Omron CX-Programmer project 新工程 (CX-Programmer 9.50)

# PLC 金泉负压氦检: CJ2M CPU34
I/O table (CPU CJ2M-CPU34): rack 0 slot 11 CJ2M-EIP21

## Global symbols (name address type ; comment)
0.00 BOOL  ; 扫码1#位有料感应（常闭）
0.01 BOOL  ; 扫码2#位有料感应（常闭）
0.02 BOOL  ; 拉带放料位有料感应（常闭）
0.03 BOOL  ; 上料1#位接近有料感应
0.04 BOOL  ; 上料2#位接近有料感应
0.05 BOOL  ; 扫码左位阻挡气缸缩回位
0.06 BOOL  ; 扫码左位阻挡气缸伸出位
0.07 BOOL  ; 扫码右位阻挡气缸缩回位
0.08 BOOL  ; 扫码右位阻挡气缸伸出位
0.09 BOOL  ; 1#位隔离气缸缩回位
0.10 BOOL  ; 左位隔离气缸伸出位
0.11 BOOL  ; 2#位隔离气缸缩回位
0.12 BOOL  ; 右位隔离气缸伸出位
0.13 BOOL  ; 1#隔离位有料感应
0.14 BOOL  ; 2#隔离位有料感应
0.15 BOOL  ; 备用
100.06 BOOL  ; 异常报警停止
100.11 BOOL  ; 报警中
10.00 BOOL  ; 2#隔离气缸缩回
10.01 BOOL  ; 2#隔离气缸伸出
10.02 BOOL  ; 1#隔离气缸缩回
10.03 BOOL  ; 1#隔离气缸伸出
10.04 BOOL  ; 扫码2#阻挡缩回
10.05 BOOL  ; 扫码2#阻挡伸出
10.06 BOOL  ; 扫码1#阻挡缩回
10.07 BOOL  ; 扫码1#阻挡伸出
10.08 BOOL  ; #1调速电机
10.09 BOOL  ; #2调速电机
10.10 BOOL  ; #3调速电机
10.11 BOOL  ; #4调速电机
10.13 BOOL  ; 进料水平伺服使能
10.14 BOOL  ; 进料升降伺服使能
10.15 BOOL  ; 进料升降伺服刹车
11.00 BOOL  ; 进料旋转伺服使能
11.01 BOOL  ; 扫码缓存推料气缸伸出
11.02 BOOL  ; 扫码缓存推料气缸缩回
11.03 BOOL  ; 进料移栽伸缩气缸伸出
11.04 BOOL  ; 进料移栽伸缩气缸缩回
11.05 BOOL  ; 进料#1夹爪气缸夹紧
11.06 BOOL  ; 进料#1夹爪气缸松开
11.07 BOOL  ; 进料#2夹爪气缸夹紧
11.08 BOOL  ; 进料#2夹爪气缸松开
11.09 BOOL  ; 进料水平伺服报警复位
11.10 BOOL  ; 进料升降伺服报警复位
11.11 BOOL  ; 进料旋转伺服报警复位
11.12 BOOL  ; 备用
11.13 BOOL  ; 腔体上料伺服使能
11.14 BOOL  ; 腔体上料提升气缸下降
11.15 BOOL  ; 腔体上料提升气缸上升
12.00 BOOL  ; 腔体上料#1夹爪气缸夹紧
12.01 BOOL  ; 腔体上料#1夹爪气缸松开
12.02 BOOL  ; 腔体上料#2夹爪气缸夹紧
12.03 BOOL  ; 腔体上料#2夹爪气缸松开
12.04 BOOL  ; 腔体上料#3夹爪气缸夹紧
12.05 BOOL  ; 腔体上料#3夹爪气缸松开
12.06 BOOL  ; 腔体上料#4夹爪气缸夹紧
12.07 BOOL  ; 腔体上料#4夹爪气缸松开
12.08 BOOL  ; 腔体下料伺服使能
12.09 BOOL  ; 腔体下料提升气缸下降
12.10 BOOL  ; 腔体下料提升气缸上升
12.11 BOOL  ; 腔体下料#1夹爪气缸夹紧
12.12 BOOL  ; 腔体下料#1夹爪气缸松开
12.13 BOOL  ; 腔体下料#2夹爪气缸夹紧
12.14 BOOL  ; 腔体下料#2夹爪气缸松开
12.15 BOOL  ; 腔体下料#3夹爪气缸夹紧
1311.00 BOOL  ; #1腔体自检步序开始条件
1311.14 BOOL  ; #1腔体自检步序
1311.15 BOOL  ; #1腔体自检步进
1312 CHANNEL  ; 1#腔体自检
1312.00 BOOL  ; #1腔体自检，数据初始化
1312.01 BOOL  ; #1腔体氦检阀打开、合模
1312.02 BOOL  ; #1腔体抽真空
1312.03 BOOL  ; #1腔体进入自检保压前状态
1312.04 BOOL  ; #1腔体进入自检保压状态
1312.05 BOOL  ; #1腔体破真空步
1312.06 BOOL  ; #1腔体自检完成
1313.00 BOOL  ; #1、#2腔体自动条件
1313.01 BOOL  ; #1、#2腔体自动步序递增条件
1313.02 BOOL  ; #1、#2腔体步进递增
1313.05 BOOL  ; 腔体#1 & #2自动启动
1314 CHANNEL  ; #1腔体自动步序
1314.00 BOOL  ; #1、#2腔体自动步序开始
1314.01 BOOL  ; 关闭#1、#2腔体合模气缸，数据初始化
1314.02 BOOL  ; 开始#1、#2腔体抽真空
1314.03 BOOL  ; #1、#2腔体氦检步
1314.04 BOOL  ; #1、#2腔体氦检结果
1314.05 BOOL  ; #1、#2腔体抽残气步
1314.06 BOOL  ; #1、#2腔体氦检结束，腔体破真空步
1314.07 BOOL  ; #1、#2腔体测试结束，开合模，停止吹气，
1314.08 BOOL  ; #1 & #2腔体一个循环结束
1315.00 BOOL  ; #1、#2腔体复检条件
1315.01 BOOL  ; #1、#2腔体在线复检步序递增条件
1315.02 BOOL  ; #1、#2腔体在线复检步进递增
1316 CHANNEL  ; #1、#2复检前抽真空、破真空步进序号
1316.00 BOOL  ; #1、#2腔体在线复检开始，所有数据初始化
1316.01 BOOL  ; 腔体#1、#2复检前抽真空
1316.02 BOOL  ; #1、#2复检前破真空步
1316.03 BOOL  ; #1、#2复检前关破真空阀、抽真空计数步
1316.04 BOOL  ; #1、#2复检抽真空步
1316.05 BOOL  ; #1、#2复检氦检步
1316.06 BOOL  ; #1、#2复检关氦检阀、破真空(复检)步
1316.07 BOOL  ; #1、#2复检关破真空(复检)步
1316.08 BOOL  ; #1、#2清氦抽真空步
1316.09 BOOL  ; #1、#2清氦抽真空计数步
1316.10 BOOL  ; #1、#2清氦氦检步
1316.11 BOOL  ; #1、#2复检清氦破真空步
1316.12 BOOL  ; #1、#2清氦关破真空步
1316.13 BOOL  ; #1、#2清氦选择步
1316.14 BOOL  ; #1、#2复检结束步
1316.15 BOOL  ; #1、#2复检结束步
1321.00 BOOL  ; #2腔体自检步序开始条件
1321.14 BOOL  ; #2腔体自检步序
1321.15 BOOL  ; #2腔体自检步进
1322 CHANNEL  ; #2腔体自检步序
1322.00 BOOL  ; #2腔体自检，数据初始化
1322.01 BOOL  ; #2腔体氦检阀打开、合模
1322.02 BOOL  ; #2腔体抽真空
1322.03 BOOL  ; #2腔体进入自检保压前状态
1322.04 BOOL  ; #2腔体进入自检保压状态
1322.05 BOOL  ; #2腔体破真空步
1322.06 BOOL  ; #2腔体自检完成
1331.00 BOOL  ; #3腔体自检步序开始条件
1331.14 BOOL  ; #3腔体自检步序
1331.15 BOOL  ; #3腔体自检步进
1332.00 BOOL  ; #3腔体自检，数据初始化
1332.01 BOOL  ; #3腔体氦检阀打开、合模
1332.02 BOOL  ; #3腔体抽真空
1332.03 BOOL  ; #3腔体进入自检保压前状态
1332.04 BOOL  ; #3腔体进入自检保压状态
1332.05 BOOL  ; #3腔体破真空步
1332.06 BOOL  ; #3腔体自检完成
1333.00 BOOL  ; #3、#4腔体自动条件
1333.01 BOOL  ; #3、#4腔体自动步序递增条件
1333.02 BOOL  ; #3、#4腔体步进递增
1333.05 BOOL  ; 腔体#3 & #4自动启动
1334 CHANNEL  ; #3、#4腔体自动步序
1334.00 BOOL  ; #3、#4腔体自动步序开始
1334.01 BOOL  ; 关闭#3、#4腔体合模气缸，数据初始化
1334.02 BOOL  ; 开始#3、#4腔体抽真空
1334.03 BOOL  ; #3、#4腔体氦检步
1334.04 BOOL  ; #3、#4腔体氦检结果
1334.05 BOOL  ; #3、#4腔体抽残气步
1334.06 BOOL  ; #3、#4腔体氦检结束，腔体破真空步
1334.07 BOOL  ; #3、#4腔体测试结束，开合模，停止吹气，
1334.08 BOOL  ; #3 & #4腔体一个循环结束
1335.00 BOOL  ; #3、#4腔体复检条件
1335.01 BOOL  ; #3、#4腔体在线复检步序递增条件
1335.02 BOOL  ; #3、#4腔体在线复检步进递增
1336 CHANNEL  ; #3、#4复检前抽真空、破真空步进序号
1336.00 BOOL  ; #3、#4腔体在线复检开始，所有数据初始化
1336.01 BOOL  ; 腔体#3、#4复检前抽真空
1336.02 BOOL  ; #3、#4复检前破真空步
1336.03 BOOL  ; #3、#4复检前关破真空阀、抽真空计数步
1336.04 BOOL  ; #3、#4复检抽真空步
1336.05 BOOL  ; #3、#4复检氦检步
1336.06 BOOL  ; #3、#4复检关氦检阀、破真空(复检)步
1336.07 BOOL  ; #3、#4复检关破真空(复检)步
1336.08 BOOL  ; #3、#4清氦抽真空步
1336.09 BOOL  ; #3、#4清氦抽真空计数步
1336.10 BOOL  ; #3、#4清氦氦检步
1336.11 BOOL  ; #3、#4复检清氦破真空步
1336.12 BOOL  ; #3、#4清氦关破真空步
1336.13 BOOL  ; #3、#4清氦选择步
1336.14 BOOL  ; #3、#4复检结束步
1336.15 BOOL  ; #3、#4复检结束步
1341.00 BOOL  ; #4腔体自检步序开始条件
1341.14 BOOL  ; #4腔体自检步序
1341.15 BOOL  ; #4腔体自检步进
1342.00 BOOL  ; #4腔体自检，数据初始化
1342.01 BOOL  ; #4腔体氦检阀打开、合模
1342.02 BOOL  ; #4腔体抽真空
1342.03 BOOL  ; #4腔体进入自检保压前状态
1342.04 BOOL  ; #4腔体进入自检保压状态
1342.05 BOOL  ; #4腔体破真空步
1342.06 BOOL  ; #4腔体自检完成
1343.00 BOOL  ; 上料水平伺服自动开始条件
1343.01 BOOL  ; 上料水平伺服自动步序递增条件
1343.02 BOOL  ; 上料水平伺服步进递增
1343.05 BOOL  ; 上料机构手自动启动
1344 CHANNEL  ; 上料水平伺服步序
1344.00 BOOL  ; 上料水平伺服开始
1344.01 BOOL  ; 上料水平伺服到取料位
1344.02 BOOL  ; 抓取料
1344.03 BOOL  ; 上料提升气缸回升
1344.04 BOOL  ; 判断腔体放料位置（优先放#1腔体）
1344.05 BOOL  ; 在腔体位置放料
1344.06 BOOL  ; 放料完成，数据传递，气缸回升
1344.07 BOOL  ; 上料水平伺服回上料位
1345.00 BOOL  ; 下料水平伺服自动开始
1345.01 BOOL  ; 下料水平伺服自动步序递增条件
1345.02 BOOL  ; 下料水平伺服步进
1345.05 BOOL  ; 下料机构手自动启动
1345.08 BOOL  ; 放料完成
1346 CHANNEL  ; 下料水平伺服步序
1346.00 BOOL  ; 下料水平伺服步进开始
1346.01 BOOL  ; 下料机构手在放料位判断取料位置(优先取#1腔体)
1346.02 BOOL  ; 下料机构手去腔体(优先取#1腔体)
1346.03 BOOL  ; 下料机构手在腔体位置下降取料
1346.04 BOOL  ; 下料机构手腔体夹料
1346.05 BOOL  ; 机构手上升 腔体→下料夹爪数据传递
1346.06 BOOL  ; 下料机构手回放料位
1346.07 BOOL  ; 下料机构手下降
1346.08 BOOL  ; 下料水平伺服放料松夹
1346.09 BOOL  ; 下料水平伺服放料完成，数据传递，气缸回升
1346.10 BOOL  ; 下料机手一个循环结束
1350.00 BOOL  ; 4-1旋转_Ready Status
1350.01 BOOL  ; 4-1旋转_Home
1350.02 BOOL  ; 4-1旋转_Sub Home
1350.03 BOOL  ; 4-1旋转_Error
1350.04 BOOL  ; 4-1旋转_Warning
1350.05 BOOL  ; 4-1旋转_Home Cmd
1350.06 BOOL  ; 4-1旋转_Auto Stop CMD
1350.07 BOOL  ; 4-1旋转_Stop Cmplt
1350.08 BOOL  ; 4-1旋转_Interlock
1350.09 BOOL  ; 4-1旋转_1Cycle CMD
1350.10 BOOL  ; 4-1旋转_Step+1C+Run
1350.11 BOOL  ; 4-1旋转_1-Cycle End
1350.12 BOOL  ; 4-1旋转_Task Start
1350.13 BOOL  ; 4-1旋转_Task INC Condition
1350.14 BOOL  ; 4-1旋转_Task INC
1350.15 BOOL  ; 4-1旋转_Task Cmplt
1351.00 BOOL  ; 4-1旋转_Cell Move Home SW[T]
1351.01 BOOL  ; 4-1旋转_Step SW[T]
1351.02 BOOL  ; 4-1旋转_1Cycle SW[T]
1351.03 BOOL  ; 4-1旋转_Task Stop SW [T]
1351.04 BOOL  ; 4-1旋转_Task Cmplt SW[T]
1351.05 BOOL  ; 4-1旋转_Task Cmplt Rst SW[T]
1351.06 BOOL  ; 4-1旋转_Product Data Clear SW[T]
1351.07 BOOL  ; 4-1旋转_
1351.08 BOOL  ; 4-1旋转_
1351.09 BOOL  ; 4-1旋转_
1351.10 BOOL  ; 4-1旋转_Step CMD
1351.11 BOOL  ; 4-1旋转_Initial CMD
1351.12 BOOL  ; 4-1旋转_
1351.13 BOOL  ; 4-1旋转_
1351.14 BOOL  ; 4-1旋转_
1351.15 BOOL  ; 4-1旋转_
1352.00 BOOL  ; 4-1旋转_→请求放料
1352.01 BOOL  ; 4-1旋转_←允许旋转
1352.02 BOOL  ; 4-1旋转_→请求取料1&2
1352.03 BOOL  ; 4-1旋转_→请求取料3&4
1352.04 BOOL  ; 4-1旋转_Allow Idx Act-4
1352.05 BOOL  ; 4-1旋转_Allow Idx Act-5
1352.06 BOOL  ; 4-1旋转_Allow Idx Act-6
1352.07 BOOL  ; 4-1旋转_Allow Idx Act-7
1352.08 BOOL  ; 4-1旋转_Allow Idx Act-8
1352.09 BOOL  ; 4-1旋转_Allow Idx Act-9
1352.10 BOOL  ; 4-1旋转_Allow Idx Act-10
1352.11 BOOL  ; 4-1旋转_Allow Idx Act-11
1352.12 BOOL  ; 4-1旋转_Allow Idx Act-12
1352.13 BOOL  ; 4-1旋转_←4-2允许旋转
1352.14 BOOL  ; 4-1旋转_←上下料允许旋转
1352.15 BOOL  ; 4-1旋转_Allow Idx Act-15
1353.00 BOOL  ; 4-1旋转_Step No.
1353.01 BOOL  ; 4-1旋转_
1353.02 BOOL  ; 4-1旋转_
1353.03 BOOL  ; 4-1旋转_
1353.04 BOOL  ; 4-1旋转_
1353.05 BOOL  ; 4-1旋转_
1353.06 BOOL  ; 4-1旋转_
1353.07 BOOL  ; 4-1旋转_
1353.08 BOOL  ; 4-1旋转_
1353.09 BOOL  ; 4-1旋转_
1353.10 BOOL  ; 4-1旋转_
1353.11 BOOL  ; 4-1旋转_
1353.12 BOOL  ; 4-1旋转_
1353.13 BOOL  ; 4-1旋转_
1353.14 BOOL  ; 4-1旋转_
1353.15 BOOL  ; 4-1旋转_
1354 CHANNEL  ; 4-1_出料旋转不序号
1354.00 BOOL  ; 4-1旋转_Run Start
1354.01 BOOL  ; 4-1旋转_Stp001 →请求放料
1354.02 BOOL  ; 4-1旋转_Stp002 ←允许旋转
1354.03 BOOL  ; 4-1旋转_Stp003
1354.04 BOOL  ; 4-1旋转_Stp004 旋转至1&2#放料位/移至放料位
1354.05 BOOL  ; 4-1旋转_Stp005 →请求4-2取料
1354.06 BOOL  ; 4-1旋转_Stp006 ←4-1允许旋转
1354.07 BOOL  ; 4-1旋转_Stp007
1354.08 BOOL  ; 4-1旋转_Stp008 4-1旋转_Stp004 旋转至3&4#放料位
1354.09 BOOL  ; 4-1旋转_Stp009→请求4-2取料
1354.10 BOOL  ; 4-1旋转_Stp010←4-1允许旋转
1354.11 BOOL  ; 4-1旋转_Stp011 旋转至待机位/移至装载位
1354.12 BOOL  ; 4-1旋转_Stp012
1354.13 BOOL  ; 4-1旋转_Stp013
1354.14 BOOL  ; 4-1旋转_Stp014
1354.15 BOOL  ; 4-1旋转_Stp015
1355.00 BOOL  ; 4-1旋转_Stp016
1355.01 BOOL  ; 4-1旋转_Stp017
1355.02 BOOL  ; 4-1旋转_Stp018
1355.03 BOOL  ; 4-1旋转_Stp019
1355.04 BOOL  ; 4-1旋转_Stp020
1355.05 BOOL  ; 4-1旋转_Stp021
1355.06 BOOL  ; 4-1旋转_Stp022
1355.07 BOOL  ; 4-1旋转_Stp023
1355.08 BOOL  ; 4-1旋转_Stp024
1355.09 BOOL  ; 4-1旋转_Stp025
1355.10 BOOL  ; 4-1旋转_Stp026
1355.11 BOOL  ; 4-1旋转_Stp027
1355.12 BOOL  ; 4-1旋转_Stp028
1355.13 BOOL  ; 4-1旋转_Stp029
1355.14 BOOL  ; 4-1旋转_Stp030
1355.15 BOOL  ; 4-1旋转_Stp031
1356.00 BOOL  ; 4-1旋转_Home
1356.01 BOOL  ; 4-1旋转_Sub Home
1356.02 BOOL  ; 4-1旋转_
1356.03 BOOL  ; 4-1旋转_
1356.04 BOOL  ; 4-1旋转_
1356.05 BOOL  ; 4-1旋转_
1356.06 BOOL  ; 4-1旋转_
1356.07 BOOL  ; 4-1旋转_
1356.08 BOOL  ; 4-1旋转_
1356.09 BOOL  ; 4-1旋转_
1356.10 BOOL  ; 4-1旋转_
1356.11 BOOL  ; 4-1旋转_
1356.12 BOOL  ; 4-1旋转_
1356.13 BOOL  ; 4-1旋转_
1356.14 BOOL  ; 4-1旋转_
1356.15 BOOL  ; 4-1旋转_
1357.00 BOOL  ; 4-1旋转_Error
1357.01 BOOL  ; 4-1旋转_Warning
1357.02 BOOL  ; 4-1旋转_Step+1C+Run
1357.03 BOOL  ; 4-1旋转_
1357.04 BOOL  ; 4-1旋转_
1357.05 BOOL  ; 4-1旋转_
1357.06 BOOL  ; 4-1旋转_
1357.07 BOOL  ; 4-1旋转_
1357.08 BOOL  ; 4-1旋转_
1357.09 BOOL  ; 4-1旋转_
1357.10 BOOL  ; 4-1旋转_
1357.11 BOOL  ; 4-1旋转_
1357.12 BOOL  ; 4-1旋转_
1357.13 BOOL  ; 4-1旋转_
1357.14 BOOL  ; 4-1旋转_
1357.15 BOOL  ; 4-1旋转_
1358.00 BOOL  ; 4-1旋转_
1358.01 BOOL  ; 4-1旋转_
1358.02 BOOL  ; 4-1旋转_
1358.03 BOOL  ; 4-1旋转_
1358.04 BOOL  ; 4-1旋转_
1358.05 BOOL  ; 4-1旋转_
1358.06 BOOL  ; 4-1旋转_
1358.07 BOOL  ; 4-1旋转_
1358.08 BOOL  ; 4-1旋转_
1358.09 BOOL  ; 4-1旋转_
1358.10 BOOL  ; 4-1旋转_
1358.11 BOOL  ; 4-1旋转_
1358.12 BOOL  ; 4-1旋转_
1358.13 BOOL  ; 4-1旋转_
1358.14 BOOL  ; 4-1旋转_
1358.15 BOOL  ; 4-1旋转_
1359.00 BOOL  ; 4-1旋转_Initial-1
1359.01 BOOL  ; 4-1旋转_Initial-2
1359.02 BOOL  ; 4-1旋转_Initial-3
1359.03 BOOL  ; 4-1旋转_Initial-4
1359.04 BOOL  ; 4-1旋转_Initial-5
1359.05 BOOL  ; 4-1旋转_Initial-6
1359.06 BOOL  ; 4-1旋转_Initial-7
1359.07 BOOL  ; 4-1旋转_Initial-8
1359.08 BOOL  ; 4-1旋转_Initial-9
1359.09 BOOL  ; 4-1旋转_Initial-10
1359.10 BOOL  ; 4-1旋转_Initial-11
1359.11 BOOL  ; 4-1旋转_Initial-12
1359.12 BOOL  ; 4-1旋转_Initial-13
1359.13 BOOL  ; 4-1旋转_Initial-14
1359.14 BOOL  ; 4-1旋转_Initial-15
1359.15 BOOL  ; 4-1旋转_Initial-16
1360.00 BOOL  ; 4-2出料模组_Ready Status
1360.01 BOOL  ; 4-2出料模组_Home
1360.02 BOOL  ; 4-2出料模组_Sub Home
1360.03 BOOL  ; 4-2出料模组_Error
1360.04 BOOL  ; 4-2出料模组_Warning
1360.05 BOOL  ; 4-2出料模组_Home Cmd
1360.06 BOOL  ; 4-2出料模组_Auto Stop CMD
1360.07 BOOL  ; 4-2出料模组_Stop Cmplt
1360.08 BOOL  ; 4-2出料模组_Interlock
1360.09 BOOL  ; 4-2出料模组_1Cycle CMD
1360.10 BOOL  ; 4-2出料模组_Step+1C+Run
1360.11 BOOL  ; 4-2出料模组_1-Cycle End
1360.12 BOOL  ; 4-2出料模组_Task Start
1360.13 BOOL  ; 4-2出料模组_Task INC Condition
1360.14 BOOL  ; 4-2出料模组_Task INC
1360.15 BOOL  ; 4-2出料模组_Task Cmplt
1361.00 BOOL  ; 4-2出料模组_Cell Move Home SW[T]
1361.01 BOOL  ; 4-2出料模组_Step SW[T]
1361.02 BOOL  ; 4-2出料模组_1Cycle SW[T]
1361.03 BOOL  ; 4-2出料模组_Task Stop SW [T]
1361.04 BOOL  ; 4-2出料模组_Task Cmplt SW[T]
1361.05 BOOL  ; 4-2出料模组_Task Cmplt Rst SW[T]
1361.06 BOOL  ; 4-2出料模组_Product Data Clear SW[T]
1361.07 BOOL  ; 4-2出料模组_
1361.08 BOOL  ; 4-2出料模组_
1361.09 BOOL  ; 4-2出料模组_
1361.10 BOOL  ; 4-2出料模组_Step CMD
1361.11 BOOL  ; 4-2出料模组_Initial CMD
1361.12 BOOL  ; 4-2出料模组_
1361.13 BOOL  ; 4-2出料模组_
1361.14 BOOL  ; 4-2出料模组_
1361.15 BOOL  ; 4-2出料模组_
1362.00 BOOL  ; 4-2出料模组_→Idx Act-0
1362.01 BOOL  ; 4-2出料模组_Allow Idx Act-1
1362.02 BOOL  ; 4-2出料模组_Allow Idx Act-2
1362.03 BOOL  ; 4-2出料模组_NG缓存自动运行
1362.04 BOOL  ; 1#NG 允许动作
1362.05 BOOL  ; 2#NG 允许动作
1362.06 BOOL  ; NG缓存动作中[伸出]
1362.07 BOOL  ; NG缓存推料气缸[缩回]
1362.08 BOOL  ; 推料完成
1362.09 BOOL  ; 4-2出料模组_Allow Idx Act-9
1362.10 BOOL  ; 4-2出料模组_Allow Idx Act-10
1362.11 BOOL  ; 4-2出料模组_Allow Idx Act-11
1362.12 BOOL  ; 4-2出料模组_Allow Idx Act-12
1362.13 BOOL  ; 4-2出料2#NG优先选择
1362.14 BOOL  ; 4-2出料NG料槽已满，请取走电芯，谢谢！
1362.15 BOOL  ; 4-2出料模组_Allow Idx Act-15
1363.00 BOOL  ; 4-2出料模组_Step No.
1363.01 BOOL  ; 4-2出料模组_
1363.02 BOOL  ; 4-2出料模组_
1363.03 BOOL  ; 4-2出料模组_
1363.04 BOOL  ; 4-2出料模组_
1363.05 BOOL  ; 4-2出料模组_
1363.06 BOOL  ; 4-2出料模组_
1363.07 BOOL  ; 4-2出料模组_
1363.08 BOOL  ; 4-2出料模组_
1363.09 BOOL  ; 4-2出料模组_
1363.10 BOOL  ; 4-2出料模组_
1363.11 BOOL  ; 4-2出料模组_
1363.12 BOOL  ; 4-2出料模组_
1363.13 BOOL  ; 4-2出料模组_
1363.14 BOOL  ; 4-2出料模组_
1363.15 BOOL  ; 4-2出料模组_
1364.00 BOOL  ; 4-2出料模组_Run Start
1364.01 BOOL  ; 4-2出料模组_Stp001 →取料请求
1364.02 BOOL  ; 4-2出料模组_Stp002
1364.03 BOOL  ; 4-2出料模组_Stp003 Z轴至下降位（取料）
1364.04 BOOL  ; 4-2出料模组_Stp004 夹取和数据传递
1364.05 BOOL  ; 4-2出料模组_Stp005
1364.06 BOOL  ; 4-2出料模组_Stp006 Z轴至上升位
1364.07 BOOL  ; 4-2出料模组_Stp007 X至NG位/OK位
1364.08 BOOL  ; 4-2出料模组_Stp007 X至NG位/OK位
1364.09 BOOL  ; 4-2出料模组_Stp008 Z轴下降（放料）
1364.10 BOOL  ; 4-2出料模组_Stp009 松开
1364.11 BOOL  ; 4-2出料模组_Stp010 Z轴上升
1364.12 BOOL  ; 4-2出料模组_Stp011 X轴至取料位
1364.13 BOOL  ; 4-2出料模组_Stp012
1364.14 BOOL  ; 4-2出料模组_Stp013
1364.14 BOOL  ; 4-2出料模组_Stp014
1364.15 BOOL  ; 4-2出料模组_Stp015
1365.00 BOOL  ; 4-2出料模组_Stp016
1365.01 BOOL  ; 4-2出料模组_Stp017
1365.02 BOOL  ; 4-2出料模组_Stp018
1365.03 BOOL  ; 4-2出料模组_Stp019
1365.04 BOOL  ; 4-2出料模组_Stp020
1365.05 BOOL  ; 4-2出料模组_Stp021
1365.06 BOOL  ; 4-2出料模组_Stp022
1365.07 BOOL  ; 4-2出料模组_Stp023
1365.08 BOOL  ; 4-2出料模组_Stp024
1365.09 BOOL  ; 4-2出料模组_Stp025
1365.10 BOOL  ; 4-2出料模组_Stp026
1365.11 BOOL  ; 4-2出料模组_Stp027
1365.12 BOOL  ; 4-2出料模组_Stp028
1365.13 BOOL  ; 4-2出料模组_Stp029
1365.14 BOOL  ; 4-2出料模组_Stp030
1365.15 BOOL  ; 4-2出料模组_Stp031
1366.00 BOOL  ; 4-2出料模组_Home
1366.01 BOOL  ; 4-2出料模组_Sub Home
1366.02 BOOL  ; 4-2出料模组_
1366.03 BOOL  ; 4-2出料模组_
1366.04 BOOL  ; 4-2出料模组_
1366.05 BOOL  ; 4-2出料模组_
1366.06 BOOL  ; 4-2出料模组_
1366.07 BOOL  ; 4-2出料模组_
1366.08 BOOL  ; 4-2出料模组_
1366.09 BOOL  ; 4-2出料模组_
1366.10 BOOL  ; 4-2出料模组_
1366.11 BOOL  ; 4-2出料模组_
1366.12 BOOL  ; 4-2出料模组_
1366.13 BOOL  ; 4-2出料模组_
1366.14 BOOL  ; 4-2出料模组_
1366.15 BOOL  ; 4-2出料模组_
1367.00 BOOL  ; 4-2出料模组_Error
1367.01 BOOL  ; 4-2出料模组_Warning
1367.02 BOOL  ; 4-2出料模组_Step+1C+Run
1367.03 BOOL  ; 4-2出料模组_
1367.04 BOOL  ; 4-2出料模组_
1367.05 BOOL  ; 4-2出料模组_
1367.06 BOOL  ; 4-2出料模组_
1367.07 BOOL  ; 4-2出料模组_
1367.08 BOOL  ; 4-2出料模组_
1367.09 BOOL  ; 4-2出料模组_
1367.10 BOOL  ; 4-2出料模组_
1367.11 BOOL  ; 4-2出料模组_
1367.12 BOOL  ; 4-2出料模组_
1367.13 BOOL  ; 4-2出料模组_
1367.14 BOOL  ; 4-2出料模组_
1367.15 BOOL  ; 4-2出料模组_
1368.00 BOOL  ; 4-2出料模组_
1368.01 BOOL  ; 4-2出料模组_
1368.02 BOOL  ; 4-2出料模组_
1368.03 BOOL  ; 4-2出料模组_
1368.04 BOOL  ; 4-2出料模组_
1368.05 BOOL  ; 4-2出料模组_
1368.06 BOOL  ; 4-2出料模组_
1368.07 BOOL  ; 4-2出料模组_
1368.08 BOOL  ; 4-2出料模组_
1368.09 BOOL  ; 4-2出料模组_
1368.10 BOOL  ; 检测NG推料气缸缩回复位
1368.11 BOOL  ; 4-2出料模组_
1368.12 BOOL  ; 4-2出料模组_
1368.13 BOOL  ; 4-2出料模组_
1368.14 BOOL  ; 4-2出料模组_
1368.15 BOOL  ; 4-2出料模组_
1369.00 BOOL  ; 4-2出料模组_Initial-1
1369.01 BOOL  ; 4-2出料模组_Initial-2
1369.02 BOOL  ; 4-2出料模组_Initial-3
1369.03 BOOL  ; 4-2出料模组_Initial-4
1369.04 BOOL  ; 4-2出料模组_Initial-5
1369.05 BOOL  ; 4-2出料模组_Initial-6
1369.06 BOOL  ; 4-2出料模组_Initial-7
1369.07 BOOL  ; 4-2出料模组_Initial-8
1369.08 BOOL  ; 4-2出料模组_Initial-9
1369.09 BOOL  ; 4-2出料模组_Initial-10
1369.10 BOOL  ; 4-2出料模组_Initial-11
1369.11 BOOL  ; 4-2出料模组_Initial-12
1369.12 BOOL  ; 4-2出料模组_Initial-13
1369.13 BOOL  ; 4-2出料模组_Initial-14
1369.14 BOOL  ; 4-2出料模组_Initial-15
1369.15 BOOL  ; 4-2出料模组_Initial-16
1390.00 BOOL  ; 进料输送机构初始位
1390.01 BOOL  ; 进料输送执行条件
1390.02 BOOL  ; 进料输送机构自动步进条件
1390.05 BOOL  ; 重复1#扫码
1390.06 BOOL  ; 重复2#扫码
1390.15 BOOL  ; 进料输送机构步序移位
1391 CHANNEL  ; 进料输送机构自动步序
1391.00 BOOL  ; 进料输送步序开始
1391.01 BOOL  ; 进料输送马达运转
1391.02 BOOL  ; 左右隔离气缸伸出
1391.03 BOOL  ; 进料输送马达停止
1391.04 BOOL  ; 扫码开始
1391.05 BOOL  ; 进料输送马达运转
1391.06 BOOL  ; 左右阻挡气缸缩回
1391.07 BOOL  ; 进料输送马达运转
1391.08 BOOL  ; 左右阻挡气缸伸出、电机停止
1391.09 BOOL  ; 左右隔离气缸缩回
1391.10 BOOL  ; 步序循环结束
1391.11 BOOL  ; 左右隔离气缸缩回
1391.12 BOOL  ; 步序循环结束
1391.13 BOOL  ; 步序循环结束
1398.00 BOOL  ; 放料缓存步序条件
1398.02 BOOL  ; 直接NG缓存放料条件
1398.14 BOOL  ; NG放料步进
1398.15 BOOL  ; 放料缓存步进
1399.00 BOOL  ; 配对缓存步序条件
1399.12 BOOL  ; 直接NG缓存放料条件
1399.13 BOOL  ; 放料缓存运行
13.00 BOOL  ; 腔体下料#3夹爪气缸松开
13.01 BOOL  ; 腔体下料#4夹爪气缸夹紧
13.02 BOOL  ; 腔体下料#4夹爪气缸松开
13.03 BOOL  ; 上料伺服报警复位
13.04 BOOL  ; 腔体下料伺服报警复位
13.05 BOOL  ; 备用
13.06 BOOL  ; 备用
13.07 BOOL  ; #1合模气缸缩回
13.08 BOOL  ; #1合模气缸伸出
13.09 BOOL  ; #2合模气缸缩回
13.10 BOOL  ; #2合模气缸伸出
13.11 BOOL  ; #3合模气缸缩回
13.12 BOOL  ; #3合模气缸伸出
13.13 BOOL  ; #4合模气缸缩回
13.14 BOOL  ; #4合模气缸伸出
13.15 BOOL  ; 备用
1400.00 BOOL  ; 进料机构正常放料执行
1400.01 BOOL  ; 进料机构缓存放料
1400.02 BOOL  ; 进料机构缓存取料
1400.03 BOOL  ; 进料机构自动步进条件
1400.04 BOOL  ; 进料旋转初始条件
1400.05 BOOL  ; 进料机构自动步进移位
1400.06 BOOL  ; 进料机构正常放料执行
1400.07 BOOL  ; 进料机构旋转步进条件
1400.08 BOOL  ; 进料机构旋转步进
1400.09 BOOL  ; 配对缓存初始条件
1400.10 BOOL  ; 执行配对
1400.11 BOOL  ; 执行正常上料
1400.12 BOOL  ; 进料旋转运行
1400.13 BOOL  ; 配对缓存运行
1400.14 BOOL  ; 配对缓存启动运行
1400.15 BOOL  ; 配对缓存步进
1401 CHANNEL  ; 进料伺服自动步序
1401.00 BOOL  ; 进料机构自动开始
1401.01 BOOL  ; 进料升降至取料位
1401.02 BOOL  ; 进料左右夹爪夹紧
1401.03 BOOL  ; 进料升降伺服取料后回待料位
1401.04 BOOL  ; 进料水平伺服平移到放料位
1401.05 BOOL  ; 进料升降伺服至放料位
1401.06 BOOL  ; 进料左右夹爪松开
1401.07 BOOL  ; 进料机构升降回待料位
1401.08 BOOL  ; 进料水平伺服回取料位
1401.09 BOOL  ; 循环结束
1402 CHANNEL  ; 进料旋转步
1402.00 BOOL  ; 进料旋转机构步序开始
1402.01 BOOL  ; 进料旋转气缸伸出
1402.02 BOOL  ; 进料旋转启动(到#1待料位)
1402.03 BOOL  ; 进料旋转伺服到#2待料位
1402.04 BOOL  ; 进料旋转伺服回上料位
1402.05 BOOL  ; 进料旋转气缸缩回
1402.06 BOOL  ; 对接等待
1402.07 BOOL  ; 进料旋转气缸伸出
1402.08 BOOL  ; 循环完成
1402.09 BOOL  ; 循环完成
1403 CHANNEL  ; 配对缓存自动步序
1403.00 BOOL  ; 步序开始
1403.01 BOOL  ; 判断NG位左/右缓存
1403.02 BOOL  ; 升降至NG缓存位
1403.03 BOOL  ; 进料夹爪张开放料
1403.04 BOOL  ; 进料升降伺服回待料位
1403.05 BOOL  ; NG缓存推料气缸伸出
1403.06 BOOL  ; 判断配对取料位
1403.07 BOOL  ; NG缓存推料气缸缩回
1403.08 BOOL  ; 进料升降伺服至配对位抓料
1403.09 BOOL  ; 进料升降夹爪夹紧
1403.10 BOOL  ; 进料升降回待料位
1403.11 BOOL  ; 配对完成
1403.12 BOOL  ; 配对步序循环完成
1404.00 BOOL  ; 放料缓存步序开始
1404.01 BOOL  ; 升降至配对位放OK料
1404.02 BOOL  ; 夹爪张开放OK料
1404.03 BOOL  ; 进料升降回待料位
1404.04 BOOL  ; 升降至NG缓存位放料
1404.05 BOOL  ; 夹爪张开放NG料
1404.06 BOOL  ; 进料升降回待料位
1404.07 BOOL  ; NG缓存推料气缸伸出
1404.08 BOOL  ; 预留
1404.09 BOOL  ; 进料夹爪无料回取料位
1404.10 BOOL  ; NG缓存推料气缸缩回
1404.11 BOOL  ; 预留
1404.12 BOOL  ; 放料缓存循环结束
1405.00 BOOL  ; 直接NG缓存放料开始
1405.01 BOOL  ; 进料机构至NG缓存位
1405.02 BOOL  ; 升降伺服至缓存放料位
1405.03 BOOL  ; 夹爪张开放NG料
1405.04 BOOL  ; 进料升降回待料位
1405.05 BOOL  ; 进料夹爪无料回取料位
1405.06 BOOL  ; 循环完成
1405.07 BOOL  ; NG缓存推料气缸缩回
1405.08 BOOL  ; 循环完成
1420.10 BOOL  ; #1腔体自检步序开始条件
1420.13 BOOL  ; #1腔体自检步序
1420.14 BOOL  ; #1腔体自检步进
1423 CHANNEL  ; #1腔体自检（复检）步序
1424 CHANNEL  ; #1腔体自检
1424.00 BOOL  ; #1腔体自检，数据初始化
1424.01 BOOL  ; #1腔体抽真空
1424.02 BOOL  ; #1腔体进入自检保压前状态
1424.03 BOOL  ; #1腔体进入自检保压状态
1424.04 BOOL  ; #1腔体破真空步
1424.05 BOOL  ; #1腔体自检完成
1425 CHANNEL  ; #2腔体自检步序
1425.00 BOOL  ; #2腔体自检，数据初始化
1425.01 BOOL  ; #2腔体抽真空
1425.02 BOOL  ; #2腔体进入自检保压前状态
1425.03 BOOL  ; #2腔体进入自检保压状态
1425.04 BOOL  ; #2腔体破真空步
1425.05 BOOL  ; #2腔体自检完成
1426 CHANNEL  ; #2腔体自检（复检）步序
1426.00 BOOL  ; #2腔体自检步序开始（关闭合模，数据初始化）
1427.10 BOOL  ; #2腔体自检步序开始条件
1427.13 BOOL  ; #2腔体自检步序条件
1427.14 BOOL  ; #2腔体自检步进
14.00 BOOL  ; 备用
14.01 BOOL  ; #1抽真空阀
14.02 BOOL  ; #2抽真空阀
14.03 BOOL  ; #3抽真空阀
14.04 BOOL  ; #4抽真空阀
14.05 BOOL  ; #1总氦检阀
14.06 BOOL  ; #2总氦检阀
14.07 BOOL  ; #1氦检阀
14.08 BOOL  ; #2氦检阀
14.09 BOOL  ; #3氦检阀
14.10 BOOL  ; #4氦检阀
14.11 BOOL  ; #1破真空阀
14.12 BOOL  ; #2破真空阀
14.13 BOOL  ; #3破真空阀
14.14 BOOL  ; #4破真空阀
14.15 BOOL  ; #1吹气阀
1534.15 BOOL  ; 单元1的串口1执行中标志
1544.15 BOOL  ; 单元1的串口2执行标志
1550.03 BOOL  ; 单元2串口1异常退出
1559.15 BOOL  ; 单元2的串口1执行标志
1584.15 BOOL  ; 单元3的串口1执行中标志
1594.15 BOOL  ; 单元3的串口2执行标志
15.00 BOOL  ; #2吹气阀
15.01 BOOL  ; #3吹气阀
15.02 BOOL  ; #4吹气阀
15.03 BOOL  ; 备用
15.04 BOOL  ; 备用
15.05 BOOL  ; 备用
15.06 BOOL  ; 备用
15.07 BOOL  ; 备用
15.08 BOOL  ; 备用
15.09 BOOL  ; 备用
15.10 BOOL  ; 备用
15.11 BOOL  ; 备用
15.12 BOOL  ; 备用
15.13 BOOL  ; 放料请求
15.14 BOOL  ; 备用
15.15 BOOL  ; 备用
1600.00 BOOL  ; NG位左缓存放左爪NG料
1600.01 BOOL  ; 去缓存放1#爪扫码NG料
1600.02 BOOL  ; 去右配对位取料
1600.03 BOOL  ; 去NG缓存放2#爪NG料
1600.04 BOOL  ; 去左配对位取料
1600.05 BOOL  ; NG位缓存放1#爪NG料
1600.06 BOOL  ; 放爪扫码NG位
1600.07 BOOL  ; 去NG缓存位放1#2#爪NG料
1600.08 BOOL  ; NG缓存位放2#爪NG料
1600.09 BOOL  ; 去OK配对位抓料
1600.10 BOOL  ; 去NG位放NG料
1600.11 BOOL  ; 去水平放料位放料
1600.12 BOOL  ; 去左配对位抓料
1600.13 BOOL  ; 去配对位抓料
16.00 BOOL  ; 出料水平伺服使能
16.01 BOOL  ; 出料升降伺服使能
16.02 BOOL  ; 出料升降伺服刹车
16.03 BOOL  ; 出料旋转伺服使能
16.04 BOOL  ; 出料移栽伸缩气缸伸出
16.05 BOOL  ; 出料移栽伸缩气缸缩回
16.06 BOOL  ; 检测NG缓存推料气缸伸出
16.07 BOOL  ; 检测NG缓存推料气缸缩回
16.08 BOOL  ; 出料#1夹爪气缸夹紧
16.09 BOOL  ; 出料#1夹爪气缸张开
16.10 BOOL  ; 出料#2夹爪气缸夹紧
16.11 BOOL  ; 出料#2夹爪气缸张开
16.12 BOOL  ; 出料水平伺服报警复位
16.13 BOOL  ; 出料升降伺服报警复位
16.14 BOOL  ; 出料旋转伺服报警复位
1700.00 BOOL  ; 进料平移伺服到达
1700.01 BOOL  ; 进料放料缓存配对位开始
1700.02 BOOL  ; 放OK料后到达NG缓存位
1700.03 BOOL  ; 放NG料到达NG缓存位
1700.05 BOOL  ; 进料平移在取料位
17.00 BOOL  ; 氦检仪启动
17.01 BOOL  ; #1真空泵
17.02 BOOL  ; #2真空泵
17.03 BOOL  ; 启动指示灯
17.04 BOOL  ; 停止指示灯
17.05 BOOL  ; 复位指示灯
17.06 BOOL  ; 三色红灯
17.07 BOOL  ; 三色黄灯
17.08 BOOL  ; 三色绿灯
17.09 BOOL  ; 蜂鸣器
17.10 BOOL  ; $?St$Bk?_#[4] / 氦检仪 / 电源$?St$Bk?_#[4]
1.00 BOOL  ; 备用
1.02 BOOL  ; 备用
1.03 BOOL  ; 备用
1.04 BOOL  ; 扫码OK配对位有料感应（常闭）
1.05 BOOL  ; 扫码NG缓存#1有料感应
1.06 BOOL  ; 扫码NG缓存#2有料感应
1.07 BOOL  ; NG位缓存对射有料感应
1.08 BOOL  ; 进料移栽料盘放料位有料感应（常闭）
1.09 BOOL  ; 备用
1.10 BOOL  ; 备用
1.11 BOOL  ; 备用
1.12 BOOL  ; 备用
1.13 BOOL  ; 进料水平伺服准备就绪
1.14 BOOL  ; 进料水平伺服报警
1.15 BOOL  ; 进料升降伺服准备就绪
2000.03 BOOL  ; 进料升降伺服绝对移动
2000.09 BOOL  ; 进料升降伺服点动
2000.10 BOOL  ; 进料升降伺服方向
2000.12 BOOL  ; 进料升降伺服复位
2000.15 BOOL  ; 进料升降伺服停止
2002.03 BOOL  ; 进料移栽伺服绝对移动
2002.06 BOOL  ; 进料旋转伺服归零
2002.09 BOOL  ; 进料旋转伺服点动
2002.10 BOOL  ; 进料旋转伺服方向
2002.12 BOOL  ; 进料旋转伺服报警复位
2002.15 BOOL  ; 进料旋转伺服停止
2004.03 BOOL  ; 出料升降伺服绝对移动
2004.06 BOOL  ; 出料升降伺服归零
2004.09 BOOL  ; 出料升降伺服点动
2004.10 BOOL  ; 出料升降伺服点动方向
2004.12 BOOL  ; 出料升降伺服报警复位
2004.15 BOOL  ; 出料升降伺服停止
2006.03 BOOL  ; 出料移栽伺服绝对移动
2006.06 BOOL  ; 出料移栽伺服归零
2006.09 BOOL  ; 出料移栽伺服点动
2006.10 BOOL  ; 出料移栽伺服点动方向
2006.12 BOOL  ; 出料移栽伺服报警复位
2006.15 BOOL  ; 出料移栽伺服停止
2008.06 BOOL  ; 进料升降伺服无原点标志
2008.13 BOOL  ; 进料升降伺服忙标志
2009.08 BOOL  ; 进料升降伺服正极限
2009.09 BOOL  ; 进料升降伺服负极限
2010 CHANNEL  ; 进料升降伺服错误代码
2011.06 BOOL  ; 进料移栽伺服无原点标志
2011.13 BOOL  ; 进料旋转伺服忙标志
2012.08 BOOL  ; 进料旋转伺服正极限
2012.09 BOOL  ; 进料旋转伺服负极限
2013 CHANNEL  ; 进料旋转伺服错误代码
2014.06 BOOL  ; 出料升降伺服无原点
2014.13 BOOL  ; 出料升降伺服脉冲输出中
2015.08 BOOL  ; 出料升降伺服正极限
2015.09 BOOL  ; 出料升降伺服负极限
2016 CHANNEL  ; 出料升降伺服错误代码
2017.06 BOOL  ; 出料移栽伺服无原点
2017.13 BOOL  ; 出料移栽伺服脉冲输出中
2018.08 BOOL  ; 出料移栽伺服正极限
2018.09 BOOL  ; 出料移栽伺服负极限
2019 CHANNEL  ; 出料移栽伺服错误代码
2031 CHANNEL  ; #1真空计读出数值
2032 CHANNEL  ; #2真空计读出数值
20.06 BOOL  ; 氦检仪内部校准
20.12 BOOL  ; 氦检仪内部校准
2960.00 BOOL  ; $?St$Bk?_#[5] / 上料水平伺服原点 / 上料水平伺服原点 / 腔体上料伺服原点$?St$Bk?_#[5]
2960.02 BOOL  ; $?St$Bk?_#[6] / 上料水平伺服原点 / 上料水平伺服原点 / 腔体下料伺服原点$?St$Bk?_#[6]
2960.06 BOOL  ; 进料水平伺服负极限
2960.07 BOOL  ; 进料水平伺服正极限
2960.08 BOOL  ; 出料水平伺服负极限
2960.09 BOOL  ; 出料水平伺服正极限
2962.06 BOOL  ; 上料水平伺服负极限
2962.07 BOOL  ; 上料水平伺服正极限
2962.08 BOOL  ; 下料水平伺服负极限
2962.09 BOOL  ; 下料水平伺服正极限
2.00 BOOL  ; 进料升降伺服报警
2.01 BOOL  ; 进料升降伺服柔性报警
2.02 BOOL  ; 进料旋转伺服准备就绪
2.03 BOOL  ; 进料旋转伺服报警
2.04 BOOL  ; 扫码NG料缓存推料气缸缩回位
2.05 BOOL  ; 扫码NG料缓存推料气缸伸出位
2.06 BOOL  ; 备用
2.07 BOOL  ; 备用
2.08 BOOL  ; 备用
2.09 BOOL  ; 备用
2.10 BOOL  ; 进料移栽伸缩气缸缩回位
2.11 BOOL  ; 进料移栽伸缩气缸伸出位
2.12 BOOL  ; 进料#1夹爪张开位
2.13 BOOL  ; 进料#1夹爪夹紧位
2.14 BOOL  ; 进料#2夹爪张开位
2.15 BOOL  ; 进料#2夹爪夹紧位
303.05 BOOL  ; 进料升降伺服异常
304.02 BOOL  ; 上料水平伺服正极限异常
304.14 BOOL  ; 下料提升气缸柔性异常
30.01 BOOL  ; 进料机构复位
30.02 BOOL  ; 上下料机构手复位
30.03 BOOL  ; 腔体机构手复位
30.04 BOOL  ; 出料机构手复位
3800.06 BOOL  ; 进料平移在取料位
3.00 BOOL  ; 备用
3.01 BOOL  ; 备用
3.02 BOOL  ; 备用
3.03 BOOL  ; 备用
3.04 BOOL  ; 备用
3.05 BOOL  ; 备用
3.06 BOOL  ; 腔体上料准备就绪
3.07 BOOL  ; 腔体上料报警
3.08 BOOL  ; 腔体上料柔性报警
3.09 BOOL  ; 腔体上料提升气缸缩回位
3.10 BOOL  ; 腔体上料提升气缸伸出位
3.11 BOOL  ; 腔体上料#1夹爪张开位
3.12 BOOL  ; 腔体上料#1夹爪夹紧位
3.13 BOOL  ; 腔体上料#2夹爪张开位
3.14 BOOL  ; 腔体上料#2夹爪夹紧位
3.15 BOOL  ; 腔体上料#3夹爪张开位
40.00 BOOL  ; 进料机构初始位
40.01 BOOL  ; 进料机构初始位
40.02 BOOL  ; 进料机构升降初始位
40.03 BOOL  ; 进料旋转机构初始位
41.10 BOOL  ; 进料机构感应器异常
41.11 BOOL  ; 进料机构出错
45.00 BOOL  ; 进料机构 出错
4.00 BOOL  ; 腔体上料#3夹爪夹紧位
4.01 BOOL  ; 腔体上料#4夹爪张开位
4.02 BOOL  ; 腔体上料#4夹爪夹紧位
4.03 BOOL  ; 备用
4.04 BOOL  ; 备用
4.05 BOOL  ; 备用
4.06 BOOL  ; 备用
4.07 BOOL  ; 腔体下料伺服准备就绪
4.08 BOOL  ; 腔体下料伺服报警
4.09 BOOL  ; 腔体下料伺服柔性报警
4.10 BOOL  ; 腔体下料提升气缸缩回位
4.11 BOOL  ; 腔体下料提升气缸伸出位
4.12 BOOL  ; 腔体下料#1夹爪张开位
4.13 BOOL  ; 腔体下料#1夹爪夹紧位
4.14 BOOL  ; 腔体下料#2夹爪张开位
4.15 BOOL  ; 腔体下料#2夹爪夹紧位
50.00 BOOL  ; 上下料机构手在初始位
50.01 BOOL  ; 上料机构手在初始位
50.02 BOOL  ; 下料机构手在初始位
50.05 BOOL  ; 整机初始化(HMI)(SW)
50.06 BOOL  ; 整机记忆清除
51.10 BOOL  ; 上料机构手感应器异常
51.11 BOOL  ; 上料机构手 出错
52.10 BOOL  ; 下料机构手感应器异常
52.11 BOOL  ; 下料机构手 出错
53.00 BOOL  ; 上料机手复位
54.00 BOOL  ; 下料机手复位
55.00 BOOL  ; 上下料机构手 出错
5.00 BOOL  ; 腔体下料#3夹爪张开位
5.01 BOOL  ; 腔体下料#3夹爪夹紧位
5.02 BOOL  ; 腔体下料#4夹爪张开位
5.03 BOOL  ; 腔体下料#4夹爪夹紧位
5.04 BOOL  ; 备用
5.05 BOOL  ; 备用
5.06 BOOL  ; 备用
5.07 BOOL  ; 备用
5.08 BOOL  ; #1合模气缸缩回位
5.09 BOOL  ; #1合模气缸伸出位
5.10 BOOL  ; #2合模气缸缩回位
5.11 BOOL  ; #2合模气缸伸出位
5.12 BOOL  ; #3合模气缸缩回位
5.13 BOOL  ; #3合模气缸伸出位
5.14 BOOL  ; #4合模气缸缩回位
5.15 BOOL  ; #4合模气缸伸出位
60.00 BOOL  ; 腔体在初始位
60.01 BOOL  ; 腔体#1 & #2在初始位
60.02 BOOL  ; 腔体#3 & #4在初始位
61.10 BOOL  ; #1 & #2 腔体感应器异常
61.11 BOOL  ; #1 & #2 腔体出错
62.10 BOOL  ; #3 & #4 腔体感应器异常
62.11 BOOL  ; #3 & #4 腔体出错
65.00 BOOL  ; 腔体机构 出错
6.00 BOOL  ; #1腔体有料感应（常闭）
6.01 BOOL  ; #2腔体有料感应（常闭）
6.02 BOOL  ; #1总氦检气缸缩回位
6.03 BOOL  ; #1总氦检气缸伸出位
6.04 BOOL  ; #2总氦检气缸缩回位
6.05 BOOL  ; #2总氦检气缸伸出位
6.06 BOOL  ; #1氦检气缸原位
6.07 BOOL  ; #1氦检气缸伸出位
6.08 BOOL  ; #2氦检气缸原位
6.09 BOOL  ; #2氦检气缸伸出位
6.10 BOOL  ; #3氦检气缸原位
6.11 BOOL  ; #3氦检气缸伸出位
6.12 BOOL  ; #4氦检气缸原位
6.13 BOOL  ; #4氦检气缸伸出位
6.14 BOOL  ; 出料水平伺服准备就绪
6.15 BOOL  ; 出料水平伺服报警
70.00 BOOL  ; 出料机构初始位
70.05 BOOL  ; 蜂鸣器关
75.00 BOOL  ; 出料机构 出错
7.00 BOOL  ; 出料升降伺服准备就绪
7.01 BOOL  ; 出料升降伺服报警
7.02 BOOL  ; 出料升降伺服柔性报警
7.03 BOOL  ; 出料旋转伺服准备
7.04 BOOL  ; 出料旋转伺服报警
7.05 BOOL  ; 出料移栽伸缩气缸缩回位
7.06 BOOL  ; 出料移栽伸缩气缸伸出位
7.07 BOOL  ; 检测NG缓存推料气缸缩回位
7.08 BOOL  ; 检测NG缓存推料气缸伸出位
7.09 BOOL  ; 出料#1夹爪张开位
7.10 BOOL  ; 出料#1夹爪夹紧位
7.11 BOOL  ; 出料#2夹爪张开位
7.12 BOOL  ; 出料#2夹爪夹紧位
7.13 BOOL  ; 备用
7.14 BOOL  ; 备用
7.15 BOOL  ; 备用
8.00 BOOL  ; 备用
8.01 BOOL  ; 出料移栽放料位有料感应（无料=1）
8.02 BOOL  ; 检测NG缓存放料位有料感应（常闭）
8.03 BOOL  ; 检测NG缓存#1有料感应
8.04 BOOL  ; 检测NG缓存#2有料感应
8.05 BOOL  ; 检测NG缓存#3有料感应
8.06 BOOL  ; 检测NG缓存#4有料感应
8.07 BOOL  ; 备用
8.08 BOOL  ; 备用
8.09 BOOL  ; 备用
8.10 BOOL  ; 备用
8.11 BOOL  ; 备用
8.12 BOOL  ; 上工站信号
8.13 BOOL  ; 下工站信号
8.14 BOOL  ; 气源压力信号
8.15 BOOL  ; 氦检仪报警信号
9.00 BOOL  ; 备用
9.01 BOOL  ; 备用
9.02 BOOL  ; 备用
9.03 BOOL  ; 备用
9.04 BOOL  ; 启动按钮信号
9.05 BOOL  ; 停止按钮信号
9.06 BOOL  ; 复位按钮信号
9.07 BOOL  ; 急停按钮信号
9.08 BOOL  ; 前门门禁信号
9.09 BOOL  ; 后门门禁信号
9.10 BOOL  ; 左门门禁信号
9.11 BOOL  ; 右门门禁信号
9.12 BOOL  ; 手/自动切换
9.13 BOOL  ; 备用
9.14 BOOL  ; 备用
9.15 BOOL  ; 备用
A202.01 BOOL  ; 通信端口1允许标志
A202.02 BOOL  ; 通讯端口2允许
A202.03 BOOL  ; 通讯端口3允许
A276 CHANNEL  ; 进料水平伺服当前脉冲
A278 CHANNEL  ; 出料水平伺服当前脉冲
A280.04 BOOL  ; 进料水平伺服脉冲输出中
A280.05 BOOL  ; 进料水平伺服无原点标志
A281.04 BOOL  ; 出料水平伺服脉冲输出中
A281.05 BOOL  ; 出料水平伺服无原点标志
A322 CHANNEL  ; 腔体上料伺服位置脉冲
A324 CHANNEL  ; 下料水平伺服位置脉冲
A326.04 BOOL  ; 上料水平伺服脉冲输出中
A326.05 BOOL  ; 上料水平伺服无原点
A327.04 BOOL  ; 下料水平伺服脉冲输出中
A327.05 BOOL  ; 下料水平伺服无原点标志
A540.08 BOOL  ; 进料水平伺服CW
A540.09 BOOL  ; 进料水平伺服CCW
A541.08 BOOL  ; 出料水平伺服正极限
A541.09 BOOL  ; 出料水平伺服负极限
A542.08 BOOL  ; 上料水平伺服正极限
A542.09 BOOL  ; 上料水平伺服负极限
A543.08 BOOL  ; 下料水平伺服正极限
A543.09 BOOL  ; 下料水平伺服负极限
C0001 BOOL  ; 1#位重复扫码次数
C0002 BOOL  ; 2#位重复扫码次数
C0011 BOOL  ; #1、#2复检前抽气次数设定值
C0012 BOOL  ; #1、#2清氦次数
C0021 BOOL  ; #3、#4复检前抽气次数设定值
C0022 BOOL  ; #3、#4清氦次数
D0.00 BOOL  ; 紧急停止
D0.01 BOOL  ; 自动运行启动
D0.01 BOOL  ; 自动中
D0.02 BOOL  ; 自动停止
D0.02 BOOL  ; 启动/停止
D0.04 BOOL  ; 报警清除&错误复位
D0.05 BOOL  ; 整机复位启动
D0.10 BOOL  ; 机台有故障
D0.12 BOOL  ; 自动运行启动条件
D10 CHANNEL  ; 进料水平伺服自动速度   HMI
D100 CHANNEL  ; 进料水平伺服上料位参数设定 (M)
D1000 CHANNEL  ; 扫码左阻挡缩回屏蔽延时设定  HMI
D10000 CHANNEL  ; 下料1#夹爪腔体真空实际值
D10002 CHANNEL  ; 下料1#夹爪腔体抽气时间
D10004 CHANNEL  ; 下料2#夹爪腔体真空值
D10006 CHANNEL  ; 下料2#夹爪腔体抽气时间
D10008 CHANNEL  ; 下料夹爪3#腔体真空值
D1001 CHANNEL  ; 扫码左阻挡伸出屏蔽延时  HMI
D10010 CHANNEL  ; 下料夹爪3#腔体抽气时间
D10012 CHANNEL  ; 下料夹爪4#腔体真空值
D10014 CHANNEL  ; 下料夹爪4#腔体抽气时间
D10016 CHANNEL  ; 出料移栽1#腔体真空值
D10018 CHANNEL  ; 出料移栽1#腔体抽气时间
D1002 CHANNEL  ; 扫码右阻挡缩回屏蔽延时  HMI
D10020 CHANNEL  ; 出料移栽2#腔体真空值
D10022 CHANNEL  ; 出料移栽2#腔体抽真空时间
D10024 CHANNEL  ; 出料移栽3#腔体真空值
D10026 CHANNEL  ; 出料移栽3#腔体抽真空时间
D10028 CHANNEL  ; 出料移栽4#腔体真空值
D1003 CHANNEL  ; 扫码右阻挡伸出屏蔽延时  HMI
D10030 CHANNEL  ; 出料移栽4#腔体抽气时间
D1004 CHANNEL  ; 左隔离气缸缩回屏蔽延时  HMI
D1005 CHANNEL  ; 左隔离气缸伸出屏蔽延时  HMI
D1006 CHANNEL  ; 右隔离气缸缩回屏蔽延时  HMI
D1007 CHANNEL  ; 右隔离伸出屏蔽延时  HMI
D1008 CHANNEL  ; 扫码缓存推料气缸缩回屏蔽延时  HMI
D1009 CHANNEL  ; 扫码缓存推料气缸伸出屏蔽延时  HMI
D100 CHANNEL  ; 进料水平伺服上料位置脉冲
D1010 CHANNEL  ; 进料移栽伸缩气缸缩回屏蔽延时  HMI
D1011 CHANNEL  ; 进料移栽伸缩气缸伸出屏蔽延时  HMI
D1012 CHANNEL  ; 进料#1夹爪张开位屏蔽延时  HMI
D1013 CHANNEL  ; 进料#1夹爪夹紧屏蔽延时  HMI
D1014 CHANNEL  ; 进料#2夹爪张开屏蔽延时  HMI
D1015 CHANNEL  ; 进料#2夹爪夹紧屏蔽延时  HMI
D1016 CHANNEL  ; 上料提升气缸上升屏蔽延时  HMI
D1017 CHANNEL  ; 上料提升气缸下降屏蔽延时  HMI
D1018 CHANNEL  ; 上料#1夹爪张开屏蔽延时  HMI
D1019 CHANNEL  ; 上料#1夹爪夹紧屏蔽延时  HMI
D102 CHANNEL  ; 进料水平伺服左爪OK配对位参数设定 (M)
D1020 CHANNEL  ; 上料#2夹爪张开屏蔽延时  HMI
D1021 CHANNEL  ; 上料#2夹爪夹紧屏蔽延时时间  HMI
D1022 CHANNEL  ; 上料#3夹爪张开屏蔽延时  HMI
D1023 CHANNEL  ; 上料#3夹爪夹紧屏蔽延时  HMI
D1024 CHANNEL  ; 上料#4夹爪张开屏蔽延时  HMI
D1025 CHANNEL  ; 上料#4夹爪夹紧屏蔽延时  HMI
D1026 CHANNEL  ; 下料提升气缸上升屏蔽延时  HMI
D1027 CHANNEL  ; 下料提升气缸下降屏蔽延时  HMI
D1028 CHANNEL  ; 下料#1夹爪张开屏蔽延时  HMI
D1029 CHANNEL  ; 下料#1夹爪夹紧屏蔽延时  HMI
D1030 CHANNEL  ; 下料#2夹爪张开屏蔽延时  HMI
D1031 CHANNEL  ; 下料#2夹爪夹紧屏蔽延时  HMI
D1032 CHANNEL  ; 下料#3夹爪张开屏蔽延时  HMI
D1032.00 BOOL  ; 100-1St 上料平移X轴1#伺服归零脉冲(M)
D1033 CHANNEL  ; 下料#3夹爪夹紧屏蔽延时  HMI
D1034 CHANNEL  ; 下料#4夹爪张开屏蔽延时  HMI
D1035 CHANNEL  ; 下料#4夹爪夹紧屏蔽延时  HMI
D1036 CHANNEL  ; #1合模气缸缩回屏蔽延时  HMI
D1037 CHANNEL  ; #1合模气缸伸出屏蔽延时  HMI
D1038 CHANNEL  ; #2合模气缸缩回屏蔽延时  HMI
D1039 CHANNEL  ; #2合模气缸伸出屏蔽延时  HMI
D104 CHANNEL  ; 进料水平伺服右爪OK配对位参数设定 (M)
D1040 CHANNEL  ; #3合模气缸缩回屏蔽延时  HMI
D1041 CHANNEL  ; #3合模气缸伸出屏蔽延时  HMI
D1042 CHANNEL  ; #4合模气缸缩回屏蔽延时  HMI
D1043 CHANNEL  ; #4合模气缸伸出屏蔽延时  HMI
D1044 CHANNEL  ; #1总氦检阀关闭屏蔽延时  HMI
D1045 CHANNEL  ; #1总氦检阀打开屏蔽延时  HMI
D1046 CHANNEL  ; #2总氦检阀关闭屏蔽延时  HMI
D1047 CHANNEL  ; #2总氦检阀打开屏蔽延时  HMI
D1048 CHANNEL  ; #1氦检阀关闭屏蔽延时  HMI
D1049 CHANNEL  ; #1氦检阀打开屏蔽延时  HMI
D1050 CHANNEL  ; #2氦检阀关闭屏蔽延时  HMI
D1051 CHANNEL  ; #2氦检阀打开屏蔽延时  HMI
D1052 CHANNEL  ; #3氦检阀关闭屏蔽延时  HMI
D1053 CHANNEL  ; #3氦检阀打开屏蔽延时  HMI
D1054 CHANNEL  ; #4氦检阀关闭屏蔽延时  HMI
D1055 CHANNEL  ; #4氦检阀打开屏蔽延时  HMI
D1056 CHANNEL  ; 出料移栽伸缩气缸缩回屏蔽延时  HMI
D1057 CHANNEL  ; 出料移栽伸缩气缸伸出屏蔽延时  HMI
D1058 CHANNEL  ; 检测NG推料气缸缩回屏蔽延时  HMI
D1059 CHANNEL  ; 检测NG推料气缸伸出屏蔽延时  HMI
D106 CHANNEL  ; 进料水平伺服左爪缓存位参数设定 (M)
D1060 CHANNEL  ; 出料#1夹爪张开屏蔽延时  HMI
D1061 CHANNEL  ; 出料#1夹爪夹紧屏蔽延时  HMI
D1062 CHANNEL  ; 出料#2夹爪张开屏蔽延时  HMI
D1063 CHANNEL  ; 出料#2夹爪夹紧屏蔽延时  HMI
D106 CHANNEL  ; 进料水平伺服右爪OK配对位参数设定 (M)
D108 CHANNEL  ; 进料水平伺服右爪缓存位参数设定 (M)
D110 CHANNEL  ; 进料水平伺服NG位参数设定 (M)
D1100 CHANNEL  ; 扫码左阻挡缩回延时时间
D1101 CHANNEL  ; 扫码左阻挡伸出延时时间
D1102 CHANNEL  ; 扫码右阻挡缩回延时时间
D1103 CHANNEL  ; 扫码右阻挡伸出延时时间
D1104 CHANNEL  ; 左隔离气缸缩回延时时间
D1105 CHANNEL  ; 左隔离气缸伸出延时时间
D1106 CHANNEL  ; 右隔离气缸缩回延时时间
D1107 CHANNEL  ; 右隔离气缸伸出延时时间
D1108 CHANNEL  ; 扫码缓存推料气缸缩回延时时间
D1109 CHANNEL  ; 扫码缓存气缸伸出延时时间
D110 CHANNEL  ; 进料水平伺服左爪缓存位参数设定 (M)
D1110 CHANNEL  ; 进料移栽伸缩气缸缩回延时时间
D1111 CHANNEL  ; 进料移栽伸缩气缸伸出延时时间
D1112 CHANNEL  ; 进料#1夹爪张开位延时时间
D1113 CHANNEL  ; 进料#1夹爪夹紧延时时间
D1114 CHANNEL  ; 进料#2夹爪张开延时时间
D1115 CHANNEL  ; 进料#2夹爪夹紧延时时间
D1116 CHANNEL  ; 上料提升气缸上升延时时间
D1117 CHANNEL  ; 上料提升气缸下降延时时间
D1118 CHANNEL  ; 上料#1夹爪张开延时时间
D1119 CHANNEL  ; 上料#1夹爪夹紧延时时间
D1120 CHANNEL  ; 上料#2夹爪张开延时时间
D1121 CHANNEL  ; 上料#2夹爪夹紧延时时间
D1122 CHANNEL  ; 上料#3夹爪张开延时时间
D1123 CHANNEL  ; 上料#3夹爪夹紧延时时间
D1124 CHANNEL  ; 上料#4夹爪张开延时时间
D1125 CHANNEL  ; 上料#4夹爪夹紧延时时间
D1126 CHANNEL  ; 下料提升气缸上升延时时间
D1127 CHANNEL  ; 下料提升气缸下降延时时间
D1128 CHANNEL  ; 下料#1夹爪张开延时时间
D1129 CHANNEL  ; 下料#1夹爪夹紧延时时间
D1130 CHANNEL  ; 下料#2夹爪张开延时时间
D1131 CHANNEL  ; 下料#2夹爪夹紧延时时间
D1132 CHANNEL  ; 下料#3夹爪张开延时时间
D1133 CHANNEL  ; 下料#3夹爪夹紧延时时间
D1134 CHANNEL  ; 下料#4夹爪张开延时时间
D1135 CHANNEL  ; 下料#4夹爪夹紧延时时间
D1136 CHANNEL  ; #1合模气缸缩回延时时间
D1137 CHANNEL  ; #1合模气缸伸出延时时间
D1138 CHANNEL  ; #2合模气缸缩回延时时间
D1139 CHANNEL  ; #2合模气缸伸出延时时间
D114 CHANNEL  ; 进料水平伺服右爪缓存位参数设定 (M)
D1140 CHANNEL  ; #3合模气缸缩回延时时间
D1141 CHANNEL  ; #3合模气缸伸出延时时间
D1142 CHANNEL  ; #4合模气缸缩回延时时间
D1143 CHANNEL  ; #4合模气缸伸出延时时间
D1144 CHANNEL  ; #1总氦检阀关闭延时时间
D1145 CHANNEL  ; #1总氦检阀打开延时时间
D1146 CHANNEL  ; #2总氦检阀关闭延时时间
D1147 CHANNEL  ; #2总氦检阀打开延时时间
D1148 CHANNEL  ; #1氦检阀关闭延时时间
D1149 CHANNEL  ; #1氦检阀打开延时时间
D1150 CHANNEL  ; #2氦检阀关闭延时时间
D1151 CHANNEL  ; #2氦检阀打开延时时间
D1152 CHANNEL  ; #3氦检阀关闭延时时间
D1153 CHANNEL  ; #3氦检阀打开延时时间
D1154 CHANNEL  ; #4氦检阀关闭延时时间
D1155 CHANNEL  ; #4氦检阀打开延时时间
D1156 CHANNEL  ; 出料移栽伸缩气缸缩回延时时间
D1157 CHANNEL  ; 出料移栽伸缩气缸伸出延时时间
D1158 CHANNEL  ; 检测NG推料气缸缩回延时时间
D1159 CHANNEL  ; 检测NG推料气缸伸出延时时间
D1160 CHANNEL  ; 出料#1夹爪张开延时时间
D1161 CHANNEL  ; 出料#1夹爪夹紧延时时间
D1162 CHANNEL  ; 出料#2夹爪张开延时时间
D1163 CHANNEL  ; 出料#2夹爪夹紧延时时间
D118 CHANNEL  ; 进料水平伺服放料位参数设定 (M)
D118 CHANNEL  ; 进料水平伺服缓存位参数设定 (M)
D1199 CHANNEL  ; 传感器延时
D12 CHANNEL  ; 进料水平伺服手动速度   HMI
D122 CHANNEL  ; 进料水平伺服放料位参数设定 (M)
D124 CHANNEL  ; 进料升降伺服缓存位参数设定
D126 CHANNEL  ; 进料升降伺服放料位参数设定
D128 CHANNEL  ; 进料升降伺服待料位参数设定
D130 CHANNEL  ; 进料旋转伺服#1待料位参数设定
D132 CHANNEL  ; 进料旋转伺服#2待料位参数设定
D134 CHANNEL  ; 进料旋转伺服上料位参数设定
D136 CHANNEL  ; 上料水平伺服待料位参数设定 (M)
D138 CHANNEL  ; 上料水平伺服#1腔体位参数设定 (M)
D14 CHANNEL  ; 进料升降伺服自动速度   HMI
D140 CHANNEL  ; 上料水平伺服#2腔体位参数设定 (M)
D142 CHANNEL  ; 下料水平伺服#1腔体位参数设定 (M)
D144 CHANNEL  ; 下料水平伺服#2腔体位参数设定 (M)
D146 CHANNEL  ; 下料水平伺服放料位参数设定 (M)
D148 CHANNEL  ; 出料水平伺服取料位参数设定 (M)
D150 CHANNEL  ; 出料水平伺服#1NG缓存位参数设定 (M)
D1501.03 BOOL  ; Inital_Cmd_Pls
D152 CHANNEL  ; 出料水平伺服#2NG缓存位参数设定 (M)
D154 CHANNEL  ; 出料放料待机位参数设定 (M)
D158 CHANNEL  ; 出料水平伺服放料位参数设定 (M)
D16 CHANNEL  ; 进料升降伺服手动速度   HMI
D160 CHANNEL  ; 出料升降伺服待料位参数设定
D162 CHANNEL  ; 出料升降伺服取料位参数设定
D164 CHANNEL  ; 出料升降伺服放料位参数设定
D166 CHANNEL  ; 出料旋转伺服#1出料位参数设定
D168 CHANNEL  ; 出料旋转伺服#2出料位参数设定
D170 CHANNEL  ; 出料旋转伺服待料位参数设定
D174 CHANNEL  ; 升降伺服上料位
D176 CHANNEL  ; 出料升降伺服NG缓存位参数设定
D18 CHANNEL  ; 进料旋转伺服自动速度   HMI
D1.00 BOOL  ; 整机复位开始
D1.01 BOOL  ; 整机复位开始延时
D1.10 BOOL  ; 整机在初始位
D20 CHANNEL  ; 进料旋转伺服手动速度   HMI
D200 CHANNEL  ; 进料水平伺服上料位置浮点数
D20124 CHANNEL  ; 进料升降伺服定位位置
D20126 CHANNEL  ; 进料升降伺服运行速度
D20128 CHANNEL  ; 进料升降伺服加速时间
D20130 CHANNEL  ; 进料升降伺服减速时间
D20136 CHANNEL  ; 进料移栽伺服位置
D20138 CHANNEL  ; 进料移栽伺服运行速度
D20140 CHANNEL  ; 进料移栽伺服加速时间
D20142 CHANNEL  ; 进料移栽伺服减速时间
D20148 CHANNEL  ; 出料升降定位位置
D20150 CHANNEL  ; 出料升降伺服运行速度
D20152 CHANNEL  ; 出料升降伺服加速时间
D20154 CHANNEL  ; 出料升降伺服减速时间
D20160 CHANNEL  ; 出料移栽定位位置
D20162 CHANNEL  ; 出料移栽伺服运行速度
D20164 CHANNEL  ; 出料移栽伺服加速时间
D20166 CHANNEL  ; 出料移栽伺服减速时间
D20172 CHANNEL  ; 进料升降伺服当前位置
D20176 CHANNEL  ; 进料移栽伺服当前位置
D20180 CHANNEL  ; 出料升降伺服当前位置
D20184 CHANNEL  ; 出料移栽伺服当前位置
D20236 CHANNEL  ; 进料移栽伺服位置
D20300 CHANNEL  ; #1至#2模拟量使用设置
D20301 CHANNEL  ; #1至#2模拟量输入范围为0-10V
D20318 CHANNEL  ; #1至#2的模拟量输入分辨率为8000   普通模式
D204 CHANNEL  ; 进料水平伺服左爪OK配对位置浮点数
D208 CHANNEL  ; 进料水平伺服右爪OK配对位置浮点数
D212 CHANNEL  ; 进料水平伺服左爪缓存位置浮点数
D216 CHANNEL  ; 进料水平伺服右爪缓存位置浮点数
D22 CHANNEL  ; 上料水平伺服自动速度   HMI
D220 CHANNEL  ; 进料水平伺服缓存位置浮点数
D224 CHANNEL  ; 进料水平伺服放料位置浮点数
D228 CHANNEL  ; 进料升降伺服上料位置浮点数
D230 CHANNEL  ; 进料升降伺服放料位置浮点数
D232 CHANNEL  ; 进料升降伺服待料位置浮点数
D234 CHANNEL  ; 进料移栽伺服#1待料位置浮点数
D236 CHANNEL  ; 进料移栽伺服#2待料位置浮点数
D238 CHANNEL  ; 进料移栽伺服上料位置浮点数
D24 CHANNEL  ; 上料水平伺服手动速度   HMI
D240 CHANNEL  ; 上料水平伺服待料位置浮点数
D244 CHANNEL  ; 上料水平伺服#1腔体位置浮点数
D248 CHANNEL  ; 上料水平伺服#2腔体位置浮点数
D2500 CHANNEL  ; 检漏口压力设定值
D2502 CHANNEL  ; 检漏口压力底数转换
D2504 CHANNEL  ; 漏率设定值
D2506 CHANNEL  ; 泄漏率底数转换
D2510 CHANNEL  ; #1 &#2腔体检漏口压力浮点数
D2512 CHANNEL  ; #1 &#2腔体漏率浮点数
D2514 CHANNEL  ; #1 &#2腔体测试检漏口压力
D2516 CHANNEL  ; #1 &#2腔体测试漏率
D252 CHANNEL  ; 下料水平伺服#1腔体位置浮点数
D2520 CHANNEL  ; #3 &#4腔体检漏口压力浮点数
D2522 CHANNEL  ; #3 &#4腔体漏率浮点数
D2524 CHANNEL  ; #3 &#4腔体测试检漏口压力
D2526 CHANNEL  ; #3 &#4腔体测试漏率
D256 CHANNEL  ; 下料水平伺服#2腔体位置浮点数
D26 CHANNEL  ; 下料水平伺服自动速度   HMI
D260 CHANNEL  ; 下料水平伺服待料位置浮点数
D264 CHANNEL  ; 出料水平伺服取料位置浮点数
D268 CHANNEL  ; 出料水平伺服#1缓存位置浮点数
D272 CHANNEL  ; 出料水平伺服#2缓存位置浮点数
D276 CHANNEL  ; 出料水平伺服放料位置浮点数
D28 CHANNEL  ; 下料水平伺服手动速度   HMI
D280 CHANNEL  ; 出料升降伺服待料位置浮点数
D282 CHANNEL  ; 出料升降伺服上料位置浮点数
D284 CHANNEL  ; 出料升降伺服放料位置浮点数
D286 CHANNEL  ; 出料移栽伺服#1出料位置浮点数
D288 CHANNEL  ; 出料移栽伺服#2出料位置浮点数
D290 CHANNEL  ; 出料移栽伺服待料位置浮点数
D30 CHANNEL  ; 出料水平伺服自动速度   HMI
D3000 CHANNEL  ; 真空阀值到达
D3002 CHANNEL  ; 抽真空时间（SP）
D3004 CHANNEL  ; 抽残气压力（SP）
D3006 CHANNEL  ; 氦检时间（SP）
D3008 CHANNEL  ; 破真空阀值（SP）
D3010 CHANNEL  ; 氦检仪稳定时间（SP）
D3011 CHANNEL  ; 氦检仪状态 0-未启用 1-未启动  2-稳定中 3-已稳定 4-内部校准中 5-校准完成 6-校准出错
D3012 CHANNEL  ; 检漏口压力指数（SP）
D3014 CHANNEL  ; 检漏口压力底数（SP）
D3016 CHANNEL  ; 泄漏率指数（SP）
D3018 CHANNEL  ; 泄漏率底数（SP）
D301.10 BOOL  ; 出料升降至取料位条件
D301.11 BOOL  ; 出料升降至NG放料位条件
D3020 CHANNEL  ; 自检真空到达阀值（SP）
D3022 CHANNEL  ; 自检抽真空时间（SP）
D3024 CHANNEL  ; 自检泄漏量（SP）
D3026 CHANNEL  ; 自检保压前延时（SP）
D3028 CHANNEL  ; 自检保压时间（SP）
D3032 CHANNEL  ; 氦检关真空延时（SP）
D3034 CHANNEL  ; #1腔体自检保压前真空值
D3036 CHANNEL  ; #1腔体自检保压后真空值
D3038 CHANNEL  ; #1腔体自检泄漏量
D3040 CHANNEL  ; #1腔体自检抽真空时间（PV）
D3042 CHANNEL  ; #1腔体自检保压前时间（PV）
D3044 CHANNEL  ; #1腔体自检保压时间（PV)
D3046 CHANNEL  ; #1腔体自检结果  0-未进行  1-自检中  2-自检OK  3-自检泄漏  4-自检抽真空NG
D3048 CHANNEL  ; #2腔体自检保压前真空值
D3050 CHANNEL  ; #2腔体自检保压后真空值
D3052 CHANNEL  ; #2腔体自检泄漏量
D3054 CHANNEL  ; #2腔体自检抽真空时间（PV）
D3056 CHANNEL  ; #2腔体自检保压前时间（PV）
D3058 CHANNEL  ; #2腔体自检保压时间（PV)
D3060 CHANNEL  ; #2腔体自检结果
D3062 CHANNEL  ; #3腔体自检保压前真空值
D3064 CHANNEL  ; #3腔体自检保压后真空值
D3066 CHANNEL  ; #3腔体自检泄漏量
D3068 CHANNEL  ; #3腔体自检抽真空时间（PV）
D3070 CHANNEL  ; #3腔体自检保压前时间（PV）
D3072 CHANNEL  ; #3腔体自检保压时间（PV)
D3074 CHANNEL  ; #3腔体自检结果  0-未进行  1-自检中  2-自检OK  3-自检泄漏  4-自检抽真空NG
D3076 CHANNEL  ; #4腔体自检保压前真空值
D3078 CHANNEL  ; #4腔体自检保压后真空值
D3080 CHANNEL  ; #4腔体自检泄漏量
D3082 CHANNEL  ; #4腔体自检抽真空时间（PV）
D3084 CHANNEL  ; #4腔体自检保压前时间（PV）
D3086 CHANNEL  ; #4腔体自检保压时间（PV)
D3088 CHANNEL  ; #4腔体自检结果  0-未进行  1-自检中  2-自检OK  3-自检泄漏  4-自检抽真空NG
D3090 CHANNEL  ; #5腔体自检保压前真空值
D3092 CHANNEL  ; #5腔体自检保压后真空值
D3094 CHANNEL  ; #5腔体自检泄漏量
D3096 CHANNEL  ; #5腔体自检抽真空时间（PV）
D3098 CHANNEL  ; #5腔体自检保压前时间（PV）
D3100 CHANNEL  ; #5腔体自检保压时间（PV)
D3102 CHANNEL  ; #5腔体自检结果  0-未进行  1-自检中  2-自检OK  3-自检泄漏  4-自检抽真空NG
D3104 CHANNEL  ; #6腔体自检保压前真空值
D3106 CHANNEL  ; #6腔体自检保压后真空值
D3108 CHANNEL  ; #6腔体自检泄漏量
D3110 CHANNEL  ; #6腔体自检抽真空时间（PV）
D3112 CHANNEL  ; #6腔体自检保压前时间（PV）
D3114 CHANNEL  ; #6腔体自检保压时间（PV)
D3116 CHANNEL  ; #6腔体自检结果  0-未进行  1-自检中  2-自检OK  3-自检泄漏  4-自检抽真空NG
D3118 CHANNEL  ; #7腔体自检保压前真空值
D3120 CHANNEL  ; #7腔体自检保压后真空值
D3122 CHANNEL  ; #7腔体自检泄漏量
D3124 CHANNEL  ; #7腔体自检抽真空时间（PV）
D3126 CHANNEL  ; #7腔体自检保压前时间（PV）
D3128 CHANNEL  ; #7腔体自检保压时间（PV)
D3130 CHANNEL  ; #7腔体自检结果  0-未进行  1-自检中  2-自检OK  3-自检泄漏  4-自检抽真空NG
D3132 CHANNEL  ; #8腔体自检保压前真空值
D3134 CHANNEL  ; #8腔体自检保压后真空值
D3136 CHANNEL  ; #8腔体自检泄漏量
D3138 CHANNEL  ; #8腔体自检抽真空时间（PV）
D3140 CHANNEL  ; #8腔体自检保压前时间（PV）
D3142 CHANNEL  ; #8腔体自检保压时间（PV)
D3144 CHANNEL  ; #8腔体自检结果  0-未进行  1-自检中  2-自检OK  3-自检泄漏  4-自检抽真空NG
D3150 CHANNEL  ; 腔体#1测试结果 1-OK  2-NG  3-腔体泄漏
D3152 CHANNEL  ; 腔体#2测试结果 1-OK  2-NG  3-腔体泄漏
D3154 CHANNEL  ; 腔体#3测试结果 1-OK  2-NG  3-腔体泄漏
D3156 CHANNEL  ; 腔体#4测试结果 1-OK  2-NG  3-腔体泄漏
D3158 CHANNEL  ; 腔体#5测试结果 1-OK  2-NG  3-腔体泄漏
D3160 CHANNEL  ; 腔体#6测试结果 1-OK  2-NG  3-腔体泄漏
D3162 CHANNEL  ; 腔体#7测试结果 1-OK  2-NG  3-腔体泄漏
D3164 CHANNEL  ; 腔体#8测试结果 1-OK  2-NG  3-腔体泄漏
D3166 CHANNEL  ; 下料机械手#1夹爪测试结果 1-OK  2-NG  3-腔体泄漏
D3168 CHANNEL  ; 下料机械手#2夹爪测试结果 1-OK  2-NG  3-腔体泄漏
D3170 CHANNEL  ; 下料机械手#3夹爪测试结果 1-OK  2-NG  3-腔体泄漏
D3172 CHANNEL  ; 下料机械手#4夹爪测试结果 1-OK  2-NG  3-腔体泄漏
D3174 CHANNEL  ; 出料移栽#1料盒测试结果 1-OK  2-NG  3-腔体泄漏
D3176 CHANNEL  ; 出料移栽#2料盒测试结果 1-OK  2-NG  3-腔体泄漏
D3178 CHANNEL  ; 出料移栽#3料盒测试结果 1-OK  2-NG  3-腔体泄漏
D3180 CHANNEL  ; 出料移栽#4料盒测试结果 1-OK  2-NG  3-腔体泄漏
D3186 CHANNEL  ; 腔体#1完成时检漏口压力
D3188 CHANNEL  ; 腔体#1完成时漏率
D3190 CHANNEL  ; 腔体#2完成时检漏口压力
D3192 CHANNEL  ; 腔体#2完成时漏率
D3193 CHANNEL  ; 腔体#2完成时漏率
D3194 CHANNEL  ; 腔体#3完成时检漏口压力
D3196 CHANNEL  ; 腔体#3完成时漏率
D3198 CHANNEL  ; 腔体#4完成时检漏口压力
D32 CHANNEL  ; 出料水平伺服手动速度   HMI
D3200 CHANNEL  ; 腔体#4完成时漏率
D3202 CHANNEL  ; 腔体#3 &#4完成时检漏口压力
D3204 CHANNEL  ; 腔体#3 &#4完成时漏率
D3206 CHANNEL  ; 腔体#6完成时检漏口压力
D3208 CHANNEL  ; 腔体#6完成时漏率
D3210 CHANNEL  ; 腔体#7完成时检漏口压力
D32100 CHANNEL  ; 左扫码NG次数
D32101 CHANNEL  ; 右扫码失败次数
D3212 CHANNEL  ; 腔体#7完成时漏率
D3214 CHANNEL  ; 腔体#8完成时检漏口压力
D3216 CHANNEL  ; 腔体#8完成时漏率
D3218 CHANNEL  ; 下料机械手#1夹爪完成时检漏口压力
D3220 CHANNEL  ; 下料机械手#1夹爪完成时漏率
D32201 CHANNEL  ; 当前扫码OK缓存数量（对）
D3222 CHANNEL  ; 下料机械手#2夹爪完成时检漏口压力
D3224 CHANNEL  ; 下料机械手#2夹爪完成时漏率
D3226 CHANNEL  ; 下料机械手#3夹爪完成时检漏口压力
D3228 CHANNEL  ; 下料机械手#3夹爪完成时漏率
D3230 CHANNEL  ; 下料机械手#4夹爪完成时检漏口压力
D3232 CHANNEL  ; 下料机械手#4夹爪完成时漏率
D3234 CHANNEL  ; 出料移栽料盘#1完成时检漏口压力
D3236 CHANNEL  ; 出料移栽料盘#1完成时漏力
D3238 CHANNEL  ; 出料移栽料盘#2完成时检漏口压力
D3240 CHANNEL  ; 出料移栽料盘#2完成时漏力
D3242 CHANNEL  ; 出料移栽料盘#3完成时检漏口压力
D3244 CHANNEL  ; 出料移栽料盘#3完成时漏力
D3246 CHANNEL  ; 出料移栽料盘#4完成时检漏口压力
D3248 CHANNEL  ; 出料移栽料盘#4完成时漏力
D3258 CHANNEL  ; #1号腔抽气时间
D3259 CHANNEL  ; #2号腔抽气时间
D3260 CHANNEL  ; #3号腔抽气时间
D3261 CHANNEL  ; #4号腔抽气时间
D3262 CHANNEL  ; #5号腔抽气时间
D3263 CHANNEL  ; #6号腔抽气时间
D3264 CHANNEL  ; #7号腔抽气时间
D3265 CHANNEL  ; #8号腔抽气时间
D328 CHANNEL  ; 进料升降伺服上料位置脉冲
D3288 CHANNEL  ; 下料机械手#1夹爪工位标记
D3290 CHANNEL  ; 下料机械手#2夹爪工位标记
D3292 CHANNEL  ; 下料机械手#3夹爪工位标记
D3294 CHANNEL  ; 下料机械手#4夹爪工位标记
D3296 CHANNEL  ; 出料移栽料盘#1工位标记
D3298 CHANNEL  ; 出料移栽料盘#2工位标记
D330 CHANNEL  ; 进料升降伺服放料位置脉冲
D3300 CHANNEL  ; 出料移栽料盘#3工位标记
D3302 CHANNEL  ; 出料移栽料盘#4工位标记
D332 CHANNEL  ; 进料升降伺服待料位置脉冲
D3320 CHANNEL  ; 接收漏率浮点数
D3322 CHANNEL  ; 氦检仪稳定漏率设定值(Float)
D3324 CHANNEL  ; 氦检设定漏率指数
D3328 CHANNEL  ; 氦检设置漏率底数
D334 CHANNEL  ; 进料移栽伺服#1待料位置脉冲
D3340 CHANNEL  ; #1真空值
D3342 CHANNEL  ; #2真空值
D3344 CHANNEL  ; #3真空值
D3346 CHANNEL  ; #4真空值
D3348 CHANNEL  ; 腔体#5实时真空值
D3350 CHANNEL  ; 腔体#1测试完成真空值
D3352 CHANNEL  ; 腔体#2测试完成真空值
D3354 CHANNEL  ; 腔体#3测试完成真空值
D3356 CHANNEL  ; 腔体#4测试完成真空值
D336 CHANNEL  ; 进料移栽伺服#2待料位置脉冲
D338 CHANNEL  ; 进料移栽伺服上料位置脉冲
D34 CHANNEL  ; 出料升降伺服自动速度   HMI
D340 CHANNEL  ; 上料水平伺服待料位置脉冲
D344 CHANNEL  ; 上料水平伺服#1腔体位置脉冲
D348 CHANNEL  ; 上料水平伺服#2腔体位置脉冲
D352 CHANNEL  ; 下料水平伺服#1腔体位置脉冲
D356 CHANNEL  ; 下料水平伺服#2腔体位置脉冲
D3560 CHANNEL  ; #1号腔抽气时间
D3562 CHANNEL  ; #2号腔抽气时间
D3564 CHANNEL  ; #3号腔抽气时间
D3566 CHANNEL  ; #4号腔抽气时间
D36 CHANNEL  ; 出料升降伺服手动速度   HMI
D360 CHANNEL  ; 下料水平伺服待料位置脉冲
D364 CHANNEL  ; 出料水平伺服取料位置脉冲
D368 CHANNEL  ; 出料水平伺服#1缓存位置脉冲
D3700 CHANNEL  ; 报警延时时间
D372 CHANNEL  ; 出料水平伺服#2缓存位置脉冲
D374 CHANNEL  ; 出料放料待机位位置脉冲
D376 CHANNEL  ; 出料水平伺服放料位置脉冲
D38 CHANNEL  ; 出料旋转伺服自动速度   HMI
D380 CHANNEL  ; 出料升降伺服待料位置脉冲
D382 CHANNEL  ; 出料升降伺服取料位置脉冲
D384 CHANNEL  ; 出料升降伺服放料位置脉冲
D386 CHANNEL  ; 出料旋转伺服#1出料位置脉冲
D388 CHANNEL  ; 出料旋转伺服#2出料位置脉冲
D390 CHANNEL  ; 出料旋转伺服待料位置脉冲
D40 CHANNEL  ; 出料旋转伺服手动速度   HMI
D400 CHANNEL  ; 伺服方向脉冲浮点
D4000 CHANNEL  ; 真空值1转存
D4002 CHANNEL  ; #1真空值运算1
D4004 CHANNEL  ; #1真空值运算2
D4006 CHANNEL  ; #1真空值运算3
D4008 CHANNEL  ; #1真空值运算4
D4010 CHANNEL  ; #1真空值
D402 CHANNEL  ; 轴控预留量
D4020 CHANNEL  ; #2真空值转存
D4022 CHANNEL  ; #2真空值运算1
D4024 CHANNEL  ; #2真空值运算2
D4026 CHANNEL  ; #2真空值运算3
D4028 CHANNEL  ; #2真空值运算4
D4030 CHANNEL  ; #3 & #4真空值
D404 CHANNEL  ; 伺服当前脉冲量（浮点数）
D404.04 BOOL  ; 复位[Flag]
D416 CHANNEL  ; 进料水平伺服当前脉冲
D426 CHANNEL  ; 进料升降伺服当前脉冲
D446 CHANNEL  ; 腔体上料伺服当前脉冲
D456 CHANNEL  ; 腔体上料伺服当前脉冲
D466 CHANNEL  ; 腔体下料伺服当前脉冲
D476 CHANNEL  ; 出料升降伺服当前脉冲
D486 CHANNEL  ; 出料升降伺服当前脉冲
D496 CHANNEL  ; 出料旋转伺服当前脉冲
D500 CHANNEL  ; 进料水平伺服自动状态加速比率
D501 CHANNEL  ; 进料水平伺服自动状态减速比率
D502 CHANNEL  ; 进料水平伺服自动状态目标频率（低位）
D503 CHANNEL  ; 进料水平伺服自动状态目标频率（高位）
D504 CHANNEL  ; 进料水平伺服自动状态脉冲输出量（低位）
D505 CHANNEL  ; 进料水平伺服自动状态脉冲输出量（高位）
D506 CHANNEL  ; 进料水平伺服自动状态启动频率（低位）
D507 CHANNEL  ; 进料水平伺服自动状态启动频率（高位）
D508 CHANNEL  ; 进料水平伺服自动状态脉冲  Plus/s
D510 CHANNEL  ; 进料升降伺服自动状态加速比率
D5100 CHANNEL  ; 1#位扫码长度
D5101 CHANNEL  ; #1位条码
D511 CHANNEL  ; 进料升降伺服自动状态减速比率
D512 CHANNEL  ; 进料升降伺服自动状态目标频率（低位）
D5120 CHANNEL  ; #1扫码位电池条码
D513 CHANNEL  ; 进料升降伺服自动状态目标频率（高位）
D514 CHANNEL  ; 进料升降伺服自动状态脉冲输出量（低位）
D515 CHANNEL  ; 进料升降伺服自动状态脉冲输出量（高位）
D516 CHANNEL  ; 进料升降伺服自动状态启动频率（低位）
D517 CHANNEL  ; 进料升降伺服自动状态启动频率（高位）
D518 CHANNEL  ; 进料升降伺服自动状态脉冲  Plus/s
D520 CHANNEL  ; 进料旋转伺服自动状态加速比率
D5200 CHANNEL  ; 2#位扫码长度
D5201 CHANNEL  ; #2位条码
D521 CHANNEL  ; 进料旋转伺服自动状态减速比率
D522 CHANNEL  ; 进料旋转伺服自动状态目标频率（低位）
D523 CHANNEL  ; 进料旋转伺服自动状态目标频率（高位）
D524 CHANNEL  ; 进料旋转伺服自动状态脉冲输出量（低位）
D5240 CHANNEL  ; #2扫码位电池条码
D525 CHANNEL  ; 进料旋转伺服自动状态脉冲输出量（高位）
D526 CHANNEL  ; 进料旋转伺服自动状态启动频率（低位）
D527 CHANNEL  ; 进料旋转伺服自动状态启动频率（高位）
D528 CHANNEL  ; 进料旋转伺服自动状态脉冲  Plus/s
D52.00 BOOL  ; 清零良品
D52.01 BOOL  ; 清零NG
D52.02 BOOL  ; 清零总数
D530 CHANNEL  ; 上料水平伺服自动状态加速比率
D531 CHANNEL  ; 上料水平伺服自动状态减速比率
D532 CHANNEL  ; 上料水平伺服自动状态目标频率（低位）
D533 CHANNEL  ; 上料水平伺服自动状态目标频率（高位）
D534 CHANNEL  ; 上料水平伺服自动状态脉冲输出量（低位）
D535 CHANNEL  ; 上料水平伺服自动状态脉冲输出量（高位）
D536 CHANNEL  ; 上料水平伺服自动状态启动频率（低位）
D537 CHANNEL  ; 上料水平伺服自动状态启动频率（高位）
D538 CHANNEL  ; 上料水平伺服自动状态脉冲  Plus/s
D540 CHANNEL  ; 下料水平伺服自动状态加速比率
D541 CHANNEL  ; 下料水平伺服自动状态减速比率
D542 CHANNEL  ; 下料水平伺服自动状态目标频率（低位）
D543 CHANNEL  ; 下料水平伺服自动状态目标频率（高位）
D544 CHANNEL  ; 下料水平伺服自动状态脉冲输出量（低位）
D545 CHANNEL  ; 下料水平伺服自动状态脉冲输出量（高位）
D546 CHANNEL  ; 下料水平伺服自动状态启动频率（低位）
D547 CHANNEL  ; 下料水平伺服自动状态启动频率（高位）
D548 CHANNEL  ; 下料水平伺服自动状态脉冲  Plus/s
D550 CHANNEL  ; 出料水平伺服自动状态加速比率
D551 CHANNEL  ; 出料水平伺服自动状态减速比率
D552 CHANNEL  ; 出料水平伺服自动状态目标频率（低位）
D553 CHANNEL  ; 出料水平伺服自动状态目标频率（高位）
D554 CHANNEL  ; 出料水平伺服自动状态脉冲输出量（低位）
D555 CHANNEL  ; 出料水平伺服自动状态脉冲输出量（高位）
D556 CHANNEL  ; 出料水平伺服自动状态启动频率（低位）
D557 CHANNEL  ; 出料水平伺服自动状态启动频率（高位）
D558 CHANNEL  ; 出料水平伺服自动状态脉冲  Plus/s
D560 CHANNEL  ; 出料升降伺服自动状态加速比率
D561 CHANNEL  ; 出料升降伺服自动状态减速比率
D562 CHANNEL  ; 出料升降伺服自动状态目标频率（低位）
D563 CHANNEL  ; 出料升降伺服自动状态目标频率（高位）
D564 CHANNEL  ; 出料升降伺服自动状态脉冲输出量（低位）
D565 CHANNEL  ; 出料升降伺服自动状态脉冲输出量（高位）
D566 CHANNEL  ; 出料升降伺服自动状态启动频率（低位）
D567 CHANNEL  ; 出料升降伺服自动状态启动频率（高位）
D568 CHANNEL  ; 出料升降伺服自动状态脉冲  Plus/s
D570 CHANNEL  ; 出料旋转伺服自动状态加速比率
D571 CHANNEL  ; 出料旋转伺服自动状态减速比率
D572 CHANNEL  ; 出料旋转伺服自动状态目标频率（低位）
D573 CHANNEL  ; 出料旋转伺服自动状态目标频率（高位）
D574 CHANNEL  ; 出料旋转伺服自动状态脉冲输出量（低位）
D575 CHANNEL  ; 出料旋转伺服自动状态脉冲输出量（高位）
D576 CHANNEL  ; 出料旋转伺服自动状态启动频率（低位）
D577 CHANNEL  ; 出料旋转伺服自动状态启动频率（高位）
D578 CHANNEL  ; 出料旋转伺服自动状态脉冲  Plus/s
D5920 CHANNEL  ; 缓存位条码
D600 CHANNEL  ; 进料水平伺服手动状态加速比率
D6000 CHANNEL  ; #1扫码位位电池条码
D601 CHANNEL  ; 进料水平伺服手动状态减速比率
D602 CHANNEL  ; 进料水平伺服手动状态目标频率（低位）
D6020 CHANNEL  ; #1扫码位电池条码
D6020 CHANNEL  ; #1上料位电池条码
D603 CHANNEL  ; 进料水平伺服手动状态目标频率（高位）
D604 CHANNEL  ; 进料水平伺服手动状态脉冲输出量（低位）
D6040 CHANNEL  ; #2上料位电池条码
D605 CHANNEL  ; 进料水平伺服手动状态脉冲输出量（高位）
D606 CHANNEL  ; 进料水平伺服手动状态启动频率（低位）
D607 CHANNEL  ; 进料水平伺服手动状态启动频率（高位）
D608 CHANNEL  ; 进料水平伺服手动状态脉冲  Plus/s
D6080 CHANNEL  ; 进料机械手#1夹爪电池条码
D610 CHANNEL  ; 进料升降伺服手动状态加速比率
D6100 CHANNEL  ; 进料机械手_腔体真空设定值
D6102 CHANNEL  ; 进料机械手_漏率设定值
D6104 CHANNEL  ; 进料机械手_检漏口压力设定值
D6106 CHANNEL  ; 进料机械手_氦检时间设定值
D6108 CHANNEL  ; 进料机械手_腔体真空实际值
D611 CHANNEL  ; 进料升降伺服手动状态减速比率
D6110 CHANNEL  ; 进料机械手_漏率
D6112 CHANNEL  ; 进料机械手_检漏口压力
D6114 CHANNEL  ; 进料机械手_腔体抽气时间
D6116 CHANNEL  ; 进料机械手_结果/NG类型
D6118 CHANNEL  ; 进料机械手_腔体工位
D6119 CHANNEL  ; 进料机械手_电池记忆
D612 CHANNEL  ; 进料升降伺服手动状态目标频率（低位）
D6120 CHANNEL  ; 进料机械手_电池条码1
D613 CHANNEL  ; 进料升降伺服手动状态目标频率（高位）
D614 CHANNEL  ; 进料升降伺服手动状态脉冲输出量（低位）
D6140 CHANNEL  ; 进料机械手_电池条码2
D615 CHANNEL  ; 进料升降伺服手动状态脉冲输出量（高位）
D616 CHANNEL  ; 进料升降伺服手动状态启动频率（低位）
D6160 CHANNEL  ; 进料机械手_电池条码3
D617 CHANNEL  ; 进料升降伺服手动状态启动频率（高位）
D618 CHANNEL  ; 进料升降伺服手动状态脉冲  Plus/s
D6180 CHANNEL  ; 进料机械手_电池条码4
D620 CHANNEL  ; 进料旋转伺服手动状态加速比率
D6200 CHANNEL  ; 进料旋转机构_腔体真空设定值
D6202 CHANNEL  ; 进料旋转机构_漏率设定值
D6204 CHANNEL  ; 进料旋转机构_检漏口压力设定值
D6206 CHANNEL  ; 进料旋转机构_氦检时间设定值
D6208 CHANNEL  ; 进料旋转机构_腔体真空实际值
D621 CHANNEL  ; 进料旋转伺服手动状态减速比率
D6210 CHANNEL  ; 进料旋转机构_漏率
D6212 CHANNEL  ; 进料旋转机构_检漏口压力
D6214 CHANNEL  ; 进料旋转机构_腔体抽气时间
D6216 CHANNEL  ; 进料旋转机构_结果/NG类型
D6218 CHANNEL  ; 进料旋转机构_腔体工位
D6219 CHANNEL  ; 进料旋转机构_电池记忆
D622 CHANNEL  ; 进料旋转伺服手动状态目标频率（低位）
D6220 CHANNEL  ; 进料旋转机构_电池条码1
D623 CHANNEL  ; 进料旋转伺服手动状态目标频率（高位）
D624 CHANNEL  ; 进料旋转伺服手动状态脉冲输出量（低位）
D6240 CHANNEL  ; 进料旋转机构_电池条码2
D625 CHANNEL  ; 进料旋转伺服手动状态脉冲输出量（高位）
D626 CHANNEL  ; 进料旋转伺服手动状态启动频率（低位）
D6260 CHANNEL  ; 进料旋转机构_电池条码4
D627 CHANNEL  ; 进料旋转伺服手动状态启动频率（高位）
D628 CHANNEL  ; 进料旋转伺服手动状态脉冲  Plus/s
D6280 CHANNEL  ; 进料旋转机构_电池条码3
D630 CHANNEL  ; 上料水平伺服手动状态加速比率
D6300 CHANNEL  ; 腔体上料机械手_腔体真空设定值
D6302 CHANNEL  ; 腔体上料机械手_漏率设定值
D6304 CHANNEL  ; 腔体上料机械手_检漏口压力设定值
D6306 CHANNEL  ; 腔体上料机械手_氦检时间设定值
D6308 CHANNEL  ; 腔体上料机械手_腔体真空实际值
D631 CHANNEL  ; 上料水平伺服手动状态减速比率
D6310 CHANNEL  ; 腔体上料机械手_漏率
D6312 CHANNEL  ; 腔体上料机械手_检漏口压力
D6314 CHANNEL  ; 腔体上料机械手_腔体抽气时间
D6316 CHANNEL  ; 腔体上料机械手_结果/NG类型
D6318 CHANNEL  ; 腔体上料机械手_腔体工位
D6319 CHANNEL  ; 腔体上料机械手_电池记忆
D632 CHANNEL  ; 上料水平伺服手动状态目标频率（低位）
D6320 CHANNEL  ; 腔体上料机械手_电池条码1
D633 CHANNEL  ; 上料水平伺服手动状态目标频率（高位）
D634 CHANNEL  ; 上料水平伺服手动状态脉冲输出量（低位）
D6340 CHANNEL  ; 腔体上料机械手_电池条码2
D635 CHANNEL  ; 上料水平伺服手动状态脉冲输出量（高位）
D636 CHANNEL  ; 上料水平伺服手动状态启动频率（低位）
D6360 CHANNEL  ; 腔体上料机械手_电池条码4
D637 CHANNEL  ; 上料水平伺服手动状态启动频率（高位）
D638 CHANNEL  ; 上料水平伺服手动状态脉冲  Plus/s
D6380 CHANNEL  ; 腔体上料机械手_电池条码3
D640 CHANNEL  ; 下料水平伺服手动状态加速比率
D6400 CHANNEL  ; 腔体#1_腔体真空设定值
D6401 CHANNEL  ; 腔体#1_腔体真空设定值
D6403 CHANNEL  ; 腔体#1_漏率设定值
D6405 CHANNEL  ; 腔体#1_检漏口压力设定值
D6407 CHANNEL  ; 腔体#1_氦检时间设定值
D6408 CHANNEL  ; 腔体#1_腔体真空实际值
D6409 CHANNEL  ; 腔体#1_腔体真空实际值
D641 CHANNEL  ; 下料水平伺服手动状态减速比率
D6410 CHANNEL  ; 腔体#1_漏率
D6411 CHANNEL  ; 腔体#1_漏率
D6412 CHANNEL  ; 腔体#1_检漏口压力
D6413 CHANNEL  ; 腔体#1_检漏口压力
D6414 CHANNEL  ; 腔体#1_腔体抽气时间
D6415 CHANNEL  ; 腔体#1_腔体抽气时间
D6416 CHANNEL  ; 腔体#1_结果/NG类型
D6417 CHANNEL  ; 腔体#1_结果/NG类型
D6418 CHANNEL  ; 腔体#1_腔体工位
D6419 CHANNEL  ; 腔体#1_腔体工位
D6419.00 BOOL  ; #1腔体1#位有电芯
D6419.01 BOOL  ; #1腔体2#位有电芯
D642 CHANNEL  ; 下料水平伺服手动状态目标频率（低位）
D6420 CHANNEL  ; 腔体#1_电池记忆
D6421 CHANNEL  ; 腔体#1_电池条码1
D643 CHANNEL  ; 下料水平伺服手动状态目标频率（高位）
D644 CHANNEL  ; 下料水平伺服手动状态脉冲输出量（低位）
D6441 CHANNEL  ; 腔体#1_电池条码2
D645 CHANNEL  ; 下料水平伺服手动状态脉冲输出量（高位）
D646 CHANNEL  ; 下料水平伺服手动状态启动频率（低位）
D647 CHANNEL  ; 下料水平伺服手动状态启动频率（高位）
D648 CHANNEL  ; 下料水平伺服手动状态脉冲  Plus/s
D6480 CHANNEL  ; #2腔体电池条码
D650 CHANNEL  ; 出料水平伺服手动状态加速比率
D6500 CHANNEL  ; 腔体#2_腔体真空设定值
D6502 CHANNEL  ; 腔体#2_漏率设定值
D6504 CHANNEL  ; 腔体#2_检漏口压力设定值
D6506 CHANNEL  ; 腔体#2_氦检时间设定值
D6508 CHANNEL  ; 腔体#2_腔体真空实际值
D651 CHANNEL  ; 出料水平伺服手动状态减速比率
D6510 CHANNEL  ; 腔体#2_漏率
D6512 CHANNEL  ; 腔体#2_检漏口压力
D6514 CHANNEL  ; 腔体#2_腔体抽气时间
D6516 CHANNEL  ; 腔体#2_结果/NG类型
D6518 CHANNEL  ; 腔体#2_腔体工位
D6519 CHANNEL  ; 腔体#2_电池记忆
D6519.00 BOOL  ; #2腔体1#位有电芯
D6519.01 BOOL  ; #2腔体2#位有电芯
D652 CHANNEL  ; 出料水平伺服手动状态目标频率（低位）
D653 CHANNEL  ; 出料水平伺服手动状态目标频率（高位）
D654 CHANNEL  ; 出料水平伺服手动状态脉冲输出量（低位）
D655 CHANNEL  ; 出料水平伺服手动状态脉冲输出量（高位）
D656 CHANNEL  ; 出料水平伺服手动状态启动频率（低位）
D6560 CHANNEL  ; 腔体#2_电池条码1
D657 CHANNEL  ; 出料水平伺服手动状态启动频率（高位）
D658 CHANNEL  ; 出料水平伺服手动状态脉冲  Plus/s
D6580 CHANNEL  ; 腔体#2_电池条码2
D660 CHANNEL  ; 出料升降伺服手动状态加速比率
D6600 CHANNEL  ; 腔体#3_腔体真空设定值
D6602 CHANNEL  ; 腔体#3_漏率设定值
D6604 CHANNEL  ; 腔体#3_检漏口压力设定值
D6606 CHANNEL  ; 腔体#3_氦检时间设定值
D6608 CHANNEL  ; 腔体#3_腔体真空实际值
D661 CHANNEL  ; 出料升降伺服手动状态减速比率
D6610 CHANNEL  ; 腔体#3_漏率
D6612 CHANNEL  ; 腔体#3_检漏口压力
D6614 CHANNEL  ; 腔体#3_腔体抽气时间
D6616 CHANNEL  ; 腔体#3_结果/NG类型
D6618 CHANNEL  ; 腔体#3_腔体工位
D6619 CHANNEL  ; 腔体#3_电池记忆
D6619.00 BOOL  ; #3腔体1#位有电芯
D6619.01 BOOL  ; #3腔体2#位有电芯
D662 CHANNEL  ; 出料升降伺服手动状态目标频率（低位）
D6620 CHANNEL  ; 腔体#3_电池条码1
D663 CHANNEL  ; 出料升降伺服手动状态目标频率（高位）
D664 CHANNEL  ; 出料升降伺服手动状态脉冲输出量（低位）
D6640 CHANNEL  ; 腔体#3_电池条码2
D665 CHANNEL  ; 出料升降伺服手动状态脉冲输出量（高位）
D666 CHANNEL  ; 出料升降伺服手动状态启动频率（低位）
D6660 CHANNEL  ; #4腔体电池条码1
D667 CHANNEL  ; 出料升降伺服手动状态启动频率（高位）
D668 CHANNEL  ; 出料升降伺服手动状态脉冲  Plus/s
D6680 CHANNEL  ; #4腔体电池条码2
D670 CHANNEL  ; 出料旋转伺服手动状态加速比率
D6700 CHANNEL  ; 腔体#4_腔体真空设定值
D6702 CHANNEL  ; 腔体#4_漏率设定值
D6704 CHANNEL  ; 腔体#4_检漏口压力设定值
D6706 CHANNEL  ; 腔体#4_氦检时间设定值
D6708 CHANNEL  ; 腔体#4_腔体真空实际值
D671 CHANNEL  ; 出料旋转伺服手动状态减速比率
D6710 CHANNEL  ; 腔体#4_漏率
D6712 CHANNEL  ; 腔体#4_检漏口压力
D6714 CHANNEL  ; 腔体#4_腔体抽气时间
D6716 CHANNEL  ; 腔体#4_结果/NG类型
D6718 CHANNEL  ; 腔体#4_腔体工位
D6719 CHANNEL  ; 腔体#4_电池记忆
D6719.00 BOOL  ; #4腔体1#位有电芯
D6719.01 BOOL  ; #4腔体2#位有电芯
D672 CHANNEL  ; 出料旋转伺服手动状态目标频率（低位）
D673 CHANNEL  ; 出料旋转伺服手动状态目标频率（高位）
D674 CHANNEL  ; 出料旋转伺服手动状态脉冲输出量（低位）
D675 CHANNEL  ; 出料旋转伺服手动状态脉冲输出量（高位）
D676 CHANNEL  ; 出料旋转伺服手动状态启动频率（低位）
D6760 CHANNEL  ; 腔体#4_电池条码3
D677 CHANNEL  ; 出料旋转伺服手动状态启动频率（高位）
D678 CHANNEL  ; 出料旋转伺服手动状态脉冲  Plus/s
D6780 CHANNEL  ; 腔体#4_电池条码4
D6800 CHANNEL  ; 腔体下料机械手1&2_腔体真空设定值
D6802 CHANNEL  ; 腔体下料机械手1&2_漏率设定值
D6804 CHANNEL  ; 腔体下料机械手1&2_检漏口压力设定值
D6806 CHANNEL  ; 腔体下料机械手1&2_氦检时间设定值
D6808 CHANNEL  ; 腔体下料机械手1&2_腔体真空实际值
D6810 CHANNEL  ; 腔体下料机械手1&2_漏率
D6812 CHANNEL  ; 腔体下料机械手1&2_检漏口压力
D6814 CHANNEL  ; 腔体下料机械手1&2_腔体抽气时间
D6816 CHANNEL  ; 腔体下料机械手1&2_结果/NG类型
D6818 CHANNEL  ; 腔体下料机械手1&2_腔体工位
D6819 CHANNEL  ; 腔体下料机械手1&2_电池记忆
D6820 CHANNEL  ; 腔体下料机械手1&2_电池条码1
D6840 CHANNEL  ; 腔体下料机械手1&2_电池条码2
D690 CHANNEL  ; 上下料水平伺服总距离（移动的距离）
D6900 CHANNEL  ; 腔体下料机械手3&4_腔体真空设定值
D6902 CHANNEL  ; 腔体下料机械手3&4_漏率设定值
D6904 CHANNEL  ; 腔体下料机械手3&4_检漏口压力设定值
D6906 CHANNEL  ; 腔体下料机械手3&4_氦检时间设定值
D6908 CHANNEL  ; 腔体下料机械手3&4_腔体真空实际值
D6910 CHANNEL  ; 腔体下料机械手3&4_漏率
D6912 CHANNEL  ; 腔体下料机械手3&4_检漏口压力
D6914 CHANNEL  ; 腔体下料机械手3&4_腔体抽气时间
D6916 CHANNEL  ; 腔体下料机械手3&4_结果/NG类型
D6918 CHANNEL  ; 腔体下料机械手3&4_腔体工位
D6919 CHANNEL  ; 腔体下料机械手3&4_电池记忆
D6919.00 BOOL  ; 旋转移载位1#有料
D6919.01 BOOL  ; 旋转移载位2#有料
D692 CHANNEL  ; 两原点之间总距离
D694 CHANNEL  ; 上下料水平伺服相距距离
D696 CHANNEL  ; 两轴限制距离
D6960 CHANNEL  ; 腔体下料机械手3&4_电池条码3
D6980 CHANNEL  ; 腔体下料机械手3&4_电池条码4
D700 CHANNEL  ; 进料水平伺服自动状态脉冲 Plus/s
D7000 CHANNEL  ; 出料旋转机构1&2_腔体真空设定值
D7001 CHANNEL  ; 左位条码
D7002 CHANNEL  ; 出料旋转机构1&2_漏率设定值
D7004 CHANNEL  ; 出料旋转机构1&2_检漏口压力设定值
D7006 CHANNEL  ; 出料旋转机构1&2_氦检时间设定值
D7008 CHANNEL  ; 出料旋转机构1&2_腔体真空实际值
D7010 CHANNEL  ; 出料旋转机构1&2_漏率
D7012 CHANNEL  ; 出料旋转机构1&2_检漏口压力
D7014 CHANNEL  ; 出料旋转机构1&2_腔体抽气时间
D7016 CHANNEL  ; 出料旋转机构1&2_结果/NG类型
D7018 CHANNEL  ; 出料旋转机构1&2_腔体工位
D7019 CHANNEL  ; 出料旋转机构1&2_电池记忆
D7019.00 BOOL  ; 旋转移载位3#有料
D7019.01 BOOL  ; 旋转移载位4#有料
D7020 CHANNEL  ; 出料旋转机构1&2_电池条码1
D7040 CHANNEL  ; 出料旋转机构1&2_电池条码2
D708 CHANNEL  ; 上料水平伺服自动状态脉冲  Puls/s
D7100 CHANNEL  ; 出料旋转机构3&4_腔体真空设定值
D7102 CHANNEL  ; 出料旋转机构3&4_漏率设定值
D7104 CHANNEL  ; 出料旋转机构3&4_检漏口压力设定值
D7106 CHANNEL  ; 出料旋转机构3&4_氦检时间设定值
D7108 CHANNEL  ; 出料旋转机构3&4_腔体真空实际值
D7110 CHANNEL  ; 出料旋转机构3&4_漏率
D7112 CHANNEL  ; 出料旋转机构3&4_检漏口压力
D7114 CHANNEL  ; 出料旋转机构3&4_腔体抽气时间
D7116 CHANNEL  ; 出料旋转机构3&4_结果/NG类型
D7118 CHANNEL  ; 出料旋转机构3&4_腔体工位
D7119 CHANNEL  ; 出料旋转机构3&4_电池记忆
D7119.00 BOOL  ; 旋转移载位1#有料
D7119.01 BOOL  ; 旋转移载位2#有料
D712 CHANNEL  ; 上料水平伺服手动状态脉冲  Puls/s
D716 CHANNEL  ; 下料水平伺服自动状态脉冲  Puls/s
D7160 CHANNEL  ; 出料旋转机构3&4_电池条码3
D7180 CHANNEL  ; 出料旋转机构3&4_电池条码4
D720 CHANNEL  ; 下料水平伺服手动状态脉冲  Puls/s
D7200 CHANNEL  ; 右位扫码长度
D7201 CHANNEL  ; 右位条码
D724 CHANNEL  ; 出料水平伺服自动状态脉冲  Puls/s
D728 CHANNEL  ; 出料水平伺服手动状态脉冲  Puls/s
D7500 CHANNEL  ; 电池条码长度设置
D7502 CHANNEL  ; 设置条码长度字
D7504 CHANNEL  ; 比较条码字长度
D7506 CHANNEL  ; #2比较条码字长度
D7550 CHANNEL  ; 重扫次数
D7560 CHANNEL  ; 复检前抽气次数设定值
D7562 CHANNEL  ; 清氦次数设定值
D7600 CHANNEL  ; 重扫次数
D800 CHANNEL  ; 氦检仪检漏状态起始字
D8000 CHANNEL  ; 检漏状态第一字节
D8001 CHANNEL  ; 检漏状态第二字节
D8002 CHANNEL  ; 检漏状态结束字节
D801 CHANNEL  ; 氦检仪接收状态
D8010 CHANNEL  ; 待机状态第一字节
D8011 CHANNEL  ; 待机状态第二字节
D8012 CHANNEL  ; 待机状态结束字节
D8020 CHANNEL  ; 定标状态第一字节
D8021 CHANNEL  ; 定标状态第二字节
D8022 CHANNEL  ; 定标状态结束字节
D8030 CHANNEL  ; 启动状态第一字节
D8031 CHANNEL  ; 启动状态第二字节
D8032 CHANNEL  ; 启动状态结束字节
D8040 CHANNEL  ; 错误状态第一字节
D8041 CHANNEL  ; 错误状态第二字节
D8042 CHANNEL  ; 错误状态结束字节
D8050 CHANNEL  ; 暂停状态第一字节
D8051 CHANNEL  ; 暂停状态第二字节
D8052 CHANNEL  ; 暂停状态结束字节
D810 CHANNEL  ; 接收检漏口压力起始字
D8100 CHANNEL  ; 氦检仪状态(1-检漏,2-待机,3-启动,4-定标,5-错误,6-暂停)
D811 CHANNEL  ; 接收的检漏口压力  ASCII
D820 CHANNEL  ; 读漏率起始字
D821 CHANNEL  ; 接收漏率ASCII.
D8400 CHANNEL  ; 读氦检仪报警
D8500 CHANNEL  ; 读氦检仪内部校准状态
D8600 CHANNEL  ; 氦检校准暂存状态1-完成
D8601 CHANNEL  ; 氦检校准暂存状态1-完成
D8610 CHANNEL  ; 氦检校准暂存状态2-通过
D8611 CHANNEL  ; 氦检校准暂存状态2-通过
D8612 CHANNEL  ; 氦检校准暂存状态3
D8620 CHANNEL  ; 氦检校准暂存状态3-进行
D8621 CHANNEL  ; 氦检校准暂存状态3-进行
D8622 CHANNEL  ; 氦检校准暂存状态3-进行
D888 CHANNEL  ; 触摸屏界面  HMI
D9000 CHANNEL  ; PC交互地址
D900.00 BOOL  ; 急停错误
D900.01 BOOL  ; 气源压力错误
D900.02 BOOL  ; 安全门开错误
D910.00 BOOL  ; 急停错误
D910.01 BOOL  ; Main Auto Start[Pls]
D910.02 BOOL  ; Main Auto Stop[Pls]
D910.03 BOOL  ; Origin Cmd
D910.05 BOOL  ; End Stop Cmd
D910.06 BOOL  ; Auto Stop Cmd
D910.07 BOOL  ; Auto Stop Complete
D910.09 BOOL  ; Buzzer Stop
D910.10 BOOL  ; All Work Empty
D910.11 BOOL  ; All Work Sensor Empty
D910.15 BOOL  ; All Cycle Stop Check
D911.00 BOOL  ; All Home Stop Check
D911.04 BOOL  ; BKT Enable
D911.05 BOOL  ; All Home Check
D911.10 BOOL  ; Emergency Stop
D911.11 BOOL  ; Safety Plug
D911.12 BOOL  ; Cp/Nfb Trip
D911.13 BOOL  ; Total Error
D911.14 BOOL  ; Total Warning
D911.15 BOOL  ; All Total Error
D912.00 BOOL  ; 自动运行中
D912.01 BOOL  ; 自动停止中
D912.02 BOOL  ; 清料停止中
D912.03 BOOL  ; 所有停止完成
D912.04 BOOL  ; 强制停止
D913.01 BOOL  ; 自动Flag
D913.02 BOOL  ; 手动Flag
D913.06 BOOL  ; 机台所有故障
D913.07 BOOL  ; 警告
D9400 CHANNEL  ; 腔体#1状态0-屏蔽 1-待料中 2-测试中 3-测试完成 4-在线复检
D9402 CHANNEL  ; 腔体#2状态0-屏蔽 1-待料中 2-测试中 3-测试完成 4-在线复检
D9404 CHANNEL  ; 腔体#3状态0-屏蔽 1-待料中 2-测试中 3-测试完成 4-在线复检
D9406 CHANNEL  ; 腔体#4状态0-屏蔽 1-待料中 2-测试中 3-测试完成 4-在线复检
D9600 CHANNEL  ; 出料机械手_腔体真空设定值
D9602 CHANNEL  ; 出料机械手_漏率设定值
D9604 CHANNEL  ; 出料机械手_检漏口压力设定值
D9606 CHANNEL  ; 出料机械手_氦检时间设定值
D9608 CHANNEL  ; 出料机械手_腔体真空实际值
D9610 CHANNEL  ; 出料机械手_漏率
D9612 CHANNEL  ; 出料机械手_检漏口压力
D9614 CHANNEL  ; 出料机械手_腔体工位
D9616 CHANNEL  ; 出料机械手_结果/NG类型
D9617 CHANNEL  ; 出料机械手_
D9618 CHANNEL  ; 出料机械手_
D9619 CHANNEL  ; 出料机械手_电池记忆
D9619.00 BOOL  ; 4-2出料模组1#电芯记忆
D9619.01 BOOL  ; 4-2出料模组2#电芯记忆
D9620 CHANNEL  ; 出料机械手_电池条码1
D9640 CHANNEL  ; 出料机械手_电池条码2
D9804 CHANNEL  ; MES接口调用结果（左位）
D9904 CHANNEL  ; MES接口调用结果（右位）
E0_0 CHANNEL  ; 异常延时
E0_32100 CHANNEL  ; 总计
E0_32102 CHANNEL  ; OK数
E0_32104 CHANNEL  ; NG数
E0_8 CHANNEL  ; Run Delay
E2_2590.00 BOOL  ; 焊接总OK
E2_2594.00 BOOL  ; 贴胶总OK
E2_3100.00 BOOL  ; 300B-11StCell Mover-1Product Detect
H0.00 BOOL  ; 1-空跑  0-正常
H0.01 BOOL  ; #1腔体  1-屏蔽   0-启用
H0.02 BOOL  ; #2腔体  1-屏蔽  0-启用
H0.03 BOOL  ; 扫码屏蔽(1-屏蔽  0-启用)
H0.04 BOOL  ; 重复扫码1-屏蔽  0-启用
H0.05 BOOL  ; 氦检仪 1-屏蔽  0-启用
H0.06 BOOL  ; MES调用 1-屏蔽 0-启用
H0.07 BOOL  ; 门磁屏蔽 1-屏蔽  0-启用
H0.09 BOOL  ; 电脑 1 -屏蔽 0-启用
H0.10 BOOL  ; 真空泵屏蔽  HMI
H0.11 BOOL  ; 拉带屏蔽  HMI
H0.12 BOOL  ; 复测开
H0.13 BOOL  ; 清氦功能打开
H10.00 BOOL  ; 扫码左阻挡缩回屏蔽  HMI
H10.01 BOOL  ; 扫码左阻挡伸出屏蔽  HMI
H10.02 BOOL  ; 扫码右阻挡缩回屏蔽  HMI
H10.03 BOOL  ; 扫码右阻挡伸出屏蔽  HMI
H10.04 BOOL  ; 左隔离气缸缩回屏蔽  HMI
H10.05 BOOL  ; 左隔离气缸伸出屏蔽  HMI
H10.06 BOOL  ; 右隔离气缸缩回屏蔽  HMI
H10.07 BOOL  ; 右隔离气缸伸出屏蔽  HMI
H10.08 BOOL  ; 扫码缓存推料气缸缩回屏蔽   HMI
H10.09 BOOL  ; 扫码缓存推料气缸伸出屏蔽   HMI
H10.10 BOOL  ; 进料移栽伸缩气缸缩回屏蔽  HMI
H10.11 BOOL  ; 进料移栽伸缩气缸伸出屏蔽   HMI
H10.12 BOOL  ; 进料#1夹爪张开位屏蔽  HMI
H10.13 BOOL  ; 进料#1夹爪夹紧屏蔽  HMI
H10.14 BOOL  ; 进料#2夹爪张开屏蔽  HMI
H10.15 BOOL  ; 进料#2夹爪夹紧屏蔽  HMI
H11.00 BOOL  ; 上料提升气缸上升屏蔽  HMI
H11.01 BOOL  ; 上料提升气缸下降屏蔽  HMI
H11.02 BOOL  ; 上料#1夹爪张开屏蔽  HMI
H11.03 BOOL  ; 上料#1夹爪夹紧屏蔽  HMI
H11.04 BOOL  ; 上料#2夹爪张开屏蔽  HMI
H11.05 BOOL  ; 上料#2夹爪夹紧屏蔽  HMI
H11.06 BOOL  ; 上料#3夹爪张开屏蔽  HMI
H11.07 BOOL  ; 上料#3夹爪夹紧屏蔽  HMI
H11.08 BOOL  ; 上料#4夹爪张开屏蔽  HMI
H11.09 BOOL  ; 上料#4夹爪夹紧屏蔽  HMI
H11.10 BOOL  ; 下料提升气缸上升屏蔽  HMI
H11.11 BOOL  ; 下料提升气缸下降屏蔽  HMI
H11.12 BOOL  ; 下料#1夹爪张开屏蔽  HMI
H11.13 BOOL  ; 下料#1夹爪夹紧屏蔽  HMI
H11.14 BOOL  ; 下料#2夹爪张开屏蔽  HMI
H11.15 BOOL  ; 下料#2夹爪夹紧屏蔽  HMI
H12.00 BOOL  ; 下料#3夹爪张开屏蔽  HMI
H12.01 BOOL  ; 下料#3夹爪夹紧屏蔽  HMI
H12.02 BOOL  ; 下料#4夹爪张开屏蔽  HMI
H12.03 BOOL  ; 下料#4夹爪夹紧屏蔽  HMI
H12.04 BOOL  ; #1合模气缸缩回屏蔽  HMI
H12.05 BOOL  ; #1合模气缸伸出屏蔽  HMI
H12.06 BOOL  ; #2合模气缸缩回屏蔽  HMI
H12.07 BOOL  ; #2合模气缸伸出屏蔽  HMI
H12.08 BOOL  ; #3合模气缸缩回屏蔽  HMI
H12.09 BOOL  ; #3合模气缸伸出屏蔽  HMI
H12.10 BOOL  ; #4合模气缸缩回屏蔽  HMI
H12.11 BOOL  ; #4合模气缸伸出屏蔽  HMI
H12.12 BOOL  ; #1总氦检阀关闭屏蔽
H12.13 BOOL  ; #1总氦检阀打开屏蔽  HMI
H12.14 BOOL  ; #2总氦检阀关闭屏蔽
H12.15 BOOL  ; #2总氦检阀打开屏蔽  HMI
H13.00 BOOL  ; #1氦检阀关闭屏蔽  HMI
H13.01 BOOL  ; #1氦检阀打开屏蔽  HMI
H13.02 BOOL  ; #2氦检阀关闭屏蔽  HMI
H13.03 BOOL  ; #2氦检阀打开屏蔽  HMI
H13.04 BOOL  ; #3氦检阀关闭屏蔽  HMI
H13.05 BOOL  ; #3氦检阀打开屏蔽延时  HMI
H13.06 BOOL  ; #4氦检阀关闭屏蔽延时  HMI
H13.07 BOOL  ; #4氦检阀打开屏蔽  HMI
H13.08 BOOL  ; 出料移栽伸缩气缸缩回屏蔽  HMI
H13.09 BOOL  ; 出料移栽伸缩气缸伸出屏蔽  HMI
H13.10 BOOL  ; 检测NG推料气缸缩回屏蔽  HMI
H13.11 BOOL  ; 检测NG推料气缸伸出屏蔽  HMI
H13.12 BOOL  ; 出料#1夹爪张开屏蔽  HMI
H13.13 BOOL  ; 出料#1夹爪夹紧屏蔽  HMI
H13.14 BOOL  ; 出料#2夹爪张开屏蔽  HMI
H13.15 BOOL  ; 出料#2夹爪夹紧屏蔽  HMI
H188.08 BOOL  ; 调试临时
H1.00 BOOL  ; 整机复位完成记忆
H25.00 BOOL  ; 进料水平伺服归零完成
H25.01 BOOL  ; 进料升降伺服归零完成
H25.02 BOOL  ; 进料旋转伺服归零完成
H25.03 BOOL  ; 上料水平伺服归零完成
H25.04 BOOL  ; 下料水平伺服归零完成
H25.05 BOOL  ; 出料水平伺服归零完成
H25.06 BOOL  ; 出料升降伺服归零完成
H25.07 BOOL  ; 出料旋转伺服归零完成
H25.13 BOOL  ; 断腔体上料伺服归零
H25.14 BOOL  ; 断下料水平伺服归零
H31.00 BOOL  ; #1复检中
H31.01 BOOL  ; #1模组清氦OK
H31.03 BOOL  ; #1清氦完成
H31.04 BOOL  ; #1复检完成
H31.05 BOOL  ; #1& #2腔体测试中
H32.00 BOOL  ; #2复检中
H32.01 BOOL  ; #2模组清氦OK
H32.04 BOOL  ; #2复检完成
H33.00 BOOL  ; #3复检中
H33.01 BOOL  ; #3模组清氦OK
H33.03 BOOL  ; #3清氦完成
H33.04 BOOL  ; #3复检完成
H33.05 BOOL  ; #3& #4腔体测试中
H34.00 BOOL  ; #4复检中
H34.01 BOOL  ; #4模组清氦OK
H34.04 BOOL  ; #4复检完成
H35.00 BOOL  ; #1、#2腔体测试完成标志
H35.01 BOOL  ; #3、#4腔体测试完成标志
H3.12 BOOL  ; 上对接开
H3.15 BOOL  ; 下对接开
H40.00 BOOL  ; 进料夹爪无料记忆辅助
H40.01 BOOL  ; 上料夹爪无料记忆辅助
H40.02 BOOL  ; 下料夹爪无料记忆辅助
H40.03 BOOL  ; 出料夹爪无料记忆辅助
H40.04 BOOL  ; 腔体无料记忆辅助
H40.05 BOOL  ; 拉带无料状态辅助
H40.06 BOOL  ; 进料移栽位无料状态
H40.07 BOOL  ; 出料移栽无料状态
H40.08 BOOL  ; 扫码OK配对位无料状态
H501.02 BOOL  ; 500_2St有料记忆
H50.00 BOOL  ; 1#扫码OK记忆
H50.01 BOOL  ; 2#扫码OK记忆
H50.02 BOOL  ; 1#扫码NG记忆
H50.03 BOOL  ; 2#扫码NG记忆
H50.04 BOOL  ; 进料1#夹爪OK有料记忆
H50.05 BOOL  ; 进料2#夹爪OK有料记忆
H50.06 BOOL  ; 进料1#夹爪NG料
H50.07 BOOL  ; 进料2#夹爪NG料
H50.08 BOOL  ; 扫码OK配对位有料
H50.09 BOOL  ; 扫码NG缓存左下料位有料
H50.10 BOOL  ; 扫码NG缓存右下料位有料
H50.11 BOOL  ; 扫码NG缓存左位有料
H50.12 BOOL  ; 扫码NG缓存右位有料
H51.02 BOOL  ; 左夹爪配对OK记忆
H51.03 BOOL  ; 右夹爪配对OK记忆
H51.05 BOOL  ; 进料#1移栽位有料
H51.06 BOOL  ; 进料#2移栽位有料
H51.07 BOOL  ; 进料#3移栽位有料
H51.08 BOOL  ; 进料#4移栽位有料
H51.09 BOOL  ; 出料#1移栽位有料
H51.10 BOOL  ; 出料#2移栽位有料
H51.11 BOOL  ; 出料#3移栽位有料
H51.12 BOOL  ; 出料#4移栽位有料
H51.13 BOOL  ; 出料#1爪有OK料
H51.14 BOOL  ; 出料#2爪有OK料
H51.15 BOOL  ; 出料#1爪有NG料
H52.00 BOOL  ; 出料#2爪有NG料
H52.01 BOOL  ; 出料#1NG缓存位有料
H52.02 BOOL  ; 出料#2NG缓存位有料
H52.03 BOOL  ; 出料#3NG缓存位有料
H52.04 BOOL  ; 出料#4NG缓存位有料
H52.06 BOOL  ; 出料#1NG缓存下料位有料
H52.07 BOOL  ; 出料#2NG缓存下料位有料
H52.08 BOOL  ; 出料#3NG缓存下料位有料
H52.09 BOOL  ; 出料#4NG缓存下料位有料
H52.12 BOOL  ; 进料#1夹爪有料记忆
H52.13 BOOL  ; 进料#2夹爪有料记忆
H52.14 BOOL  ; 出料夹爪#1有料
H52.15 BOOL  ; 出料夹爪#2有料
H53.00 BOOL  ; 进料夹爪#1手动记忆有料
H53.01 BOOL  ; 进料夹爪#2手动记忆有料
H53.02 BOOL  ; 上料夹爪#1手动记忆有料
H53.03 BOOL  ; 上料夹爪#2手动记忆有料
H53.04 BOOL  ; 上料夹爪#3手动记忆有料
H53.05 BOOL  ; 上料夹爪#4手动记忆有料
H53.06 BOOL  ; 下料夹爪#1手动记忆有料
H53.07 BOOL  ; 下料夹爪#2手动记忆有料
H53.08 BOOL  ; 下料夹爪#3手动记忆有料
H53.09 BOOL  ; 下料夹爪#4手动记忆有料
H53.10 BOOL  ; 出料夹爪#1手动记忆有料
H53.11 BOOL  ; 出料夹爪#2手动记忆有料
H55.00 BOOL  ; 上料#1夹爪有料标志
H55.01 BOOL  ; 上料#2夹爪有料标志
H55.02 BOOL  ; 上料#3夹爪有料标志
H55.03 BOOL  ; 上料#4夹爪有料标志
H55.04 BOOL  ; 下料#1夹爪有料标志
H55.05 BOOL  ; 下料#2夹爪有料标志
H55.06 BOOL  ; 下料#3夹爪有料标志
H55.07 BOOL  ; 下料#4夹爪有料标志
H55.08 BOOL  ; 上料水平伺服去#1腔体标志
H55.09 BOOL  ; 下料水平伺服去#1腔体标志
H55.10 BOOL  ; 上料水平伺服去#2腔体标志
H55.11 BOOL  ; 下料水平伺服去#2腔体标志
H56.00 BOOL  ; 1#上料OK记忆
H56.01 BOOL  ; 2#上料OK记忆
H56.02 BOOL  ; 1#上料NG记忆
H56.03 BOOL  ; 2#上料NG记忆
H57.00 BOOL  ; 缓存有料记忆
H5.15 BOOL  ; 清氦后进行氦检确认
H60.00 BOOL  ; #1腔体测试完成标志
H60.01 BOOL  ; #2腔体测试完成标志
H60.02 BOOL  ; #1、#2腔体放料完成标志
H60.03 BOOL  ; #2腔体放料完成标志
H60.04 BOOL  ; #1 & #2腔体有料标记
H60.05 BOOL  ; #3 & #4腔体有料标记
H60.06 BOOL  ; 腔体#1-1有料标记
H60.07 BOOL  ; 腔体#1-2有料标记
H60.08 BOOL  ; 腔体#2-1有料标记
H60.09 BOOL  ; 腔体#2-2有料标记
H60.10 BOOL  ; 腔体#3-1有料标记
H60.11 BOOL  ; 腔体#3-2有料标记
H60.12 BOOL  ; 腔体#4-1有料标记
H60.13 BOOL  ; 腔体#4-2有料标记
H60.14 BOOL  ; #1腔体有待测料
H70.00 BOOL  ; 上料加速
H81.00 BOOL  ; 老氦检仪选择
H81.01 BOOL  ; 氦检仪电源关闭中
H8.00 BOOL  ; 进料水平伺服归零标志
H8.01 BOOL  ; 进料升降伺服归零标志
H8.02 BOOL  ; 进料旋转伺服归零标志
H8.03 BOOL  ; 上料水平伺服归零标志
H8.04 BOOL  ; 下料水平伺服归零标志
H8.05 BOOL  ; 出料水平伺服归零标志
H8.06 BOOL  ; 出料升降伺服归零标志
H8.07 BOOL  ; 出料移栽伺服归零标志
T0000 BOOL  ; PLC上电
T0001 BOOL  ; PC断线持续时间
T0002 BOOL  ; PC正常持续时间
T0003 BOOL  ; 启动延时  2秒
T0004 BOOL  ; 自动停止完成延时
T0005 BOOL  ; 整机在初始位延时
T0006 BOOL  ; 切换手动延时
T0007 BOOL  ; 切换自动延时
T0008 BOOL  ; 停止开关ON延时
T0009 BOOL  ; 机台有故障延时
T0010 BOOL  ; 启动进料旋转步进延时
T0011 BOOL  ; 1St#1 Cell MoveTask Start Delay
T0013 BOOL  ; 推料伸出延时
T0014 BOOL  ; 复位开关ON延时
T0015 BOOL  ; 整机初始化延时
T0016 BOOL  ; 启动进料放料缓存步进延时
T0017 BOOL  ; 直接NG缓存放料延时
T0018 BOOL  ; 配对缓存步进延时
T0019 BOOL  ; 切换手动延时复位自动SET
T0020 BOOL  ; 进料旋转机构步进延时
T0021 BOOL  ; 进料输送启动延时
T0023 BOOL  ; 整机在初始位延时
T0025 BOOL  ; 1#位扫码完成延时
T0026 BOOL  ; 2#位扫码完成延时
T0030 BOOL  ; 出料升降伺服柔性异常延时
T0031 BOOL  ; 进料升降伺服柔性异常延时
T0033 BOOL  ; PC数据调试延时
T0034 BOOL  ; PC数据调试延时
T0035 BOOL  ; 延时归零
T0040 BOOL  ; 进料夹爪取料后无法往下放料判断延时
T0090 BOOL  ; 进料机构在初始位延时
T0102 BOOL  ; 进料水平轴空闲=1
T0103 BOOL  ; 进料旋转伺服停止延时
T0104 BOOL  ; 进料升降伺服停止延时
T0105 BOOL  ; 进料机构感应器异常延时
T0106 BOOL  ; 进料机构伺服异常延时
T0107 BOOL  ; 进料机构升降回待料位 延时
T0108 BOOL  ; 气源压力过低延时
T0109 BOOL  ; 延时关氦检仪没稳定报警
T0111 BOOL  ; #1抽真空阀关闭延时
T0112 BOOL  ; #2抽真空阀关闭延时
T0113 BOOL  ; #1、#2破真空阀关闭延时
T0114 BOOL  ; #1、#2抽真空值到达延时
T0115 BOOL  ; #1/#2破真空阀值延时
T0116 BOOL  ; #1/#2氦检阀关闭延时
T0117 BOOL  ; #1 & #2腔体抽真空异常结束延时跳转
T0118 BOOL  ; 都没有氦检延时
T0121 BOOL  ; #3抽真空阀关闭延时
T0122 BOOL  ; #4抽真空阀关闭延时
T0123 BOOL  ; #3、#4破真空阀关闭延时
T0124 BOOL  ; #3、#4抽真空值到达延时
T0125 BOOL  ; #3、#4破真空阀值延时
T0126 BOOL  ; #3、#4氦检阀关闭延时
T0127 BOOL  ; #3 & #4腔体抽真空异常结束延时跳转
T0130 BOOL  ; 上料水平伺服脉冲输出停止延时
T0131 BOOL  ; 下料伺服自动定位延时
T0132 BOOL  ; 下料伺服自动定位关延时
T0135 BOOL  ; 上料机构手感应器异常延时
T0136 BOOL  ; 上料机构手在初始位延时
T0137 BOOL  ; 腔体上料伺服延时报警
T0138 BOOL  ; 腔体上料柔性报警延时
T0140 BOOL  ; 下料水平伺服脉冲输出停止延时
T0141 BOOL  ; 上料伺服自动定位延时
T0142 BOOL  ; 上料伺服自动定位关延时
T0145 BOOL  ; 下料机构手感应器异常延时
T0146 BOOL  ; 下料机构手在初始位延时
T0148 BOOL  ; 腔体下料伺服延时报警
T0149 BOOL  ; 腔体下料柔性报警延时
T0153 BOOL  ; 出料旋转伺服停止延时
T0155 BOOL  ; 腔体#1 & #2感应器异常延时
T0156 BOOL  ; 腔体#3 & #4感应器异常延时
T0160 BOOL  ; #1腔体自检数据初始化延时
T0161 BOOL  ; #1腔体抽真空设定时间
T0162 BOOL  ; #1腔体自检保压前延时
T0163 BOOL  ; 腔体自检保压设定时间
T0164 BOOL  ; #1腔体自检破真空到达延时
T0165 BOOL  ; #1腔体抽真空失败延时跳转
T0166 BOOL  ; #1复检关氦检后延时
T0167 BOOL  ; #1复检关破真空后延时
T0170 BOOL  ; #2腔体自检数据初始化延时
T0171 BOOL  ; #2腔体抽真空设定时间
T0172 BOOL  ; #2腔体自检保压前延时
T0173 BOOL  ; #2腔体自检保压设定时间
T0174 BOOL  ; #2腔体自检破真空到达延时
T0175 BOOL  ; #2腔体抽真空失败延时跳转
T0176 BOOL  ; 腔体#1 & #2在初始位延时
T0177 BOOL  ; 腔体#3 & #4在初始位延时
T0180 BOOL  ; #3腔体自检数据初始化延时
T0181 BOOL  ; #3腔体抽真空设定时间
T0182 BOOL  ; #3腔体自检保压前延时
T0183 BOOL  ; #3腔体自检保压设定时间
T0184 BOOL  ; #3腔体自检破真空到达延时
T0185 BOOL  ; #3腔体抽真空失败延时跳转
T0190 BOOL  ; #4腔体自检数据初始化延时
T0191 BOOL  ; #4腔体抽真空设定时间
T0192 BOOL  ; #4腔体自检保压前延时
T0193 BOOL  ; #4腔体自检保压设定时间
T0194 BOOL  ; #4腔体自检破真空到达延时
T0195 BOOL  ; #4腔体抽真空失败延时跳转
T0200 BOOL  ; 自动回进料水平伺服上料位辅助延时
T0201 BOOL  ; 自动回进料水平伺服左爪OK配对位辅助延时
T0202 BOOL  ; 自动回进料水平伺服右爪OK配对位辅助延时
T0203 BOOL  ; 自动回进料水平伺服左爪缓存位辅助延时
T0204 BOOL  ; 自动回进料水平伺服右爪缓存位辅助延时
T0205 BOOL  ; 自动回进料水平伺服缓存位辅助延时
T0206 BOOL  ; 备用
T0207 BOOL  ; 备用
T0208 BOOL  ; 备用
T0209 BOOL  ; 自动回进料水平伺服放料位辅助延时
T0210 BOOL  ; 备用
T0211 BOOL  ; 进料升降伺服回上料位辅助延时
T0212 BOOL  ; 进料升降伺服回放料位辅助延时
T0213 BOOL  ; 进料升降伺服回待料位辅助延时
T0214 BOOL  ; 备用
T0215 BOOL  ; 进料旋转伺服回#1待料位辅助延时
T0216 BOOL  ; 进料旋转伺服回#2待料位辅助延时
T0217 BOOL  ; 进料旋转伺服回上料位位辅助延时
T0218 BOOL  ; 自动回上料料水平伺服待料位辅助延时
T0219 BOOL  ; 自动回上料料水平伺服#1腔体位辅助延时
T0220 BOOL  ; 自动回上料料水平伺服#2腔体位辅助延时
T0221 BOOL  ; 自动回下料水平伺服#1腔体位辅助延时
T0222 BOOL  ; 自动回下料水平伺服#2腔体位辅助延时
T0223 BOOL  ; 自动回下料水平伺服放料位辅助延时
T0224 BOOL  ; 自动回出料水平伺服取料位辅助延时
T0225 BOOL  ; 自动回出料水平伺服#1缓存位辅助延时
T0226 BOOL  ; 自动回出料水平伺服#2缓存位辅助延时
T0227 BOOL  ; 出料水平伺服自动回放料待机位延时
T0229 BOOL  ; 自动回出料水平伺服放料位辅助延时
T0230 BOOL  ; 出料升降伺服回待料位辅助延时
T0231 BOOL  ; 出料升降伺服回取料位辅助延时
T0232 BOOL  ; 出料升降伺服回放料位辅助延时
T0233 BOOL  ; 出料旋转伺服回#1出料位辅助延时
T0234 BOOL  ; 出料旋转伺服回#2出料位辅助延时
T0235 BOOL  ; 出料旋转伺服回待料位辅助延时
T0250 BOOL  ; 进料水平伺服归零辅助延时
T0251 BOOL  ; 进料水平伺服前进辅助延时
T0252 BOOL  ; 进料水平伺服后退辅助延时
T0253 BOOL  ; 手动回进料水平伺服上料位辅助延时
T0254 BOOL  ; 手动回进料水平伺服左爪OK配对位辅助延时
T0255 BOOL  ; 手动回进料水平伺服右爪OK配对位辅助延时
T0256 BOOL  ; 手动回进料水平伺服左爪缓存位辅助延时
T0257 BOOL  ; 手动回进料水平伺服右爪缓存位辅助延时
T0258 BOOL  ; 手动回进料水平伺服缓存位辅助延时
T0259 BOOL  ; 手动回进料水平伺服放料位辅助延时
T0261 BOOL  ; 进料升降伺服归零辅助延时
T0262 BOOL  ; 进料升降伺服前进辅助延时
T0263 BOOL  ; 进料升降伺服后退辅助延时
T0264 BOOL  ; 进料升降伺服回上料位辅助延时
T0265 BOOL  ; 进料升降伺服回放料位辅助延时
T0266 BOOL  ; 进料升降伺服回待料位辅助延时
T0269 BOOL  ; 进料旋转伺服归零辅助延时
T0270 BOOL  ; 进料旋转伺服前进辅助延时
T0271 BOOL  ; 进料旋转伺服后退辅助延时
T0272 BOOL  ; 进料旋转伺服回#1待料位辅助延时
T0273 BOOL  ; 进料旋转伺服回#2待料位辅助延时
T0274 BOOL  ; 进料旋转伺服回上料位位辅助延时
T0275 BOOL  ; 备用
T0276 BOOL  ; 备用
T0277 BOOL  ; 上料水平伺服归零辅助延时
T0278 BOOL  ; 上料水平伺服前进辅助延时
T0279 BOOL  ; 上料水平伺服后退辅助延时
T0280 BOOL  ; 手动回上料料水平伺服待料位辅助延时
T0281 BOOL  ; 手动回上料料水平伺服#1腔体位辅助延时
T0282 BOOL  ; 手动回上料料水平伺服#2腔体位辅助延时
T0283 BOOL  ; 下料水平伺服归零辅助延时
T0284 BOOL  ; 下料水平伺服前进辅助延时
T0285 BOOL  ; 下料水平伺服后退辅助延时
T0286 BOOL  ; 手动回下料水平伺服#1腔体位辅助延时
T0287 BOOL  ; 手动回下料水平伺服#2腔体位辅助延时
T0288 BOOL  ; 手动回下料水平伺服放料位辅助延时
T0289 BOOL  ; 出料水平伺服归零辅助延时
T0290 BOOL  ; 出料水平伺服前进辅助延时
T0291 BOOL  ; 出料水平伺服后退辅助延时
T0292 BOOL  ; 手动回出料水平伺服取料位辅助延时
T0293 BOOL  ; 手动回出料水平伺服#1缓存位辅助延时
T0294 BOOL  ; 手动回出料水平伺服#2缓存位辅助延时
T0295 BOOL  ; 手动回出料水平伺服放料待机位延时
T0297 BOOL  ; 手动回出料水平伺服放料位辅助延时
T0300 BOOL  ; #1腔体有料感应延时
T0301 BOOL  ; #2腔体有料感应延时
T0302 BOOL  ; 氦检仪电源关闭延时
T0303 BOOL  ; 氦检仪电源打开延时延时
T0320 BOOL  ; 扫码1#阻挡缩回位延时
T0321 BOOL  ; 扫码1#阻挡伸出位延时
T0322 BOOL  ; 扫码2#阻挡缩回位延时
T0323 BOOL  ; 扫码2#阻挡伸出位延时
T0324 BOOL  ; 1#隔离气缸缩回位延时
T0325 BOOL  ; 左隔离气缸伸出位延时
T0326 BOOL  ; 2#隔离气缸缩回位延时
T0327 BOOL  ; 右隔离气缸伸出位延时
T0328 BOOL  ; 扫码缓存推料气缸缩回位延时
T0329 BOOL  ; 扫码缓存推料气缸伸出位延时
T0330 BOOL  ; 进料旋转伸缩气缸缩回位延时
T0331 BOOL  ; 进料移栽伸缩气缸伸出位延时
T0332 BOOL  ; 进料1#夹爪张开位延时
T0333 BOOL  ; 进料1#夹爪夹紧位延时
T0334 BOOL  ; 进料2#夹爪张开位延时
T0335 BOOL  ; 进料2#夹爪夹紧位延时
T0336 BOOL  ; 上料提升气缸缩回位延时
T0337 BOOL  ; 上料提升气缸伸出延时
T0338 BOOL  ; 上料#1夹爪张开位延时
T0339 BOOL  ; 上料#1夹爪夹紧位延时
T0340 BOOL  ; 上料#2夹爪张开位延时
T0341 BOOL  ; 上料#2夹爪夹紧位延时
T0342 BOOL  ; 上料#3夹爪张开位延时
T0343 BOOL  ; 上料#3夹爪夹紧位延时
T0344 BOOL  ; 上料#4夹爪张开位延时
T0345 BOOL  ; 上料#4夹爪夹紧位延时
T0346 BOOL  ; 下料提升气缸缩回位延时
T0347 BOOL  ; 下料提升气缸伸出延时
T0348 BOOL  ; 下料#1夹爪张开位延时
T0349 BOOL  ; 下料#1夹爪夹紧位延时
T0350 BOOL  ; 下料#2夹爪张开位延时
T0351 BOOL  ; 下料#2夹爪夹紧位延时
T0352 BOOL  ; 下料#3夹爪张开位延时
T0353 BOOL  ; 下料#3夹爪夹紧延时
T0354 BOOL  ; 下料#4夹爪张开位延时
T0355 BOOL  ; 下料#4夹爪夹紧位延时
T0356 BOOL  ; #1合模气缸缩回位延时
T0357 BOOL  ; #1合模气缸伸出位延时
T0358 BOOL  ; #2合模气缸缩回位延时
T0359 BOOL  ; #2合模气缸伸出位延时
T0360 BOOL  ; #3合模气缸缩回位延时
T0361 BOOL  ; #3合模伸出位延时
T0362 BOOL  ; #4合模气缸缩回位延时
T0363 BOOL  ; #4合模气缸伸出位延时
T0364 BOOL  ; #1总氦检阀关闭位延时
T0365 BOOL  ; #1总氦检阀打开延时
T0366 BOOL  ; #2总氦检阀关闭位延时
T0367 BOOL  ; #2总氦检阀打开延时
T0368 BOOL  ; #1氦检阀关闭位延时
T0369 BOOL  ; #1氦检阀打开位延时
T0370 BOOL  ; #2氦检阀关闭延时
T0371 BOOL  ; #2氦检阀打开延时
T0372 BOOL  ; #3氦检阀关闭延时
T0373 BOOL  ; #3氦检阀打开延时
T0374 BOOL  ; #4氦检阀关闭延时
T0375 BOOL  ; #4氦检阀打开延时
T0376 BOOL  ; 出料旋转伸缩气缸缩回延时
T0377 BOOL  ; 出料旋转伸缩气缸伸出延时
T0378 BOOL  ; 检测NG推料气缸缩回位延时
T0379 BOOL  ; 检测NG推料气缸伸出位延时
T0380 BOOL  ; 出料#1夹爪张开延位时
T0381 BOOL  ; 出料#1夹爪夹紧位延时
T0382 BOOL  ; 出料#2夹爪张开位延时
T0383 BOOL  ; 出料#2夹爪夹紧位延时
T0390 BOOL  ; #4氦检气缸原位延时
T0392 BOOL  ; #1真空泵启动延时
T0393 BOOL  ; #1真空泵关闭延时
T0394 BOOL  ; #2真空泵启动延时
T0395 BOOL  ; #2真空泵关闭延时
T0410 BOOL  ; 真空屏蔽
T0411 BOOL  ; 开抽真空延时
T0412 BOOL  ; 1#腔体抽真空设置时间到达
T0413 BOOL  ; 氦检延时关抽气阀
T0414 BOOL  ; 氦检时间
T0415 BOOL  ; #1腔体氦检正常结束数据传递延时
T0416 BOOL  ; 抽残气延时
T0417 BOOL  ; 破真空阀值到达延时
T0418 BOOL  ; 开腔体#1到达延时
T0419 BOOL  ; #1延时打开氦检阀
T0420 BOOL  ; #1、#2清氦抽真空计数步延时
T0421 BOOL  ; #1抽真空时间
T0422 BOOL  ; 腔体#1、#2复检关抽真空延时
T0423 BOOL  ; #1、#2氦检时间
T0425 BOOL  ; #1、#2腔体氦检正常结束数据传递延时
T0426 BOOL  ; #1/#2破真空阀值到达延时
T0427 BOOL  ; #1、#2腔体吹气延时
T0428 BOOL  ; #1/#2破真空延时
T0429 BOOL  ; #1复检关破真空后延时
T0430 BOOL  ; 真空屏蔽
T0431 BOOL  ; 开抽真空延时
T0432 BOOL  ; 3#腔体抽真空设置时间到达
T0433 BOOL  ; 氦检延时关抽气阀
T0434 BOOL  ; 氦检时间
T0435 BOOL  ; #3腔体氦检正常结束数据传递延时
T0436 BOOL  ; 抽残气延时
T0437 BOOL  ; 破真空阀值到达延时
T0438 BOOL  ; 开腔体#1到达延时
T0439 BOOL  ; #3延时打开氦检阀
T0440 BOOL  ; #3、#4清氦抽真空计数步延时
T0441 BOOL  ; #3抽真空时间
T0442 BOOL  ; 腔体#3、#4复检关抽真空延时
T0443 BOOL  ; #3、#4氦检时间
T0445 BOOL  ; #3、#4腔体氦检正常结束数据传递延时
T0446 BOOL  ; #3、#4破真空阀值到达延时
T0447 BOOL  ; #3、#4腔体吹气延时
T0448 BOOL  ; #1/#2破真空延时
T0449 BOOL  ; #3复检关破真空后延时
T0450 BOOL  ; 1#腔体抽残气超时
T0451 BOOL  ; 2#腔体抽残气超时
T0455 BOOL  ; 检测异常结束
T0456 BOOL  ; 检测异常传输
T0463 BOOL  ; #1总氦检气缸伸出位延时
T0465 BOOL  ; #2总氦检气缸伸出位延时
T0466 BOOL  ; #1氦检气缸原位延时
T0468 BOOL  ; #2氦检气缸原位延时
T0470 BOOL  ; #3氦检气缸原位延时
T0472 BOOL  ; #4氦检气缸原位延时
T0481 BOOL  ; 出料移栽放料位有料感应（常闭）延时
T0502 BOOL  ; 自动回进料升降伺服待料位辅助延时
T0504 BOOL  ; 旋转到待料位延时
T0531 BOOL  ; 下料夹紧延时
T0532 BOOL  ; #3&#4腔体夹紧延时
T0533 BOOL  ; 数据传到旋转托盘延时
T0534 BOOL  ; 延时传送数据
T0535 BOOL  ; 腔体#1 & #2数据延时传送
T0536 BOOL  ; 腔体#3 & #4数据延时传送
T0600 BOOL  ; 扫码左阻挡缩回异常延时
T0601 BOOL  ; 扫码左阻挡伸出异常延时
T0602 BOOL  ; 扫码右阻挡缩回异常延时
T0603 BOOL  ; 扫码右阻挡伸出异常延时
T0604 BOOL  ; 左隔离气缸缩回异常延时
T0605 BOOL  ; 左隔离气缸伸出异常延时
T0606 BOOL  ; 右隔离气缸缩回异常延时
T0607 BOOL  ; 右隔离气缸伸出异常
T0608 BOOL  ; 扫码NG缓存推料气缸缩回异常延时
T0609 BOOL  ; 扫码NG缓存推料气缸伸出异常延时
T0610 BOOL  ; 进料移栽伸缩气缸缩回异常延时
T0611 BOOL  ; 进料移栽伸缩气缸伸出异常延时
T0612 BOOL  ; 进料#1夹爪张开异常延时
T0613 BOOL  ; 进料#1夹爪夹紧异常延时
T0614 BOOL  ; 进料#2夹爪张开异常延时
T0615 BOOL  ; 进料#2夹爪夹紧异常延时
T0616 BOOL  ; 上料提升气缸上升异常延时
T0617 BOOL  ; 上料提升气缸下降异常延时
T0618 BOOL  ; 上料#1夹爪张开异常延时
T0619 BOOL  ; 上料#1夹爪夹紧异常延时
T0620 BOOL  ; 上料#2夹爪张开异常延时
T0621 BOOL  ; 上料#2夹爪夹紧异常延时
T0622 BOOL  ; 上料#2夹爪张开异常延时
T0623 BOOL  ; 上料#3夹爪夹紧异常延时
T0624 BOOL  ; 上料#4夹爪张开异常延时
T0625 BOOL  ; 上料#4夹爪夹紧异常延时
T0626 BOOL  ; 下料提升气缸上升异常延时
T0627 BOOL  ; 下料提升气缸下降异常延时
T0628 BOOL  ; 下料#1夹爪张开异常延时
T0629 BOOL  ; 下料#1夹爪夹紧异常延时
T0630 BOOL  ; 下料#2夹爪张开异常延时
T0631 BOOL  ; 下料#2夹爪夹紧异常延时
T0632 BOOL  ; 下料#3夹爪张开异常延时
T0633 BOOL  ; 下料#3夹爪夹紧异常延时
T0634 BOOL  ; 下料#4夹爪张开异常延时
T0635 BOOL  ; #4下料夹爪夹紧异常延时
T0636 BOOL  ; #1合模气缸缩回异常延时
T0637 BOOL  ; #合模气缸伸出异常延时
T0638 BOOL  ; #2合模气缸缩回异常延时
T0639 BOOL  ; #2合模气缸伸出异常延时
T0640 BOOL  ; #3合模气缸缩回异常延时
T0641 BOOL  ; #3合模气缸伸出异常延时
T0642 BOOL  ; #4合模气缸缩回异常延时
T0643 BOOL  ; #4合模气缸伸出异常延时
T0644 BOOL  ; 出料移栽伸缩气缸缩回异常延时
T0645 BOOL  ; 出料移栽伸缩气缸伸出异常延时
T0646 BOOL  ; 检测NG推料气缸缩回异常延时
T0647 BOOL  ; 检测NG推料气缸伸出异常延时
T0648 BOOL  ; 出料#1夹爪张开异常延时
T0649 BOOL  ; 出料#1夹爪夹紧异常延时
T0650 BOOL  ; 出料#2夹爪张开异常延时
T0651 BOOL  ; 出料#2夹爪夹紧异常延时
T0652 BOOL  ; 进料伺服使能异常延时
T0653 BOOL  ; 进料升降伺服异常延时
T0654 BOOL  ; 进料移栽伺服异常延时
T0655 BOOL  ; 上料水平伺服异常延时
T0656 BOOL  ; 下料水平伺服异常延时
T0657 BOOL  ; 出料水平伺服异常延时
T0658 BOOL  ; 出料升降伺服异常延时
T0659 BOOL  ; 出料移栽伺服异常延时
T0680 BOOL  ; #1总氦检阀打开异常延时
T0681 BOOL  ; #1总氦检阀关闭异常延时
T0682 BOOL  ; #2总氦检阀打开异常延时
T0683 BOOL  ; #2总氦检阀关闭异常延时
T0684 BOOL  ; #1氦检阀打开异常延时
T0685 BOOL  ; #1氦检阀关闭异常延时
T0686 BOOL  ; #2氦检阀打开异常延时
T0687 BOOL  ; #2氦检阀关闭异常延时
T0688 BOOL  ; #3氦检阀打开异常延时
T0689 BOOL  ; #3氦检阀关闭异常延时
T0690 BOOL  ; #4氦检阀打开异常延时
T0691 BOOL  ; #4氦检阀关闭异常延时
T0700 BOOL  ; 扫码左阻挡缩回异常延时
T0701 BOOL  ; 扫码左阻挡伸出异常延时
T0702 BOOL  ; 扫码右阻挡缩回异常延时
T0703 BOOL  ; 扫码右阻挡伸出异常延时
T0704 BOOL  ; 左隔离气缸缩回异常延时
T0705 BOOL  ; 左隔离气缸伸出异常延时
T0706 BOOL  ; 右隔离气缸缩回异常延时
T0707 BOOL  ; 右隔离气缸伸出异常延时
T0708 BOOL  ; 扫码NG缓存推料气缸缩回异常延时
T0709 BOOL  ; 扫码NG推料气缸伸出异常延时
T0710 BOOL  ; 进料移栽伸缩气缸缩回异常延时
T0711 BOOL  ; 进料移栽伸缩气缸伸出异常延时
T0900 BOOL  ; 读氦检仪报警延时
T0901 BOOL  ; 读氦检状态完成延时
T0902 BOOL  ; 氦检仪稳定时间
T0904 BOOL  ; 检漏口压力判断延时
T0905 BOOL  ; 漏率判断延时
T0906 BOOL  ; 氦检启动延时
T0907 BOOL  ; 氦检仪通讯异常时间
T0909 BOOL  ; 延时关校准
T1000 BOOL  ; #1扫码感应有料延时
T1001 BOOL  ; #2扫码感应有料延时
T1002 BOOL  ; 拉带放料延时感应
T1500 BOOL  ; 上料OK缓存记忆与感应不一致延时
T1501 BOOL  ; #1上料位记忆与感应延时
T1502 BOOL  ; #2上料位记忆与感应延时
T1503 BOOL  ; 进料移栽#1记忆与感应延时
T1504 BOOL  ; 进料移栽#2记忆与感应延时
T1505 BOOL  ; 下料#1夹爪记忆与感应延时
T1506 BOOL  ; 上料#2夹爪记忆与感应延时
T1507 BOOL  ; 上料#3夹爪记忆与感应延时
T1508 BOOL  ; #2腔体记忆与感应延时
T1509 BOOL  ; 下料#1夹爪记忆与感应延时
T1510 BOOL  ; 下料#2夹爪记忆与感应延时
T1511 BOOL  ; 下料#3夹爪记忆与感应延时
T1512 BOOL  ; 下料#4夹爪感应与记忆延时
T1513 BOOL  ; 移栽位记忆与感应延时
T1514 BOOL  ; 出料#1夹爪记忆与感应延时
T1515 BOOL  ; 出料#2夹爪记忆与感应延时
T1520 BOOL  ; #1腔体记忆与感应延时
T1521 BOOL  ; 上料#4夹爪记忆与感应延时
W0.00 BOOL  ; 门禁信号
W0.01 BOOL  ; 异常报警停止
W0.02 BOOL  ; 启动/停止
W0.03 BOOL  ; 启动按钮  HMI
W0.05 BOOL  ; 停止按钮  HMI
W0.06 BOOL  ; 清料按钮  HMI
W0.07 BOOL  ; 手/自动切换  HMI
W0.08 BOOL  ; 手/自动切换辅助
W0.10 BOOL  ; 氦检仪已稳定
W100.00 BOOL  ; 进料水平伺服上料位置设定按钮  HMI
W100.01 BOOL  ; 进料水平伺服左爪OK配对位置设定按钮  HMI
W100.02 BOOL  ; 进料水平伺服右爪OK配对位置设定按钮  HMI
W100.03 BOOL  ; 进料水平伺服左爪缓存位置设定按钮  HMI
W100.04 BOOL  ; 进料水平伺服右爪缓存位置设定按钮  HMI
W100.05 BOOL  ; 进料水平伺服缓存位置设定按钮  HMI
W100.06 BOOL  ; 备用
W100.07 BOOL  ; 备用
W100.08 BOOL  ; 备用
W100.09 BOOL  ; 进料水平伺服放料位置设定按钮  HMI
W100.10 BOOL  ; 备用
W100.11 BOOL  ; 备用
W100.12 BOOL  ; 进料升降伺服上料位置设定按钮  HMI
W100.13 BOOL  ; 进料升降伺服放料位置设定按钮  HMI
W100.14 BOOL  ; 进料升降伺服待料位置设定按钮  HMI
W100.15 BOOL  ; 进料旋转伺服#1待料位置设定按钮  HMI
W101.00 BOOL  ; 进料旋转伺服#2待料位置设定按钮  HMI
W101.01 BOOL  ; 进料旋转伺服上料位置设定按钮  HMI
W101.02 BOOL  ; 上料水平伺服待料位置设定按钮  HMI
W101.03 BOOL  ; 上料水平伺服#1腔体位置设定按钮  HMI
W101.04 BOOL  ; 上料水平伺服#2腔体位置设定按钮  HMI
W101.05 BOOL  ; 下料水平伺服#1腔体位置设定按钮  HMI
W101.06 BOOL  ; 下料水平伺服#2腔体位置设定按钮  HMI
W101.07 BOOL  ; 下料水平伺服放料位置设定按钮  HMI
W101.08 BOOL  ; 出料水平伺服取料位置设定按钮  HMI
W101.09 BOOL  ; 出料水平伺服#1缓存位置设定按钮  HMI
W101.10 BOOL  ; 出料水平伺服#2缓存位置设定按钮  HMI
W101.11 BOOL  ; 出料水平伺服放料待机位置设定按钮  HMI
W101.13 BOOL  ; 出料水平伺服放料位置设定按钮  HMI
W101.14 BOOL  ; 出料升降伺服待料位置设定按钮  HMI
W101.15 BOOL  ; 出料升降伺服上料位置设定按钮  HMI
W102.00 BOOL  ; 出料升降伺服放料位置设定按钮  HMI
W102.01 BOOL  ; 出料旋转伺服#1出料位置设定按钮  HMI
W102.02 BOOL  ; 出料旋转伺服#2出料位置设定按钮  HMI
W102.03 BOOL  ; 出料旋转伺服待料位置设定按钮  HMI
W105.00 BOOL  ; 进料水平伺服归零辅助
W105.01 BOOL  ; 进料水平伺服前进辅助
W105.02 BOOL  ; 进料水平伺服后退辅助
W105.03 BOOL  ; 手动回进料水平伺服取料位辅助
W105.04 BOOL  ; 手动回进料水平伺服左爪OK配对位辅助
W105.05 BOOL  ; 手动回进料水平伺服右爪OK配对位辅助
W105.06 BOOL  ; 手动回进料水平伺服左爪缓存位辅助
W105.07 BOOL  ; 手动回进料水平伺服右爪缓存位辅助
W105.08 BOOL  ; 手动回进料水平伺服NG位辅助
W105.09 BOOL  ; 备用
W105.10 BOOL  ; 备用
W105.11 BOOL  ; 备用
W105.12 BOOL  ; 手动回进料水平伺服放料位辅助
W105.13 BOOL  ; 备用
W105.14 BOOL  ; 进料升降伺服取料位
W105.15 BOOL  ; 进料升降伺服归零辅助
W106.00 BOOL  ; 进料升降伺服下降
W106.01 BOOL  ; 进料升降伺服上升
W106.02 BOOL  ; 手动回进料升降伺服缓存位
W106.03 BOOL  ; 手动回进料升降伺服放料位辅助
W106.04 BOOL  ; 手动回进料升降伺服待料位辅助
W106.05 BOOL  ; 进料旋转伺服归零辅助
W106.06 BOOL  ; 进料旋转伺服前进辅助
W106.07 BOOL  ; 进料旋转伺服后退辅助
W106.08 BOOL  ; 手动回进料旋转伺服#1待料位辅助
W106.09 BOOL  ; 手动回进料旋转伺服#2待料位辅助
W106.10 BOOL  ; 手动回进料旋转伺服上料位辅助
W106.11 BOOL  ; 上料水平伺服归零辅助
W106.12 BOOL  ; 上料水平伺服前进辅助
W106.13 BOOL  ; 上料水平伺服后退辅助
W106.14 BOOL  ; 手动回上料水平伺服待料位辅助
W106.15 BOOL  ; 手动回上料水平伺服#1腔体位辅助
W107.00 BOOL  ; 手动回上料水平伺服#2腔体位辅助
W107.01 BOOL  ; 下料水平伺服归零辅助
W107.02 BOOL  ; 下料水平伺服前进辅助
W107.03 BOOL  ; 下料水平伺服后退辅助
W107.04 BOOL  ; 手动回下料水平伺服#1腔体位辅助
W107.05 BOOL  ; 手动回下料水平伺服#2腔体位辅助
W107.06 BOOL  ; 手动回下料水平伺服放料位辅助
W107.07 BOOL  ; 出料水平伺服归零辅助
W107.08 BOOL  ; 出料水平伺服前进辅助
W107.09 BOOL  ; 出料水平伺服后退辅助
W107.10 BOOL  ; 手动回出料水平伺服取料位辅助
W107.11 BOOL  ; 手动回出料水平伺服#1缓存位辅助
W107.12 BOOL  ; 手动回出料水平伺服#2缓存位辅助
W107.13 BOOL  ; 手动回出料水平伺服放料待机位置
W107.14 BOOL  ; 手动回出料水平伺服#4缓存位辅助
W107.15 BOOL  ; 手动回出料水平伺服放料位辅助
W108.00 BOOL  ; 出料升降伺服归零辅助
W108.01 BOOL  ; 出料升降伺服前进辅助
W108.02 BOOL  ; 出料升降伺服后退辅助
W108.03 BOOL  ; 手动回出料升降伺服待料位辅助
W108.04 BOOL  ; 手动回出料升降伺服NG缓存位辅助
W108.05 BOOL  ; 手动回出料升降伺服放料位辅助
W108.06 BOOL  ; 出料旋转伺服归零辅助
W108.07 BOOL  ; 出料移栽伺服前进辅助
W108.08 BOOL  ; 出料移栽伺服后退辅助
W108.09 BOOL  ; 手动回出料旋转伺服#1出料位辅助
W108.10 BOOL  ; 手动回出料旋转伺服#2出料位辅助
W108.11 BOOL  ; 手动回出料旋转伺服待料位辅助
W108.12 BOOL  ; 手动回出料水平伺服#5缓存位辅助
W108.13 BOOL  ; 手动回出料升降伺服取料位辅助
W109.15 BOOL  ; 手动回出料水平伺服#5缓存位辅助
W10.00 BOOL  ; 进料水平伺服归零   HMI
W10.01 BOOL  ; 进料水平伺服前进   HMI
W10.02 BOOL  ; 进料水平伺服后退   HMI
W10.03 BOOL  ; 手动回进料水平伺服取料位置  HMI
W10.04 BOOL  ; 手动回进料水平伺服左爪OK配对位置  HMI
W10.05 BOOL  ; 手动回进料水平伺服右爪OK配对位置  HMI
W10.06 BOOL  ; 手动回进料水平伺服左爪缓存位置  HMI
W10.07 BOOL  ; 手动回进料水平伺服右爪缓存位置  HMI
W10.08 BOOL  ; 手动进料水平伺服NG位置  HMI
W10.09 BOOL  ; 备用
W10.10 BOOL  ; 备用
W10.11 BOOL  ; 备用
W10.12 BOOL  ; 手动回进料水平伺服放料位置  HMI
W10.13 BOOL  ; 备用
W10.14 BOOL  ; 备用
W10.15 BOOL  ; 进料升降伺服归零   HMI
W110.00 BOOL  ; 自动回进料水平伺服上料位辅助
W110.01 BOOL  ; 自动回进料水平伺服左配对位辅助
W110.02 BOOL  ; 自动回进料水平伺服右配对位辅助
W110.03 BOOL  ; 自动回进料水平伺服左爪缓存位辅助
W110.04 BOOL  ; 自动回进料水平伺服右爪缓存位辅助
W110.05 BOOL  ; 自动回进料水平伺服缓存位辅助
W110.06 BOOL  ; 备用
W110.07 BOOL  ; 备用
W110.08 BOOL  ; 备用
W110.09 BOOL  ; 进料水平伺自动回服放料位辅助
W110.10 BOOL  ; 备用
W110.11 BOOL  ; 备用
W110.12 BOOL  ; 自动回进料升降伺服缓存位辅助
W110.13 BOOL  ; 自动回进料升降伺服放料位辅助
W110.14 BOOL  ; 自动回进料升降伺服待料位辅助
W110.15 BOOL  ; 自动回进料旋转伺服#1待料位辅助
W111.00 BOOL  ; 自动回进料旋转伺服#2待料位辅助
W111.01 BOOL  ; 自动回进料旋转伺服上料位辅助
W111.02 BOOL  ; 自动回上料水平伺服待料位辅助
W111.03 BOOL  ; 自动回上料水平伺服#1腔体位辅助
W111.04 BOOL  ; 自动回上料水平伺服#2腔体位辅助
W111.05 BOOL  ; 自动回下料水平伺服#1腔体位辅助
W111.06 BOOL  ; 自动回下料水平伺服#2腔体位辅助
W111.07 BOOL  ; 自动回下料水平伺服放料位辅助
W111.08 BOOL  ; 自动回出料水平伺服取料位辅助
W111.09 BOOL  ; 自动回出料水平伺服#1缓存位辅助
W111.10 BOOL  ; 自动回出料水平伺服#2缓存位辅助
W111.11 BOOL  ; 出料水平伺服自动回放料待机位
W111.13 BOOL  ; 出料水平伺服自动回放料位
W111.14 BOOL  ; 自动回出料升降伺服待料位辅助
W111.15 BOOL  ; 自动回出料升降伺服取料位辅助
W112.00 BOOL  ; 自动回出料升降伺服放料位辅助
W112.01 BOOL  ; 自动回出料旋转伺服#1出料位辅助
W112.02 BOOL  ; 自动回出料旋转伺服#2出料位辅助
W112.03 BOOL  ; 自动回出料旋转伺服待料位辅助
W112.04 BOOL  ; 自动回出料升降伺服NG放料位辅助
W112.05 BOOL  ; 备用
W112.06 BOOL  ; 备用
W112.07 BOOL  ; 备用
W112.08 BOOL  ; 备用
W112.09 BOOL  ; 备用
W112.10 BOOL  ; 备用
W112.11 BOOL  ; 备用
W112.12 BOOL  ; 备用
W112.13 BOOL  ; 备用
W112.14 BOOL  ; 备用
W112.15 BOOL  ; 备用
W115.00 BOOL  ; 进料水平伺服在取料位
W115.01 BOOL  ; 进料水平伺服在左爪OK配对位
W115.02 BOOL  ; 进料水平伺服在右爪OK配对位
W115.03 BOOL  ; 进料水平伺服在左爪缓存位
W115.04 BOOL  ; 进料水平伺服在右爪缓存位
W115.05 BOOL  ; 进料水平伺服在NG位
W115.06 BOOL  ; 备用
W115.07 BOOL  ; 备用
W115.08 BOOL  ; 备用
W115.09 BOOL  ; 进料水平伺服在放料位
W115.10 BOOL  ; 备用
W115.11 BOOL  ; 进料升降伺服取料位
W115.12 BOOL  ; 进料升降伺服在缓存位
W115.13 BOOL  ; 进料升降伺服在放料位
W115.14 BOOL  ; 进料升降伺服在待料位
W115.15 BOOL  ; 进料旋转伺服在#1待料位
W116.00 BOOL  ; 进料旋转伺服在#2待料位
W116.01 BOOL  ; 进料旋转伺服在上料位
W116.02 BOOL  ; 上料料水平伺服在待料位
W116.03 BOOL  ; 上料料水平伺服在#1腔体位
W116.04 BOOL  ; 上料料水平伺服在#2腔体位
W116.05 BOOL  ; 下料水平伺服在#1腔体位
W116.06 BOOL  ; 下料水平伺服在#2腔体位
W116.07 BOOL  ; 下料水平伺服在放料位
W116.08 BOOL  ; 出料水平伺服在取料位
W116.09 BOOL  ; 出料水平伺服在#1缓存位
W116.10 BOOL  ; 出料水平伺服在#2缓存位
W116.11 BOOL  ; 出料水平伺服在放料待机位
W116.12 BOOL  ; 出料水平伺服在#4缓存位
W116.13 BOOL  ; 出料水平伺服在放料位
W116.14 BOOL  ; 出料升降伺服在待料位
W116.15 BOOL  ; 出料升降伺服在取料位
W117.00 BOOL  ; 出料升降伺服在放料位
W117.01 BOOL  ; 出料移栽伺服在#1出料位
W117.02 BOOL  ; 出料移栽伺服在#2出料位
W117.03 BOOL  ; 出料移栽伺服在待料位
W117.04 BOOL  ; 进料水平伺服在原点位置
W117.05 BOOL  ; 进料升降伺服在原点位置
W117.06 BOOL  ; 进料旋转伺服在原点位置
W117.07 BOOL  ; 上料水平伺服在原点位置
W117.08 BOOL  ; 下料水平伺服在原点位置
W117.09 BOOL  ; 出料水平伺服在原点位置
W117.10 BOOL  ; 出料升降伺服在原点位置
W117.11 BOOL  ; 出料移栽伺服在原点位置
W117.13 BOOL  ; 出料升降伺服在NG缓存位
W117.14 BOOL  ; 备用
W117.15 BOOL  ; 备用
W118.00 BOOL  ; 备用
W118.01 BOOL  ; 备用
W118.02 BOOL  ; 出料移栽伸缩气缸安全条件
W118.03 BOOL  ; 进料夹爪安全条件
W118.04 BOOL  ; 进料伸缩气缸安全移动条件
W118.10 BOOL  ; 上下料水平伺服距离过小
W118.11 BOOL  ; 下料水平伺服回腔体#1安全条件
W118.12 BOOL  ; 下料水平伺服回腔体#2安全条件
W118.13 BOOL  ; 上料机械手回腔体#1安全条件
W118.14 BOOL  ; 上料机械手回腔体#2安全条件
W118.15 BOOL  ; 上料水平提升气缸安全条件
W119.00 BOOL  ; 下料水平伺服提升气缸安全条件
W119.06 BOOL  ; 出料水平伺服安全移动条件
W11.00 BOOL  ; 进料升降伺服前进   HMI
W11.01 BOOL  ; 进料升降伺服后退   HMI
W11.02 BOOL  ; 手动回进料升降伺服缓存位  HMI
W11.03 BOOL  ; 手动回进料升降伺服放料位置  HMI
W11.04 BOOL  ; 手动回进料升降伺服待料位置  HMI
W11.05 BOOL  ; 进料旋转伺服归零   HMI
W11.06 BOOL  ; 进料旋转伺服前进   HMI
W11.07 BOOL  ; 进料旋转伺服后退   HMI
W11.08 BOOL  ; 手动回进料旋转伺服#1待料位置  HMI
W11.09 BOOL  ; 手动回进料旋转伺服#2待料位置  HMI
W11.10 BOOL  ; 手动回进料旋转伺服上料位置  HMI
W11.11 BOOL  ; 上料水平伺服归零   HMI
W11.12 BOOL  ; 上料水平伺服前进   HMI
W11.13 BOOL  ; 上料水平伺服后退   HMI
W11.14 BOOL  ; 手动回上料水平伺服待料位置  HMI
W11.15 BOOL  ; 手动回上料水平伺服#1腔体位置  HMI
W120.00 BOOL  ; 扫码2#位隔离气缸缩回(M)
W120.01 BOOL  ; 扫码2#位隔离气缸伸出(M)
W120.02 BOOL  ; 扫码1#位隔离气缸缩回(M)
W120.03 BOOL  ; 扫码1#位隔离气缸伸出(M)
W120.04 BOOL  ; 扫码2#位阻挡气缸缩回(M)
W120.05 BOOL  ; 扫码2#位阻挡气缸伸出(M)
W120.06 BOOL  ; 扫码1#位阻挡气缸缩回(M)
W120.07 BOOL  ; 扫码1#位阻挡气缸伸出(M)
W120.08 BOOL  ; #1调速电机辅助
W120.09 BOOL  ; #2调速电机辅助
W120.10 BOOL  ; #3调速电机辅助
W120.11 BOOL  ; #4调速电机辅助
W120.13 BOOL  ; 进料水平伺服使能辅助
W120.14 BOOL  ; 进料升降伺服使能辅助
W120.15 BOOL  ; 进料升降伺服刹车辅助
W121.00 BOOL  ; 进料移栽伺服使能辅助
W121.01 BOOL  ; 扫码缓存推料气缸辅助伸出
W121.02 BOOL  ; 扫码缓存推料气缸辅助缩回
W121.03 BOOL  ; 进料旋转伸缩气缸辅助伸出
W121.04 BOOL  ; 进料旋转伸缩气缸辅助缩回
W121.05 BOOL  ; 进料1#夹爪气缸辅助夹紧
W121.06 BOOL  ; 进料1#夹爪气缸辅助松开
W121.07 BOOL  ; 进料2#夹爪气缸辅助夹紧
W121.08 BOOL  ; 进料2#夹爪气缸辅助松开
W121.10 BOOL  ; 上料提升气缸辅助
W121.13 BOOL  ; 腔体上料伺服使能辅助
W121.14 BOOL  ; 腔体上料提升气缸辅助下降
W121.15 BOOL  ; 腔体上料提升气缸辅助上升
W122.00 BOOL  ; 腔体上料#1夹爪气缸辅助夹紧
W122.01 BOOL  ; 腔体上料#1夹爪气缸辅助松开
W122.02 BOOL  ; 腔体上料#2夹爪气缸辅助夹紧
W122.03 BOOL  ; 腔体上料#2夹爪气缸辅助松开
W122.04 BOOL  ; 腔体上料#3夹爪气缸辅助夹紧
W122.05 BOOL  ; 腔体上料#3夹爪气缸辅助松开
W122.06 BOOL  ; 腔体上料#4夹爪气缸辅助夹紧
W122.07 BOOL  ; 腔体上料#4夹爪气缸辅助松开
W122.08 BOOL  ; 腔体下料伺服使能辅助
W122.09 BOOL  ; 腔体下料提升气缸辅助下降
W122.10 BOOL  ; 腔体下料提升气缸辅助上升
W122.11 BOOL  ; 腔体下料#1夹爪气缸辅助夹紧
W122.12 BOOL  ; 腔体下料#1夹爪气缸辅助松开
W122.13 BOOL  ; 腔体下料#2夹爪气缸辅助夹紧
W122.14 BOOL  ; 腔体下料#3夹爪气缸辅助松开
W122.15 BOOL  ; 腔体下料#3夹爪气缸辅助夹紧
W123.00 BOOL  ; 腔体下料#3夹爪气缸辅助松开
W123.01 BOOL  ; 腔体下料#4夹爪气缸辅助夹紧
W123.02 BOOL  ; 腔体下料#4夹爪气缸辅助松开
W123.03 BOOL  ; 备用
W123.04 BOOL  ; 备用
W123.05 BOOL  ; 备用
W123.06 BOOL  ; 备用
W123.07 BOOL  ; #1合模气缸手动缩回
W123.08 BOOL  ; #1合模气缸手动伸出
W123.09 BOOL  ; #2合模气缸辅助缩回
W123.10 BOOL  ; #2合模气缸辅助伸出
W123.11 BOOL  ; #3合模气缸辅助缩回
W123.12 BOOL  ; #3合模气缸辅助伸出
W123.13 BOOL  ; #4合模气缸辅助缩回
W123.14 BOOL  ; #4合模气缸辅助伸出
W123.15 BOOL  ; 氦检阀#7辅助
W124.00 BOOL  ; 氦检阀#8辅助
W124.01 BOOL  ; 抽真空阀#1辅助
W124.02 BOOL  ; 抽真空阀#2辅助
W124.03 BOOL  ; 抽真空阀#3辅助
W124.04 BOOL  ; 抽真空阀#4辅助
W124.05 BOOL  ; 总氦检阀#1辅助
W124.06 BOOL  ; 总氦检阀#2辅助
W124.07 BOOL  ; 氦检阀#1辅助
W124.08 BOOL  ; 氦检阀#2辅助
W124.09 BOOL  ; 氦检阀#3辅助
W124.10 BOOL  ; 氦检阀#4辅助
W124.11 BOOL  ; 破真空阀#1辅助
W124.12 BOOL  ; 破真空阀#2辅助
W124.13 BOOL  ; 破真空阀#3辅助
W124.14 BOOL  ; 破真空阀#4辅助
W124.15 BOOL  ; 吹气阀#1辅助
W125.00 BOOL  ; 吹气阀#2辅助
W125.01 BOOL  ; 吹气阀#3辅助
W125.02 BOOL  ; 吹气阀#4辅助
W125.05 BOOL  ; 吹气阀#2辅助
W126.00 BOOL  ; 出料水平伺服使能辅助
W126.01 BOOL  ; 出料升降伺服使能辅助
W126.02 BOOL  ; 出料升降伺服刹车辅助
W126.03 BOOL  ; 出料旋转伺服使能辅助
W126.04 BOOL  ; 出料移栽伸缩气缸辅助伸出
W126.05 BOOL  ; 出料移栽伸缩气缸辅助缩回
W126.06 BOOL  ; 检测NG缓存推料气缸辅助伸出
W126.07 BOOL  ; 检测NG缓存推料气缸辅助缩回
W126.08 BOOL  ; 出料#1夹爪气缸辅助夹紧
W126.09 BOOL  ; 出料#1夹爪气缸辅助松开
W126.10 BOOL  ; 出料#2夹爪气缸辅助夹紧
W126.11 BOOL  ; 出料#2夹爪气缸辅助松开
W126.12 BOOL  ; 备用
W126.13 BOOL  ; 备用
W126.14 BOOL  ; 备用
W126.15 BOOL  ; 备用
W127.00 BOOL  ; 氦检仪启动辅助
W127.01 BOOL  ; #1真空泵辅助
W127.02 BOOL  ; #2真空泵辅助
W127.03 BOOL  ; 启动指示灯辅助
W127.04 BOOL  ; 停止指示灯辅助
W127.05 BOOL  ; 复位指示灯辅助
W127.06 BOOL  ; 三色红灯辅助
W127.07 BOOL  ; 三色黄灯辅助
W127.08 BOOL  ; 三色绿灯辅助
W127.09 BOOL  ; 蜂鸣器辅助
W127.10 BOOL  ; 扫码左位阻挡气缸辅助
W127.11 BOOL  ; 扫码右位阻挡气缸辅助
W127.13 BOOL  ; #1腔体自检开真空
W127.14 BOOL  ; #2腔体自检开真空
W128.01 BOOL  ; #2腔体自检#1抽真空阀关闭
W128.03 BOOL  ; #4腔体自检#3抽真空阀关闭
W128.04 BOOL  ; #3腔体自检#4抽真空阀关闭
W12.00 BOOL  ; 手动回上料水平伺服#2腔体位置  HMI
W12.01 BOOL  ; 下料水平伺服归零   HMI
W12.02 BOOL  ; 下料水平伺服前进   HMI
W12.03 BOOL  ; 下料水平伺服后退   HMI
W12.04 BOOL  ; 手动回下料水平伺服#1腔体位置  HMI
W12.05 BOOL  ; 手动回下料水平伺服#2腔体位置  HMI
W12.06 BOOL  ; 手动回下料水平伺服放料位置  HMI
W12.07 BOOL  ; 出料水平伺服归零   HMI
W12.08 BOOL  ; 出料水平伺服前进   HMI
W12.09 BOOL  ; 出料水平伺服后退   HMI
W12.10 BOOL  ; 手动回出料水平伺服取料位置  HMI
W12.11 BOOL  ; 手动回出料水平伺服#1缓存位置  HMI
W12.12 BOOL  ; 手动回出料水平伺服#2缓存位置  HMI
W12.13 BOOL  ; 手动回出料水平伺服放料待机位置 HMI
W12.14 BOOL  ; 手动回出料水平伺服#4缓存位置  HMI
W12.15 BOOL  ; 手动回出料水平伺服放料位置  HMI
W131.12 BOOL  ; 出料水平伺服在#5缓存位
W13.00 BOOL  ; 出料升降伺服归零   HMI
W13.01 BOOL  ; 出料升降伺服下降   HMI
W13.02 BOOL  ; 出料升降伺服上升   HMI
W13.03 BOOL  ; 手动回出料升降伺服待料位置  HMI
W13.04 BOOL  ; 手动回出料升降伺服取料位置  HMI
W13.05 BOOL  ; 手动回出料升降伺服放料位置  HMI
W13.06 BOOL  ; 出料旋转伺服归零   HMI
W13.07 BOOL  ; 出料移栽伺服前进   HMI
W13.08 BOOL  ; 出料移栽伺服后退   HMI
W13.09 BOOL  ; 手动回出料旋转伺服#1出料位置  HMI
W13.10 BOOL  ; 手动回出料旋转伺服#2出料位置  HMI
W13.11 BOOL  ; 手动回出料旋转伺服待料位置  HMI
W13.12 BOOL  ; 手动回出料水平伺服#5缓存位置  HMI
W13.13 BOOL  ; 手动回出料升降伺服取料位置  HMI
W13.14 BOOL  ; 备用
W13.15 BOOL  ; 备用
W145.04 BOOL  ; 旋转单元至卸载位（伸出）[PLS]
W145.05 BOOL  ; 旋转单元至装载位（缩回）[PLS]
W146.04 BOOL  ; 旋转单元至卸载位（伸出）辅助[A]
W146.05 BOOL  ; 旋转单元至装载位（缩回）辅助[A]
W146.08 BOOL  ; 出料#1夹爪气缸辅助夹紧[A]
W146.09 BOOL  ; 出料#1夹爪气缸辅助松开[A]
W146.10 BOOL  ; 出料#2夹爪气缸辅助夹紧[A]
W146.11 BOOL  ; 出料#2夹爪气缸辅助松开[A]
W146.12 BOOL  ; NG推料气缸伸出[A]
W146.13 BOOL  ; NG推料气缸缩回[A]
W14.01 BOOL  ; #1腔体自检步序
W14.02 BOOL  ; #1腔体自检步序
W14.02 BOOL  ; #2腔体自检步序
W14.03 BOOL  ; #3腔体自检步序
W14.04 BOOL  ; #4腔体自检步序
W168.08 BOOL  ; 测试复检
W188.05 BOOL  ; 调试
W188.08 BOOL  ; 调试
W188.09 BOOL  ; 调试
W188.13 BOOL  ; PC数据调试
W188.14 BOOL  ; PC数据调试
W189.00 BOOL  ; 拉带调试
W189.01 BOOL  ; 拉带调试
W190.00 BOOL  ; 测试置位
W1.01 BOOL  ; 复位完成
W1.02 BOOL  ; 带料复位触发
W1.05 BOOL  ; 清料进行中
W1.08 BOOL  ; 进料机构在初始位
W1.10 BOOL  ; 上下料机构初始位
W1.12 BOOL  ; 腔体机构初始位
W1.14 BOOL  ; 出料机构初始位
W200.00 BOOL  ; 左右夹爪NG料
W200.01 BOOL  ; 左右夹爪扫码OK
W200.02 BOOL  ; 右配对开始（2#OK 1#NG）
W200.03 BOOL  ; 左配对开始（1#OK 2#NG）
W200.05 BOOL  ; 右配对完成
W200.06 BOOL  ; 左配对完成
W200.07 BOOL  ; 配对完成标志
W200.08 BOOL  ; 左夹爪放料完成
W200.09 BOOL  ; 右夹爪放料完成
W200.10 BOOL  ; 返回NG位放料标志
W200.11 BOOL  ; 启动放料配对
W200.12 BOOL  ; 放料缓存段完成标志
W200.13 BOOL  ; 进料夹爪取料完成
W200.14 BOOL  ; 1#放料完成信号
W200.15 BOOL  ; 2#放料完成信号
W201.00 BOOL  ; 下部机构抓取完成信号
W201.01 BOOL  ; 启动配对缓存程序段
W201.11 BOOL  ; 上料水平伺服归零(Lamp)
W201.14 BOOL  ; 手动回上料水平伺服待料位(Lamp)
W201.15 BOOL  ; 手动回上料水平伺服#1腔体位(Lamp)
W202.00 BOOL  ; 手动回上料水平伺服#2腔体位(Lamp)
W202.01 BOOL  ; 下料水平伺服归零(Lamp)
W202.04 BOOL  ; 手动回下料水平伺服#1腔体位(Lamp)
W202.05 BOOL  ; 手动回下料水平伺服#2腔体位(Lamp)
W202.06 BOOL  ; 下料水平伺服在放料位(Lamp)
W20.00 BOOL  ; 扫码2#位隔离气缸伸出   HMI按钮
W20.01 BOOL  ; 扫码2#位隔离气缸缩回   HMI按钮
W20.02 BOOL  ; 扫码1#位隔离气缸缩回   HMI按钮
W20.03 BOOL  ; 扫码1#位隔离气缸伸出   HMI按钮
W20.04 BOOL  ; 扫码2#位阻挡气缸缩回   HMI按钮
W20.05 BOOL  ; 扫码左位阻挡气缸伸出  HMI按钮
W20.06 BOOL  ; 扫码1#位阻挡气缸缩回   HMI按钮
W20.07 BOOL  ; 扫码1#位阻挡气缸伸出   HMI按钮
W20.08 BOOL  ; #1调速电机   HMI按钮
W20.09 BOOL  ; #2调速电机   HMI按钮
W20.10 BOOL  ; #3调速电机   HMI按钮
W20.11 BOOL  ; #4调速电机   HMI按钮
W211.01 BOOL  ; 抽真空阀#1自检打开
W211.07 BOOL  ; #1合模气缸自检缩回
W211.08 BOOL  ; #1合模气缸自检伸出
W211.11 BOOL  ; #1自检破真空
W212.02 BOOL  ; 抽真空阀#2自检打开
W212.09 BOOL  ; #2合模气缸自检缩回
W212.10 BOOL  ; #2合模气缸自检伸出
W212.12 BOOL  ; #2自检破真空
W213.03 BOOL  ; 抽真空阀#3自检打开
W213.11 BOOL  ; #3合模气缸自检缩回
W213.12 BOOL  ; #3合模气缸自检伸出
W213.13 BOOL  ; #3腔体自检破真空阀
W214.04 BOOL  ; 抽真空阀#4自检打开
W214.13 BOOL  ; #4合模气缸自检缩回
W214.14 BOOL  ; #4合模气缸自检伸出
W215.00 BOOL  ; #1腔体抽真空失败
W215.01 BOOL  ; #1腔体自检结束
W215.08 BOOL  ; #1腔体自检#2抽真空阀关闭
W216.00 BOOL  ; #2腔体抽真空失败
W216.01 BOOL  ; #2腔体自检结束
W216.07 BOOL  ; #2腔体自检#1抽真空阀关闭
W217.00 BOOL  ; #3腔体抽真空失败
W217.01 BOOL  ; #3腔体自检结束
W217.10 BOOL  ; #3腔体自检#4抽真空阀关闭
W218.00 BOOL  ; #4腔体抽真空失败
W218.01 BOOL  ; #4腔体自检结束
W218.09 BOOL  ; #4腔体自检#3抽真空阀关闭
W218.13 BOOL  ; #4腔体自检破真空阀
W21.01 BOOL  ; 扫码缓存推料气缸伸出   HMI按钮
W21.02 BOOL  ; 扫码缓存推料气缸缩回   HMI按钮
W21.03 BOOL  ; 进料旋转伸缩气伸出   HMI按钮
W21.04 BOOL  ; 进料旋转伸缩气缩回   HMI按钮
W21.05 BOOL  ; 进料夹爪#1气缸夹紧   HMI按钮
W21.06 BOOL  ; 进料夹爪#1气缸松开   HMI按钮
W21.07 BOOL  ; 进料夹爪#2气缸夹紧   HMI按钮
W21.08 BOOL  ; 进料夹爪#2气缸松开   HMI按钮
W21.14 BOOL  ; 腔体上料提升气缸下降   HMI按钮
W21.15 BOOL  ; 腔体上料提升气缸上升   HMI按钮
W221.01 BOOL  ; #1腔体抽真空阀
W221.02 BOOL  ; #2腔体抽真空阀
W221.05 BOOL  ; #1总氦检阀
W221.07 BOOL  ; #1合模气缸缩回
W221.08 BOOL  ; #1合模气缸伸出
W221.09 BOOL  ; #2合模气缸缩回
W221.10 BOOL  ; #2合模气缸辅助伸出
W221.11 BOOL  ; #1腔体破真空阀
W221.15 BOOL  ; #1吹气阀
W223.03 BOOL  ; #3腔体抽真空阀
W223.04 BOOL  ; #4腔体抽真空阀
W223.06 BOOL  ; #2总氦检阀
W223.11 BOOL  ; #3合模气缸缩回
W223.12 BOOL  ; #3合模气缸伸出
W223.13 BOOL  ; #4合模气缸缩回
W223.14 BOOL  ; #4合模气缸辅助伸出
W224.01 BOOL  ; #3、#4吹气阀
W225.01 BOOL  ; 关#1腔体抽真空阀
W225.02 BOOL  ; 关#2腔体抽真空阀
W225.05 BOOL  ; 关#1总氦检阀
W225.07 BOOL  ; #2腔体复检检#1氦检阀关闭
W225.08 BOOL  ; #1腔体复检检#2氦检阀关闭
W225.11 BOOL  ; 关#1、#2腔体破真空阀
W226.01 BOOL  ; #1腔体复检打开抽真空阀条件
W226.02 BOOL  ; #2腔体复检打开抽真空阀条件
W226.07 BOOL  ; 复检检#1氦检阀打开
W226.08 BOOL  ; 复检检#2氦检阀打开
W227.03 BOOL  ; 关#3腔体抽真空阀
W227.04 BOOL  ; 关#4腔体抽真空阀
W227.06 BOOL  ; 关#2总氦检阀
W227.09 BOOL  ; #4腔体复检检#3氦检阀关闭
W227.10 BOOL  ; #3腔体复检检#4氦检阀关闭
W227.13 BOOL  ; #3、#4腔体破真空阀
W228.03 BOOL  ; #3腔体复检打开抽真空阀条件
W228.04 BOOL  ; #4腔体复检打开抽真空阀条件
W228.09 BOOL  ; 复检检#3氦检阀打开
W228.10 BOOL  ; 复检检#4氦检阀打开
W228.13 BOOL  ; 关#3、#4腔体破真空阀
W22.00 BOOL  ; 腔体上料#1夹爪气缸夹紧   HMI按钮
W22.01 BOOL  ; 腔体上料#1夹爪气缸松开   HMI按钮
W22.02 BOOL  ; 腔体上料#2夹爪气缸夹紧   HMI按钮
W22.03 BOOL  ; 腔体上料#2夹爪气缸松开   HMI按钮
W22.04 BOOL  ; 腔体上料#3夹爪气缸夹紧   HMI按钮
W22.05 BOOL  ; 腔体上料#3夹爪气缸松开   HMI按钮
W22.06 BOOL  ; 腔体上料#4夹爪气缸夹紧   HMI按钮
W22.07 BOOL  ; 腔体上料#4夹爪气缸松开   HMI按钮
W22.08 BOOL  ; 备用
W22.09 BOOL  ; 腔体下料提升气缸下降   HMI按钮
W22.10 BOOL  ; 腔体下料提升气缸上升   HMI按钮
W22.11 BOOL  ; 腔体下料#1夹爪气缸夹紧   HMI按钮
W22.12 BOOL  ; 腔体下料#1夹爪气缸松开   HMI按钮
W22.13 BOOL  ; 腔体下料#2夹爪气缸夹紧   HMI按钮
W22.14 BOOL  ; 腔体下料#2夹爪气缸松开   HMI按钮
W22.15 BOOL  ; 腔体下料#3夹爪气缸夹紧   HMI按钮
W231.00 BOOL  ; 自动回进料水平伺服上料位
W231.01 BOOL  ; 自动上料水平伺服去#1腔体位
W231.02 BOOL  ; 自动回上料水平伺服#2腔体位辅助
W231.05 BOOL  ; 上料水平伺服去腔体基本条件
W231.15 BOOL  ; 上料机构手自动运行
W232.00 BOOL  ; 上料#1夹爪气缸夹紧
W232.01 BOOL  ; 腔体上料#1夹爪气缸松开
W232.02 BOOL  ; 上料#2夹爪气缸夹紧
W232.03 BOOL  ; 腔体上料#2夹爪气缸松开
W232.04 BOOL  ; 上料#3夹爪气缸夹紧
W232.05 BOOL  ; 腔体上料#3夹爪气缸松开
W232.06 BOOL  ; 上料#4夹爪气缸夹紧
W232.07 BOOL  ; 腔体上料#4夹爪气缸松开
W232.14 BOOL  ; 腔体上料提升气缸下降
W232.15 BOOL  ; 腔体上料提升气缸上升
W233.00 BOOL  ; 自动回下料水平伺服放料位辅助
W233.01 BOOL  ; 自动回下料水平伺服#1腔体位
W233.02 BOOL  ; 自动回下料水平伺服#2腔体位
W233.15 BOOL  ; 下料机构手自动运行
W234.09 BOOL  ; 下料提升气缸下降
W234.10 BOOL  ; 腔体下料提升气缸辅助上升
W234.11 BOOL  ; 下料#1夹爪气缸辅助
W234.12 BOOL  ; 腔体下料#1夹爪气缸辅助松开
W234.13 BOOL  ; 下料#2夹爪气缸辅助
W234.14 BOOL  ; 腔体下料#2夹爪气缸辅助松开
W234.15 BOOL  ; 下料#3夹爪气缸辅助
W235.00 BOOL  ; 腔体下料#3夹爪气缸辅助松开
W235.01 BOOL  ; 下料#4夹爪气缸辅助
W235.02 BOOL  ; 腔体下料#4夹爪气缸辅助松开
W236.00 BOOL  ; 下料水平伺服自动回待料位条件
W236.03 BOOL  ; 下料机构到下步传数据条件
W236.04 BOOL  ; 下料机构手腔体夹料条件
W236.05 BOOL  ; 下料水平伺服自动去腔体条件
W236.09 BOOL  ; 下料机构手自动在腔体位下降条件
W23.00 BOOL  ; 腔体下料#3夹爪气缸松开   HMI按钮
W23.01 BOOL  ; 腔体下料#4夹爪气缸夹紧   HMI按钮
W23.02 BOOL  ; 腔体下料#4夹爪气缸松开   HMI按钮
W23.03 BOOL  ; 备用
W23.04 BOOL  ; 备用
W23.05 BOOL  ; 备用
W23.06 BOOL  ; 备用
W23.07 BOOL  ; #1合模气缸缩回   HMI按钮
W23.08 BOOL  ; #1合模气缸伸出   HMI按钮
W23.09 BOOL  ; #2合模气缸缩回   HMI按钮
W23.10 BOOL  ; #2合模气缸伸出   HMI按钮
W23.11 BOOL  ; #3合模气缸缩回   HMI按钮
W23.12 BOOL  ; #3合模气缸伸出   HMI按钮
W23.13 BOOL  ; #4合模气缸缩回   HMI按钮
W23.14 BOOL  ; #4合模气缸伸出   HMI按钮
W24.01 BOOL  ; 抽真空阀#1 开    HMI按钮
W24.02 BOOL  ; 抽真空阀#2 开    HMI按钮
W24.03 BOOL  ; 抽真空阀#3 开    HMI按钮
W24.04 BOOL  ; 抽真空阀#4 开    HMI按钮
W24.05 BOOL  ; #1总氦检阀 开    HMI按钮
W24.06 BOOL  ; #2总氦检阀 开    HMI按钮
W24.07 BOOL  ; 氦检阀#1 开   HMI按钮
W24.08 BOOL  ; 氦检阀#2 开   HMI按钮
W24.09 BOOL  ; 氦检阀#3 开   HMI按钮
W24.10 BOOL  ; 氦检阀#4 开   HMI按钮
W24.11 BOOL  ; 破真空阀#1 开   HMI按钮
W24.12 BOOL  ; 破真空阀#2 开   HMI按钮
W24.13 BOOL  ; 破真空阀#3 开   HMI按钮
W24.14 BOOL  ; 破真空阀#4 开   HMI按钮
W24.15 BOOL  ; 吹气阀#1 开   HMI按钮
W256.08 BOOL  ; 屏蔽
W25.00 BOOL  ; 吹气阀#2 开   HMI按钮
W25.01 BOOL  ; 吹气阀#3 开   HMI按钮
W25.02 BOOL  ; 吹气阀#4 开   HMI按钮
W26.04 BOOL  ; 出料移栽伸缩气缸伸出  HMI按钮
W26.05 BOOL  ; 出料移栽伸缩气缸缩回  HMI按钮
W26.06 BOOL  ; 检测NG缓存推料气缸伸出   HMI按钮
W26.07 BOOL  ; 检测NG缓存推料气缸缩回   HMI按钮
W26.08 BOOL  ; 出料#1夹爪气缸夹紧   HMI按钮
W26.09 BOOL  ; 出料#1夹爪气缸松开   HMI按钮
W26.10 BOOL  ; 出料#2夹爪气缸夹紧   HMI按钮
W26.11 BOOL  ; 出料#2夹爪气缸松开   HMI按钮
W27.00 BOOL  ; 氦检仪启动   HMI按钮
W27.01 BOOL  ; #1真空泵启动   HMI按钮
W27.02 BOOL  ; #2真空泵   HMI按钮
W27.03 BOOL  ; 启动按钮信号   HMI按钮
W27.04 BOOL  ; 停止按钮信号   HMI按钮
W27.05 BOOL  ; 复位按钮信号   HMI按钮
W27.09 BOOL  ; 蜂鸣器  HMI按钮
W27.10 BOOL  ; 扫码左位阻挡气缸  HMI按钮
W27.11 BOOL  ; 扫码右位阻挡气缸  HMI按钮
W28.01 BOOL  ; 抽真空阀#1 关    HMI按钮
W28.02 BOOL  ; 抽真空阀#2 关    HMI按钮
W28.03 BOOL  ; 抽真空阀#3 关    HMI按钮
W28.04 BOOL  ; 抽真空阀#4 关    HMI按钮
W28.05 BOOL  ; #1总氦检阀 关    HMI按钮
W28.06 BOOL  ; #2总氦检阀 关    HMI按钮
W28.07 BOOL  ; 氦检阀#1 关   HMI按钮
W28.08 BOOL  ; 氦检阀#2 关   HMI按钮
W28.09 BOOL  ; 氦检阀#3 关   HMI按钮
W28.10 BOOL  ; 氦检阀#4 关   HMI按钮
W28.11 BOOL  ; 破真空阀#1 关   HMI按钮
W28.12 BOOL  ; 破真空阀#2 关   HMI按钮
W28.13 BOOL  ; 破真空阀#3 关   HMI按钮
W28.14 BOOL  ; 破真空阀#4 关   HMI按钮
W28.15 BOOL  ; 吹气阀#1 关   HMI按钮
W29.00 BOOL  ; 吹气阀#2 关   HMI按钮
W29.01 BOOL  ; 吹气阀#3 关   HMI按钮
W29.02 BOOL  ; 吹气阀#4 关   HMI按钮
W29.11 BOOL  ; #1真空泵关闭  HMI按钮
W29.12 BOOL  ; #2真空泵关闭  HMI
W300.00 BOOL  ; 扫码左阻挡缩回异常
W300.01 BOOL  ; 扫码左阻挡伸出异常
W300.02 BOOL  ; 扫码右阻挡缩回异常
W300.03 BOOL  ; 扫码右阻挡伸出异常
W300.04 BOOL  ; 左隔离气缸缩回异常
W300.05 BOOL  ; 左隔离气缸伸出异常
W300.06 BOOL  ; 右隔离气缸缩回异常
W300.07 BOOL  ; 右隔离气缸伸出异常
W300.08 BOOL  ; 扫码NG缓存推料气缸缩回异常
W300.09 BOOL  ; 扫码NG推料气缸伸出异常
W300.10 BOOL  ; 进料移栽伸缩气缸缩回异常
W300.11 BOOL  ; 进料移栽伸缩气缸伸出异常
W300.12 BOOL  ; 进料#1夹爪张开异常
W300.13 BOOL  ; 进料#1夹爪夹紧异常
W300.14 BOOL  ; 进料#2夹爪张开异常
W300.15 BOOL  ; 进料#2夹爪夹紧异常
W301.00 BOOL  ; 上料提升气缸上升异常
W301.01 BOOL  ; 上料提升气缸下降异常
W301.02 BOOL  ; 上料#1夹爪张开异常
W301.03 BOOL  ; 上料#1夹爪夹紧异常
W301.04 BOOL  ; 上料#2夹爪张开异常
W301.05 BOOL  ; 上料#2夹爪夹紧异常
W301.06 BOOL  ; 上料#3夹爪张开异常
W301.07 BOOL  ; 上料#3夹爪夹紧异常
W301.08 BOOL  ; 上料#4夹爪张开异常
W301.09 BOOL  ; 上料#4夹爪夹紧异常
W301.10 BOOL  ; 下料提升气缸上升异常
W301.11 BOOL  ; 下料提升气缸下降异常
W301.12 BOOL  ; 下料#1夹爪张开异常
W301.13 BOOL  ; 下料#1夹爪夹紧异常
W301.14 BOOL  ; 下料#2夹爪张开异常
W301.15 BOOL  ; 下料#2夹爪夹紧异常
W302.00 BOOL  ; 下料#3夹爪张开异常
W302.01 BOOL  ; 下料#夹爪夹紧异常
W302.02 BOOL  ; 下料#4夹爪张开异常
W302.03 BOOL  ; 下料#4夹爪夹紧异常
W302.04 BOOL  ; #1合模气缸缩回异常
W302.05 BOOL  ; #1合模气缸伸出异常
W302.06 BOOL  ; #2合模气缸缩回延时
W302.07 BOOL  ; #2合模气缸伸出异常
W302.08 BOOL  ; #1总氦检阀打开异常
W302.09 BOOL  ; #1氦检阀打开异常
W302.10 BOOL  ; #2氦检阀打开异常
W303.00 BOOL  ; #3合模气缸缩回异常
W303.01 BOOL  ; #3合模气缸伸出异常
W303.02 BOOL  ; #4合模气缸缩回异常
W303.03 BOOL  ; #4合模气缸伸出异常
W303.04 BOOL  ; #2总氦检阀打开异常
W303.05 BOOL  ; #3氦检阀打开异常
W303.06 BOOL  ; #4氦检阀打开异常
W304.00 BOOL  ; 进料移栽伺服正极限异常
W304.01 BOOL  ; 进料移栽伺服负极限异常
W304.03 BOOL  ; 上料水平伺服负极限异常
W304.04 BOOL  ; 下料水平伺服正极限异常
W304.05 BOOL  ; 下料水平伺服负极限异常
W304.06 BOOL  ; 出料水平伺服正极限异常
W304.07 BOOL  ; 出料水平伺服负极限异常
W304.08 BOOL  ; 出料升降伺服正极限异常
W304.09 BOOL  ; 出料升降伺服负极限异常
W304.10 BOOL  ; 出料移栽伺服正极限异常
W304.11 BOOL  ; 出料移栽伺服负极限异常
W304.12 BOOL  ; 进料升降伺服柔性异常
W304.13 BOOL  ; 上料提升气缸柔性异常
W304.14 BOOL  ; 下料提升气缸柔性异常
W304.15 BOOL  ; 出料升降伺服柔性异常
W305.00 BOOL  ; 前门打开
W305.01 BOOL  ; 后门打开
W305.02 BOOL  ; 左门打开
W305.03 BOOL  ; 右门打开
W305.04 BOOL  ; 气源压力过低或供气异常
W305.05 BOOL  ; PLC与电脑通讯异常
W305.06 BOOL  ; 氦检仪没稳定！！
W305.07 BOOL  ; 紧急停止
W306.01 BOOL  ; 进料移栽伺服异常
W306.02 BOOL  ; 上料水平伺服异常
W306.03 BOOL  ; 下料水平伺服异常
W306.04 BOOL  ; 进料水平伺服正极限异常
W306.05 BOOL  ; 进料水平伺服负极限异常
W306.06 BOOL  ; 进料升降伺服负极限异常
W306.07 BOOL  ; 进料升降伺服正极限异常
W307.00 BOOL  ; 出料移栽伸缩气缸缩回异常
W307.01 BOOL  ; 出料移栽伸缩气缸伸出异常
W307.02 BOOL  ; 检测NG推料气缸缩回异常
W307.03 BOOL  ; 检测NG推料气缸伸出异常
W307.06 BOOL  ; 出料#1夹爪张开异常
W307.07 BOOL  ; 出料#1夹爪夹紧异常
W307.08 BOOL  ; 出料#2夹爪张开异常
W307.09 BOOL  ; 出料#2夹爪夹紧异常
W307.10 BOOL  ; 出料水平伺服异常
W307.11 BOOL  ; 出料升降伺服异常
W307.12 BOOL  ; 出料移栽伺服异常
W309.01 BOOL  ; 扫码NG槽满料
W309.02 BOOL  ; 上料OK缓存记忆与感应不一致
W309.03 BOOL  ; #1上料位记忆与感应不一致
W309.04 BOOL  ; #2上料位记忆与感应不一致
W309.05 BOOL  ; 进料移栽#1记忆与感应不一致
W309.06 BOOL  ; 进料移栽#2记忆与感应不一致
W309.07 BOOL  ; 下料#1夹爪记忆与感应不一致
W309.08 BOOL  ; 上料#2夹爪记忆与感应不一致
W309.09 BOOL  ; 上料#3夹爪记忆与感应不一致
W309.10 BOOL  ; 上料#4夹爪记忆与感应不一致
W309.11 BOOL  ; 下料#1夹爪记忆与感应不一致
W309.12 BOOL  ; 下料#2夹爪记忆与感应不一致
W309.13 BOOL  ; 下料#3夹爪记忆与感应不一致
W309.14 BOOL  ; 下料#4夹爪记忆与感应不一致
W309.15 BOOL  ; 移栽位记忆与感应不一致
W30.00 BOOL  ; 1#位手动扫码  HMI
W30.01 BOOL  ; 1#位自动扫码
W30.02 BOOL  ; 1#位重复扫码
W30.03 BOOL  ; 1#位扫码完成
W30.04 BOOL  ; 1#位扫码OK
W30.05 BOOL  ; 1#位扫码失败
W30.07 BOOL  ; 左来料扫码检测OK
W30.08 BOOL  ; 1#来料扫码检测NG
W30.13 BOOL  ; 1#位扫码已完成
W310.00 BOOL  ; 出料#1夹爪记忆与感应不一致
W310.01 BOOL  ; 出料#2夹爪记忆与感应不一致
W310.02 BOOL  ; 检测NG满料
W310.04 BOOL  ; #1腔体记忆与感应不一致
W310.05 BOOL  ; #2腔体记忆与感应不一致
W31.00 BOOL  ; 2#位手动扫码
W31.01 BOOL  ; 2#位自动扫码
W31.02 BOOL  ; 2#位重复扫码
W31.03 BOOL  ; 2#位扫码完成
W31.04 BOOL  ; 2#位扫码OK
W31.05 BOOL  ; 2#位扫码失败
W31.07 BOOL  ; 右来料扫码检测OK
W31.08 BOOL  ; 2#来料扫码检测NG
W31.13 BOOL  ; 2#位扫码已完成
W327.05 BOOL  ; 下料水平伺服无原点
W32.00 BOOL  ; 氦检仪当前为检漏状态
W32.01 BOOL  ; 读氦检仪状态完成
W32.02 BOOL  ; 读检漏口压力
W32.03 BOOL  ; 读检漏口压力完成
W32.05 BOOL  ; 读漏率
W32.06 BOOL  ; 读漏率完成
W32.07 BOOL  ; 读漏率失败
W32.08 BOOL  ; 读氦检仪状态失败
W32.09 BOOL  ; 读检漏口压力失败
W32.10 BOOL  ; 读氦检仪报警
W33.00 BOOL  ; 氦检仪检漏状态
W33.01 BOOL  ; 氦检仪待机状态
W33.02 BOOL  ; 氦检仪启动状态
W33.03 BOOL  ; 氦检仪定标状态
W33.04 BOOL  ; 氦检仪错误
W33.05 BOOL  ; 氦检仪暂停状态
W33.09 BOOL  ; 校准完成
W33.10 BOOL  ; 校准出错
W33.11 BOOL  ; 校准中
W33.13 BOOL  ; 下工位回可放料
W34.00 BOOL  ; #1、#2腔体氦检正常结束
W34.01 BOOL  ; #1、#2腔体氦检异常结束
W34.02 BOOL  ; #1腔体抽真空异常结束
W34.03 BOOL  ; #1、#2腔体氦检进行中标记
W34.13 BOOL  ; 手动信号输出对接
W35.00 BOOL  ; #1复检氦检正常结束
W35.01 BOOL  ; #1复检氦检异常结束
W35.02 BOOL  ; #1复检抽真空异常结束
W35.03 BOOL  ; #1、#2腔体复检氦检进行中标记
W35.09 BOOL  ; #1复检清氦失败
W35.10 BOOL  ; 清氦失败后跳过再次清氦按钮
W35.11 BOOL  ; #1复检前抽真空完成
W36.00 BOOL  ; #2复检氦检正常结束
W36.01 BOOL  ; #2复检氦检异常结束
W36.02 BOOL  ; #2复检抽真空异常结束
W36.08 BOOL  ; #2腔体抽真空失败
W36.09 BOOL  ; #2复检清氦失败
W37.00 BOOL  ; #3、#4腔体氦检正常结束
W37.01 BOOL  ; #3、#4腔体氦检异常结束
W37.02 BOOL  ; #3腔体抽真空异常结束
W37.03 BOOL  ; #3、#4腔体氦检进行中标记
W38.00 BOOL  ; #3复检氦检正常结束
W38.01 BOOL  ; #3复检氦检异常结束
W38.02 BOOL  ; #3复检抽真空异常结束
W38.03 BOOL  ; #3、#4腔体复检氦检进行中标记
W38.09 BOOL  ; #3复检清氦失败
W38.10 BOOL  ; 清氦失败后跳过再次清氦按钮
W38.11 BOOL  ; #3复检前抽真空完成
W39.00 BOOL  ; #4复检氦检正常结束
W39.01 BOOL  ; #4复检氦检异常结束
W39.02 BOOL  ; #4复检抽真空异常结束
W39.08 BOOL  ; #4腔体抽真空失败
W39.09 BOOL  ; #4复检清氦失败
W39.11 BOOL  ; #4复检前抽真空完成
W3.00 BOOL  ; 进料拉带记忆清除（SW）
W3.04 BOOL  ; #1腔体有NG物料
W3.05 BOOL  ; #3 & #4腔体有NG物料
W3.06 BOOL  ; 扫码有NG物料
W3.08 BOOL  ; 进料夹爪#1清料
W3.09 BOOL  ; 进料夹爪#2清料
W3.10 BOOL  ; 上料夹爪#1清料
W3.11 BOOL  ; 上料夹爪#2清料
W3.12 BOOL  ; 上料夹爪#3清料
W3.13 BOOL  ; 上料夹爪#4清料
W3.14 BOOL  ; 下料夹爪#1清料
W3.15 BOOL  ; 下料夹爪#2清料
W40.01 BOOL  ; 进料机构复位启动
W40.10 BOOL  ; 进料机构复位
W41.00 BOOL  ; 进料升降伺服归零
W41.01 BOOL  ; 进料升降伺服回待料位
W41.02 BOOL  ; 进料水平伺服归零
W41.03 BOOL  ; 进料水平伺服回取料位
W41.04 BOOL  ; 进料旋转伺服归零
W41.05 BOOL  ; 进料旋转伺服回上料位
W41.06 BOOL  ; 2#隔离气缸缩回复位
W41.07 BOOL  ; 1#隔离气缸缩回复位
W41.08 BOOL  ; 扫码2#阻挡气缸伸出复位
W41.09 BOOL  ; 扫码1#阻挡气缸伸出复位
W41.10 BOOL  ; NG缓存推料气缸缩回复位
W41.11 BOOL  ; 进料旋转伸缩气缸伸出复位
W41.12 BOOL  ; 进料1#夹爪气缸夹紧
W41.13 BOOL  ; 进料1#夹爪气缸松开复位
W41.14 BOOL  ; 进料2#夹爪气缸夹紧复位
W41.15 BOOL  ; 进料2#夹爪气缸松开复位
W4.00 BOOL  ; 下料夹爪#3清料
W4.01 BOOL  ; 下料夹爪#4清料
W4.02 BOOL  ; 出料夹爪#1清料
W4.03 BOOL  ; 出料2夹爪清除
W4.04 BOOL  ; #1腔体有料清除
W4.05 BOOL  ; #2腔体有料清除
W4.10 BOOL  ; 进料移栽有料清除
W4.11 BOOL  ; 出料移栽有料清除
W500.00 BOOL  ; 上料位没料记忆
W500.01 BOOL  ; 进料夹爪没记忆
W500.02 BOOL  ; 扫码记忆状态
W500.05 BOOL  ; 升降触发条件
W501.00 BOOL  ; 启动条件
W502.00 BOOL  ; 上料夹爪没有料记忆
W502.01 BOOL  ; 出料移栽没料
W502.02 BOOL  ; 下料夹爪没有料标志
W502.04 BOOL  ; 进料夹爪无料状态
W502.05 BOOL  ; 进料#2夹爪无料状态
W50.00 BOOL  ; 进料机构自动开始
W50.01 BOOL  ; 上料机构手复位启动
W50.02 BOOL  ; 进料输送机构自动运行
W50.10 BOOL  ; 上下料机构手复位
W50.11 BOOL  ; 下料机构复位启动
W510.00 BOOL  ; 进料1#夹爪气缸夹紧
W510.01 BOOL  ; 进料2#夹爪气缸夹紧
W510.02 BOOL  ; 进料旋转伸缩气缸伸出
W510.03 BOOL  ; 进料1#夹爪气缸辅助松开
W510.04 BOOL  ; 进料2#夹爪气缸辅助松开
W510.05 BOOL  ; 进料旋转气缸伸出
W510.06 BOOL  ; 进料旋转气缸缩回
W510.10 BOOL  ; 进料输送马达
W510.11 BOOL  ; 扫码2#隔离气缸缩回
W510.12 BOOL  ; 扫码2#隔离气缸伸出
W510.13 BOOL  ; 1#隔离气缸缩回
W510.14 BOOL  ; 1#隔离气缸伸出
W510.15 BOOL  ; 2#阻挡气缸缩回
W511.00 BOOL  ; 2#阻挡气缸伸出
W511.01 BOOL  ; 1#阻挡气缸缩回
W511.02 BOOL  ; 1#阻挡气缸伸出
W511.03 BOOL  ; NG缓存推料气缸伸出
W511.04 BOOL  ; NG缓存推料气缸缩回
W51.00 BOOL  ; 腔体上料#1夹爪气缸夹紧复位(M)
W51.01 BOOL  ; 腔体上料#1夹爪气缸松开复位(M)
W51.02 BOOL  ; 腔体上料#2夹爪气缸夹紧复位(M)
W51.03 BOOL  ; 腔体上料#2夹爪气缸松开复位(M)
W51.04 BOOL  ; 腔体上料#3夹爪气缸夹紧复位(M)
W51.05 BOOL  ; 腔体上料#3夹爪气缸松开复位(M)
W51.06 BOOL  ; 腔体上料#4夹爪气缸夹紧复位(M)
W51.07 BOOL  ; 腔体上料#4夹爪气缸松开复位(M)
W51.10 BOOL  ; 腔体上料伺服复位(M)
W51.15 BOOL  ; 腔体上料提升气缸上升复位(M)
W52.00 BOOL  ; 腔体下料#3夹爪气缸松开复位(M)
W52.01 BOOL  ; 腔体下料#4夹爪气缸夹紧复位(M)
W52.02 BOOL  ; 腔体下料#4夹爪气缸松开复位(M)
W52.08 BOOL  ; 腔体下料伺服复位
W52.10 BOOL  ; 腔体下料提升气缸上升复位(M)
W52.11 BOOL  ; 腔体下料#1夹爪气缸夹紧复位(M)
W52.12 BOOL  ; 腔体下上料#1夹爪气缸松开复位(M)
W52.13 BOOL  ; 腔体下料#2夹爪气缸夹紧复位(M)
